// TIA Portal V20 export
// export: Created 2025-12-01T14:56:32.2454153Z, ExportSetting None, DisplayName Totally Integrated Automation Portal, DisplayVersion V20 Update 3, DisplayName TIA Portal Openness, DisplayVersion V20 Update 3, DisplayName TIA Portal Version Control Interface, DisplayVersion V20 Update 3, DisplayName STEP 7 Professional, DisplayVersion V20 Update 3, DisplayName STEP 7 Safety, DisplayVersion V20 Update 2, DisplayName WinCC Basic/Comfort/Advanced, DisplayVersion V20 Update 3, DisplayName WinCC Professional, DisplayVersion V20 Update 3, DisplayName WinCC Unified, DisplayVersion V20 Update 3
FUNCTION_BLOCK "FB450_CRTL_TR_TP_E1_S234_AusSIM+Ord"   // FB450, LAD
TITLE = Control del Ramal de Salidas
{ S7_Optimized_Access := 'FALSE' }
AUTHOR : TLigero
NAME : 20191014
VERSION : 3.3
// FECHA:    19/03/2018  AUTOR: Alonso se parte de E1_S23
//                  19/03/2018                Alonso se mete orden del JdT
// stored: AutoNumber false, SetENOAutomatically false
   VAR_INPUT
      Mesa : UInt;   // Número de mesa
      En_tension : Bool;
      pHsMx_E1 : Bool;   // pHs DE AUSENCIA de la Mesa en E1
      pHsMx_S2 : Bool;   // pHs DE AUSENCIA de la Mesa en S2
      pHsMx_S3 : Bool;   // pHs DE AUSENCIA de la Mesa en S3
      pHsMx_S4 : Bool;   // pHs DE AUSENCIA de la Mesa en S4
      PosTR_E1 : Bool;   // Posicion del TR en E1E3
      PosTR_E2 : Bool;   // Posicion del TR en E2E4
      TP1_Up : Bool;   // TP1 Arriba. E1 >> S3. si no hay tope poner ON
      TP1_Down : Bool;   // TP1 Abajo. E1 >> S3. si no hay tope poner ON
      Termico_E1S3 : Bool;   // Proteccion del Tx en E1E3
      Termico_S2S4 : Bool;   // Proteccion del Tx en E2E4
      Avance_E1S3 : Bool;   // Avance del Tx en E1E3
      Avance_S2S4 : Bool;   // Avance del Tx en E2E4
      PTF_Sal_M2 : Bool;   // S2 >> Mesa Siguiente PTF
      NXT_Avance_S2 : Bool;   // S2 >> Mesa Siguiente avanzando
      PTF_Sal_M3 : Bool;   // S3 >> Mesa Siguiente PTF
      NXT_Avance_S3 : Bool;   // S3 >> Mesa Siguiente avanzando
      PTF_Sal_M4 : Bool;   // S4 >> Mesa Siguiente PTF
      NXT_Avance_S4 : Bool;   // S4 >> Mesa Siguiente avanzando
      F_EnvMens_Mx : Bool;   // Fin de Envio de Mensaje
      Mx_BloqActivo : Bool;   // Bloqueo Activo de la Mesa
      Mx_FlujoPrin_S2 : Bool;   // El flujo principal es Saliendo por S2
      Mx_FlujoPrin_S4 : Bool;   // El flujo principal es Saliendo por S4
      AVTF_MAnt_Mx : Bool;   // E1 >> Mesa Anterior AVTF
      Habilitar_orden_JDT : Bool;   // El JDT tendrá el control del cruce con orden
      ValorOrden_S2 : Word := 16#81;   // Valor de la orden para salir por S2
      ValorOrden_S4 : Word := 16#82;   // Valor de la orden para salir por S4
      MesaS2 : UInt;   // Número de mesa por S2
      MesaS3 : UInt;   // Número de mesa por S3
      MesaS4 : UInt;   // Número de mesa por S4
      Num_Cruce : UInt;   // Número de cruce.
      DB_FIFO_Cruce : UInt := 213;   // DB de la FIFO de ordenes del cruce
      Long_FIFO_Cruce : UInt := 1;   // Longitut de la FIFO de ordenes del cruce
      V_CNT_ApHsMx_E1 : UDInt := 250;   // Valor de Ausencia por E1 en ms
      V_CNT_ApHsMx_S2 : UDInt := 250;   // Valor de Ausencia por S2 en ms
      V_CNT_ApHsMx_S3 : UDInt := 250;   // Valor de Ausencia por S3 en ms
      V_CNT_ApHsMx_S4 : UDInt := 250;   // Valor de Ausencia por S4 en ms
      V_Vaciado : UDInt := 10000;   // Valor de vaciado en ms
      V_Estabilizacion_carga : UDInt := 10;   // en ms
      V_TOut_Tx_Mx : UDInt := 5000;   // TimeOut de Atasco en ms
      V_Avance_S2 : UDInt := 5000;   // en ms
      V_TOut_TR : UDInt := 5000;   // TimeOut de Transfer en ms
      V_TOut_TP : UDInt;   // TimeOut de Tope en ms
      V_Subir_TP_Min : UDInt;   // Valor Minimo para Subir Tope. Decimas de segundo
      V_Bajar_TP_Max : UDInt;   // Valor Maximo para Bajar Tope. Decimas de segundo
      V_Paro : UDInt := 4000;   // tiempo que avanza el transportador sin aviso hasta que se para (ms)
      V_Bloqueo_largo : Time := T#20s;   // tiempo
      V_Bloqueo_corto : Time := T#4s;   // tiempo
   END_VAR
   VAR_OUTPUT
      P_EnvMens_PMx : Bool;   // Permiso de Enviar Mensaje de Presencia
      Etiqueta_Jdt : UDInt;   // Etiqueta que ha sido leida
      Orden_Ejecutada_Jdt : UInt;   // Orden que se ha ejecutado
      PTF_MAnt_Mx : Bool;   // E1 >> Mesa Anterior PTF
      AVTF_Sal_M2 : Bool;   // S2 >> Mesa Siguiente descarga activa
      AVTF_Sal_M3 : Bool;   // S3 >> Mesa Siguiente AVTF
      AVTF_Sal_M4 : Bool;   // S4 >> Mesa Siguiente descarga activa
   END_VAR
   VAR
      T1_ET00 : Bool;
      T1_ET01 : Bool;
      T1_ET02 : Bool;
      T1_ET02_JdT : Bool;
      T1_ET03 : Bool;
      T1_ET10 : Bool;
      T1_ET11 : Bool;
      T1_ET12 : Bool;
      T1_ET50 : Bool;
      T1_ET60 : Bool;
      T1_ET70 : Bool;
      T1_ET80 : Bool;
      T1_ET81 : Bool;
      T1_ET110 : Bool;
      T1_ET111 : Bool;
      T1_ET112 : Bool;
      FIFO_OK : Bool;
      TRANS_OK : Bool;
      O_Bloqueo : Bool;
      Bloqueado : Bool;
      Err_Detec_PHS : Bool;
      FN_ET02 : Bool;
      FN_ET02_JdT : Bool;
      FP_ET02_JdT : Bool;
      FP_ET80 : Bool;
      MemFN_pHsE1 : Bool;
      MemFN_pHsS3 : Bool;
      MemFN_pHsS2 : Bool;
      MemFN_pHsS4 : Bool;
      MemAuxFN_pHsE1 : Bool;
      MemAuxFN_pHsS3 : Bool;
      MemAuxFN_pHsS2 : Bool;
      MemAuxFN_pHsS4 : Bool;
      OK_TmpAusE1 : Bool;
      OK_TmpAusS3 : Bool;
      OK_TmpAusS2 : Bool;
      OK_TmpAusS4 : Bool;
      maux_fp_disparo : Bool;
      ok_vaciado : Bool;
      CNT_Mov_TP : UDInt;
      TmpAus_E1 : UDInt;
      TmpAus_S2 : UDInt;
      TmpAus_S3 : UDInt;
      TmpAus_S4 : UDInt;
      TMP_Paro : UDInt;
      TOUT_Tope : UDInt;
      TOUT_Transfer : UDInt;
      TIMVacido : UDInt;
      TOUT_Atasco : UDInt;
      TOUT_S2 : UDInt;
      TSubidaTR : UDInt;
      TMP_Bloqueo : UDInt;
      TMP_En_Tension : UDInt;
      Datos_Scanner { S7_SetPoint := 'True'} : "ROUT_Orden_Fifo_Scanner";
   END_VAR
   VAR_TEMP
      EstadoZona : "EstadoZona";   // Estado de Zona de la Mesa
      EstadoVI : "EstadosMesa";   // Estado del Vehiculo Inteliguente de la Mesa
      ConfigFB : "UDT_ConfigFB";   // Configuracion de la FB de la Mesa
      TopeUp_EnEntrada : Bool;
      producto_estable : Bool;
      tout_avance_s2 : Bool;
      O_Continuar : Bool;
      O_Entrar_S2 : Bool;
      O_Entrar_S4 : Bool;
      O_Vaciar : Bool;
      JdT_Continuar : Bool;
      JdT_Entrar_S2 : Bool;
      JdT_Entrar_S4 : Bool;
      Moti_ERRO : Bool;
      Moti_NENC : Bool;
      Moti_NORM : Bool;
      Moti_INIC : Bool;
      OK_TP_DW : Bool;
      OK_Paro : Bool;
      t_bloqueo : Bool;
      atasco : Bool;
      timeout_tr : Bool;
      timeout_tope : Bool;
      ok_tension : Bool;
      Aux_W_Moti : Word;
      INT_ORDEN : UInt;
      Aux_W_Orden : Word;
      I_Ord_Filtrada : UInt;
      I_V_Ord_Entrar_S2 : UInt;
      I_V_Ord_Entrar_S4 : UInt;
      V_TMP_BLQ : UDInt;
   END_VAR
   VAR_TEMP   // added for the SCL form of the ladder/FBD networks
      _w1 : Bool;
      _w2 : Bool;
      _w3 : Bool;
      _w4 : Bool;
      _w5 : Bool;
      _w6 : Bool;
      _w7 : Bool;
   END_VAR
BEGIN

REGION Network 1: INICIALIZAR - Recoger las Variables de Estado de la Mesa
   // Se recoge - Estado_CBx
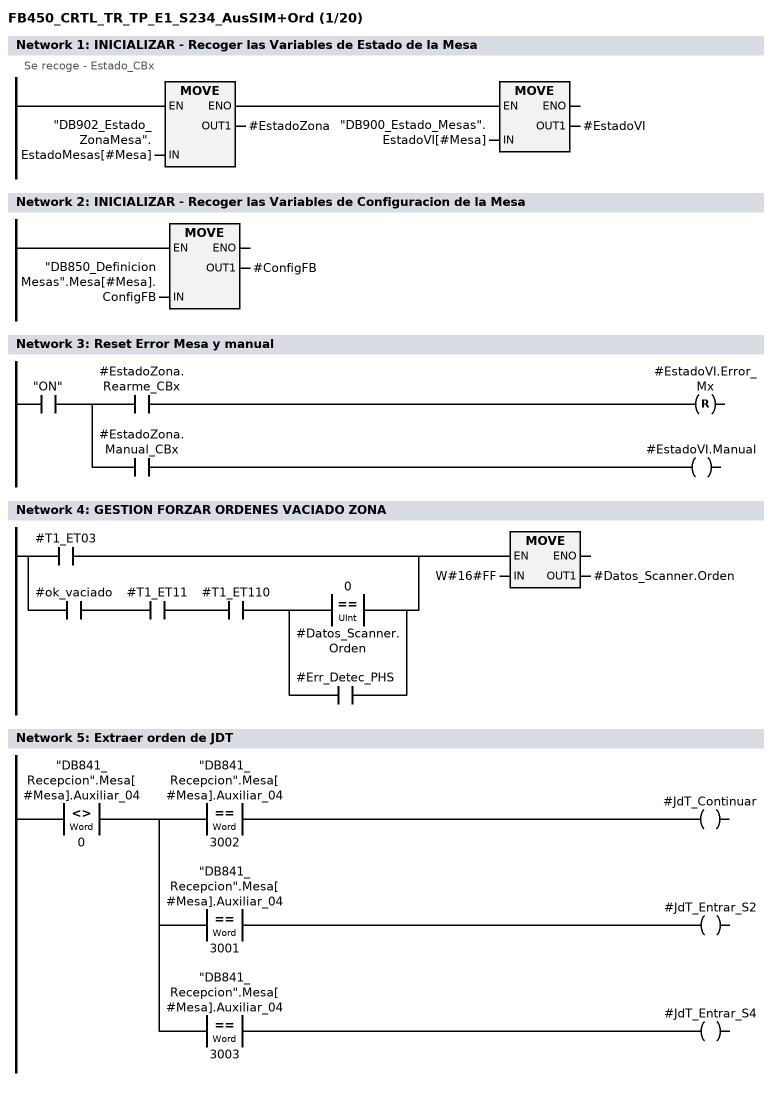
   RUNG wire#powerrail
      Move(in := "DB902_Estado_ZonaMesa".EstadoMesas[#Mesa], out1 => #EstadoZona)
      Move(in := "DB900_Estado_Mesas".EstadoVI[#Mesa], out1 => #EstadoVI)
   END_RUNG
   // the same network as SCL:
   #EstadoZona := "DB902_Estado_ZonaMesa".EstadoMesas[#Mesa];
   #EstadoVI := "DB900_Estado_Mesas".EstadoVI[#Mesa];
END_REGION

REGION Network 2: INICIALIZAR - Recoger las Variables de Configuracion de la Mesa
   RUNG wire#powerrail
      Move(in := "DB850_DefinicionMesas".Mesa[#Mesa].ConfigFB, out1 => #ConfigFB)
   END_RUNG
   // the same network as SCL:
   #ConfigFB := "DB850_DefinicionMesas".Mesa[#Mesa].ConfigFB;
END_REGION

REGION Network 3: Reset Error Mesa y manual
   RUNG wire#powerrail
      Contact( "ON" )
      wire#w1
      Contact( #EstadoZona.Rearme_CBx )
      R_Coil( #EstadoVI.Error_Mx )
   END_RUNG
   RUNG wire#w1
      Contact( #EstadoZona.Manual_CBx )
      Coil( #EstadoVI.Manual )
   END_RUNG
   // the same network as SCL:
   IF "ON" AND #EstadoZona.Rearme_CBx THEN #EstadoVI.Error_Mx := FALSE; END_IF;
   #EstadoVI.Manual := "ON" AND #EstadoZona.Manual_CBx;
END_REGION

REGION Network 4: GESTION FORZAR ORDENES VACIADO ZONA
   RUNG wire#powerrail
      Contact( #T1_ET03 )
      wire#w1
      { S7_GenerateENO := "TRUE" } Move(in := W#16#FF, out1 => #Datos_Scanner.Orden)
   END_RUNG
   RUNG wire#powerrail
      Contact( #ok_vaciado )
      Contact( #T1_ET11 )
      Contact( #T1_ET110 )
      wire#w2
      { S7_Templates := "SrcType := UInt" } EQ_Contact(in1 := 0, in2 := #Datos_Scanner.Orden)
   END_RUNG wire#w1
   RUNG wire#w2
      Contact( #Err_Detec_PHS )
   END_RUNG wire#w1
   // the same network as SCL:
   IF #T1_ET03 OR (#ok_vaciado AND #T1_ET11 AND #T1_ET110 AND ((0 = #Datos_Scanner.Orden) OR #Err_Detec_PHS)) THEN
       #Datos_Scanner.Orden := W#16#FF;
   END_IF;
END_REGION

REGION Network 5: Extraer orden de JDT
   RUNG wire#powerrail
      { S7_Templates := "SrcType := Word" } NE_Contact(in1 := "DB841_Recepcion".Mesa[#Mesa].Auxiliar_04, in2 := 0)
      wire#w1
      { S7_Templates := "SrcType := Word" } EQ_Contact(in1 := "DB841_Recepcion".Mesa[#Mesa].Auxiliar_04, in2 := 3002)
      Coil( #JdT_Continuar )
   END_RUNG
   RUNG wire#w1
      { S7_Templates := "SrcType := Word" } EQ_Contact(in1 := "DB841_Recepcion".Mesa[#Mesa].Auxiliar_04, in2 := 3001)
      Coil( #JdT_Entrar_S2 )
   END_RUNG
   RUNG wire#w1
      { S7_Templates := "SrcType := Word" } EQ_Contact(in1 := "DB841_Recepcion".Mesa[#Mesa].Auxiliar_04, in2 := 3003)
      Coil( #JdT_Entrar_S4 )
   END_RUNG
   // the same network as SCL:
   #_w1 := "DB841_Recepcion".Mesa[#Mesa].Auxiliar_04 <> 0;
   #JdT_Continuar := #_w1 AND ("DB841_Recepcion".Mesa[#Mesa].Auxiliar_04 = 3002);
   #JdT_Entrar_S2 := #_w1 AND ("DB841_Recepcion".Mesa[#Mesa].Auxiliar_04 = 3001);
   #JdT_Entrar_S4 := #_w1 AND ("DB841_Recepcion".Mesa[#Mesa].Auxiliar_04 = 3003);
END_REGION

REGION Network 6: extraer ordenes mesa
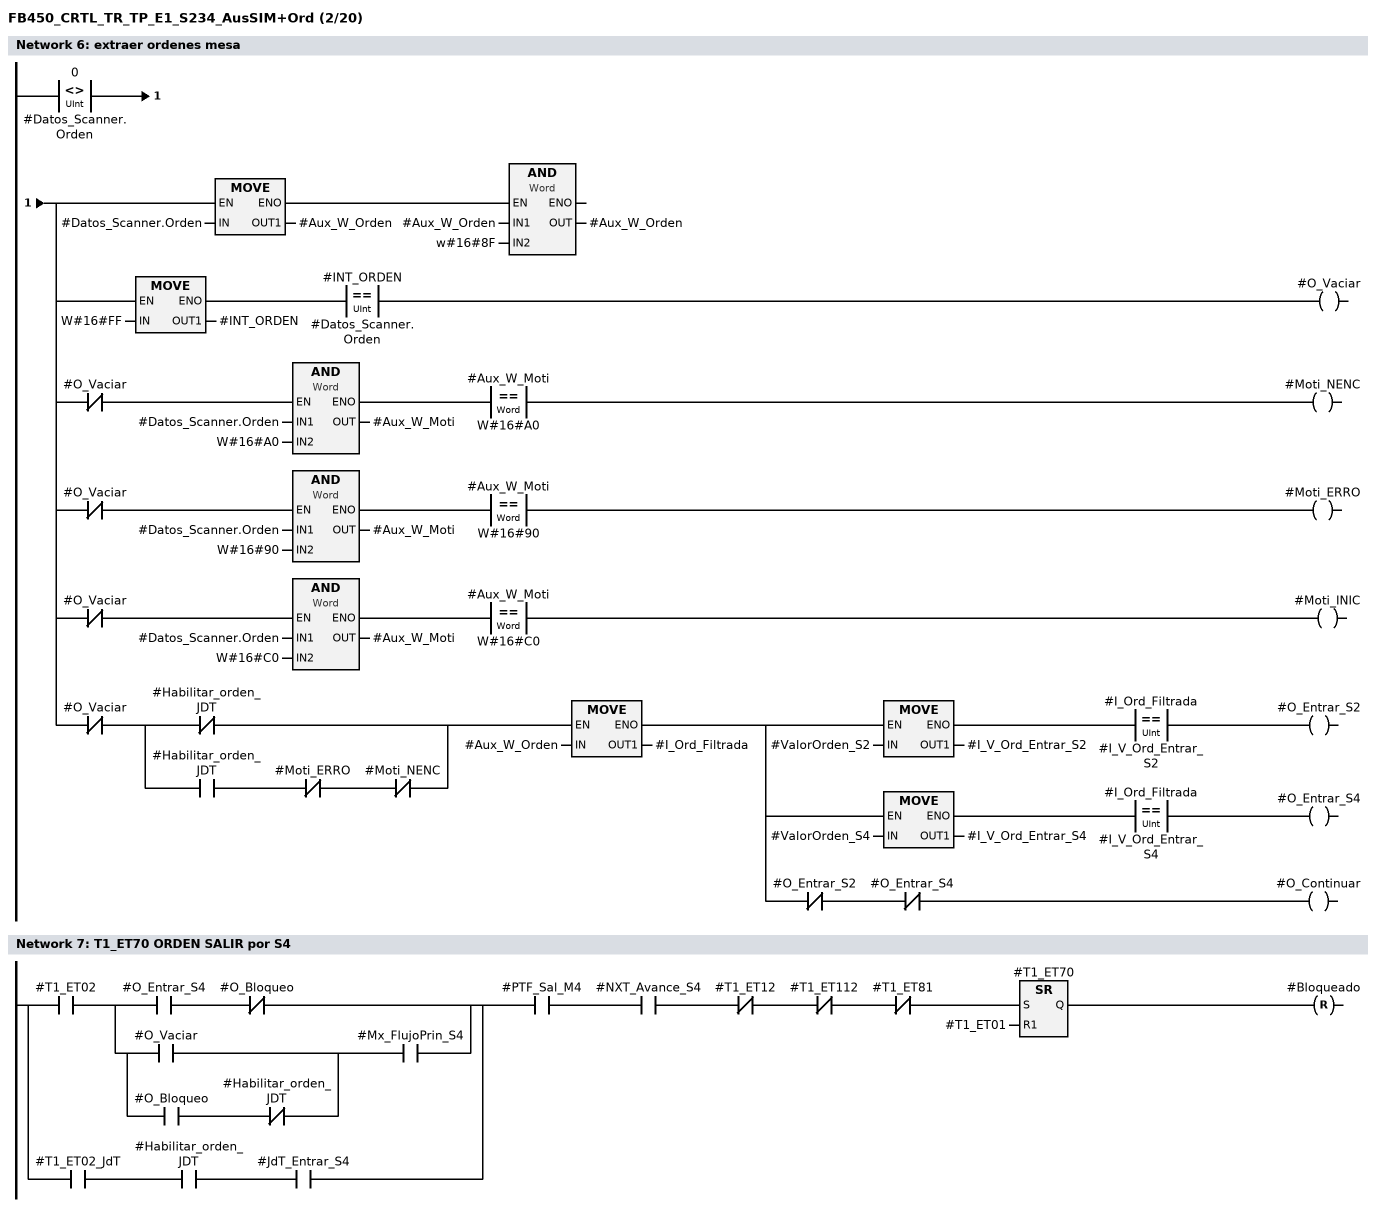
   RUNG wire#powerrail
      { S7_Templates := "SrcType := UInt" } NE_Contact(in1 := 0, in2 := #Datos_Scanner.Orden)
      wire#w1
      { S7_GenerateENO := "TRUE" } Move(in := #Datos_Scanner.Orden, out1 => #Aux_W_Orden)
      { S7_Templates := "SrcType := Word"; S7_GenerateENO := "TRUE" } And(in1 := #Aux_W_Orden, in2 := w#16#8F, out => #Aux_W_Orden)
   END_RUNG
   RUNG wire#w1
      { S7_GenerateENO := "TRUE" } Move(in := W#16#FF, out1 => #INT_ORDEN)
      { S7_Templates := "SrcType := UInt" } EQ_Contact(in1 := #INT_ORDEN, in2 := #Datos_Scanner.Orden)
      Coil( #O_Vaciar )
   END_RUNG
   RUNG wire#w1
      I_Contact( #O_Vaciar )
      { S7_Templates := "SrcType := Word"; S7_GenerateENO := "TRUE" } And(in1 := #Datos_Scanner.Orden, in2 := W#16#A0, out => #Aux_W_Moti)
      { S7_Templates := "SrcType := Word" } EQ_Contact(in1 := #Aux_W_Moti, in2 := W#16#A0)
      Coil( #Moti_NENC )
   END_RUNG
   RUNG wire#w1
      I_Contact( #O_Vaciar )
      { S7_Templates := "SrcType := Word"; S7_GenerateENO := "TRUE" } And(in1 := #Datos_Scanner.Orden, in2 := W#16#90, out => #Aux_W_Moti)
      { S7_Templates := "SrcType := Word" } EQ_Contact(in1 := #Aux_W_Moti, in2 := W#16#90)
      Coil( #Moti_ERRO )
   END_RUNG
   RUNG wire#w1
      I_Contact( #O_Vaciar )
      { S7_Templates := "SrcType := Word"; S7_GenerateENO := "TRUE" } And(in1 := #Datos_Scanner.Orden, in2 := W#16#C0, out => #Aux_W_Moti)
      { S7_Templates := "SrcType := Word" } EQ_Contact(in1 := #Aux_W_Moti, in2 := W#16#C0)
      Coil( #Moti_INIC )
   END_RUNG
   RUNG wire#w1
      I_Contact( #O_Vaciar )
      wire#w2
      I_Contact( #Habilitar_orden_JDT )
      wire#w3
      { S7_GenerateENO := "TRUE" } Move(in := #Aux_W_Orden, out1 => #I_Ord_Filtrada)
      wire#w4
      { S7_GenerateENO := "TRUE" } Move(in := #ValorOrden_S2, out1 => #I_V_Ord_Entrar_S2)
      { S7_Templates := "SrcType := UInt" } EQ_Contact(in1 := #I_Ord_Filtrada, in2 := #I_V_Ord_Entrar_S2)
      Coil( #O_Entrar_S2 )
   END_RUNG
   RUNG wire#w2
      Contact( #Habilitar_orden_JDT )
      I_Contact( #Moti_ERRO )
      I_Contact( #Moti_NENC )
   END_RUNG wire#w3
   RUNG wire#w4
      { S7_GenerateENO := "TRUE" } Move(in := #ValorOrden_S4, out1 => #I_V_Ord_Entrar_S4)
      { S7_Templates := "SrcType := UInt" } EQ_Contact(in1 := #I_Ord_Filtrada, in2 := #I_V_Ord_Entrar_S4)
      Coil( #O_Entrar_S4 )
   END_RUNG
   RUNG wire#w4
      I_Contact( #O_Entrar_S2 )
      I_Contact( #O_Entrar_S4 )
      Coil( #O_Continuar )
   END_RUNG
   // the same network as SCL:
   // ENO of a box is taken as its EN; it also drops when the box reports an error
   #_w1 := 0 <> #Datos_Scanner.Orden;
   IF #_w1 THEN
       #Aux_W_Orden := #Datos_Scanner.Orden;
       #Aux_W_Orden := #Aux_W_Orden AND w#16#8F;
       #INT_ORDEN := W#16#FF;
   END_IF;
   #O_Vaciar := #_w1 AND (#INT_ORDEN = #Datos_Scanner.Orden);
   #_w2 := #_w1 AND NOT #O_Vaciar;
   IF #_w2 THEN #Aux_W_Moti := #Datos_Scanner.Orden AND W#16#A0; END_IF;
   #Moti_NENC := #_w2 AND (#Aux_W_Moti = W#16#A0);
   #_w3 := #_w1 AND NOT #O_Vaciar;
   IF #_w3 THEN #Aux_W_Moti := #Datos_Scanner.Orden AND W#16#90; END_IF;
   #Moti_ERRO := #_w3 AND (#Aux_W_Moti = W#16#90);
   #_w4 := #_w1 AND NOT #O_Vaciar;
   IF #_w4 THEN #Aux_W_Moti := #Datos_Scanner.Orden AND W#16#C0; END_IF;
   #Moti_INIC := #_w4 AND (#Aux_W_Moti = W#16#C0);
   #_w5 := #_w1 AND NOT #O_Vaciar AND (NOT #Habilitar_orden_JDT OR (#Habilitar_orden_JDT AND NOT #Moti_ERRO AND NOT #Moti_NENC));
   IF #_w5 THEN
       #I_Ord_Filtrada := #Aux_W_Orden;
       #I_V_Ord_Entrar_S2 := #ValorOrden_S2;
   END_IF;
   #O_Entrar_S2 := #_w5 AND (#I_Ord_Filtrada = #I_V_Ord_Entrar_S2);
   IF #_w5 THEN #I_V_Ord_Entrar_S4 := #ValorOrden_S4; END_IF;
   #O_Entrar_S4 := #_w5 AND (#I_Ord_Filtrada = #I_V_Ord_Entrar_S4);
   #O_Continuar := #_w5 AND NOT #O_Entrar_S2 AND NOT #O_Entrar_S4;
END_REGION

REGION Network 7: T1_ET70 ORDEN SALIR por S4
   RUNG wire#powerrail
      Contact( #T1_ET02 )
      wire#w1
      Contact( #O_Entrar_S4 )
      I_Contact( #O_Bloqueo )
      wire#w2
      Contact( #PTF_Sal_M4 )
      Contact( #NXT_Avance_S4 )
      I_Contact( #T1_ET12 )
      I_Contact( #T1_ET112 )
      I_Contact( #T1_ET81 )
      S_SR(operand := #T1_ET70, r1 := #T1_ET01)
      R_Coil( #Bloqueado )
   END_RUNG
   RUNG wire#w1
      Contact( #O_Vaciar )
      wire#w3
      Contact( #Mx_FlujoPrin_S4 )
   END_RUNG wire#w2
   RUNG wire#w1
      Contact( #O_Bloqueo )
      I_Contact( #Habilitar_orden_JDT )
   END_RUNG wire#w3
   RUNG wire#powerrail
      Contact( #T1_ET02_JdT )
      Contact( #Habilitar_orden_JDT )
      Contact( #JdT_Entrar_S4 )
   END_RUNG wire#w2
   // the same network as SCL:
   IF ((#T1_ET02 AND ((#O_Entrar_S4 AND NOT #O_Bloqueo) OR ((#O_Vaciar OR (#O_Bloqueo AND NOT #Habilitar_orden_JDT)) AND #Mx_FlujoPrin_S4))) OR (#T1_ET02_JdT AND #Habilitar_orden_JDT AND #JdT_Entrar_S4)) AND #PTF_Sal_M4 AND #NXT_Avance_S4 AND NOT #T1_ET12 AND NOT #T1_ET112 AND NOT #T1_ET81 THEN
       #T1_ET70 := TRUE;   // SR flip-flop
   END_IF;
   IF #T1_ET01 THEN #T1_ET70 := FALSE; END_IF;
   IF #T1_ET70 THEN #Bloqueado := FALSE; END_IF;
END_REGION

REGION Network 8: T1_ET60 ORDEN SALIR por S2
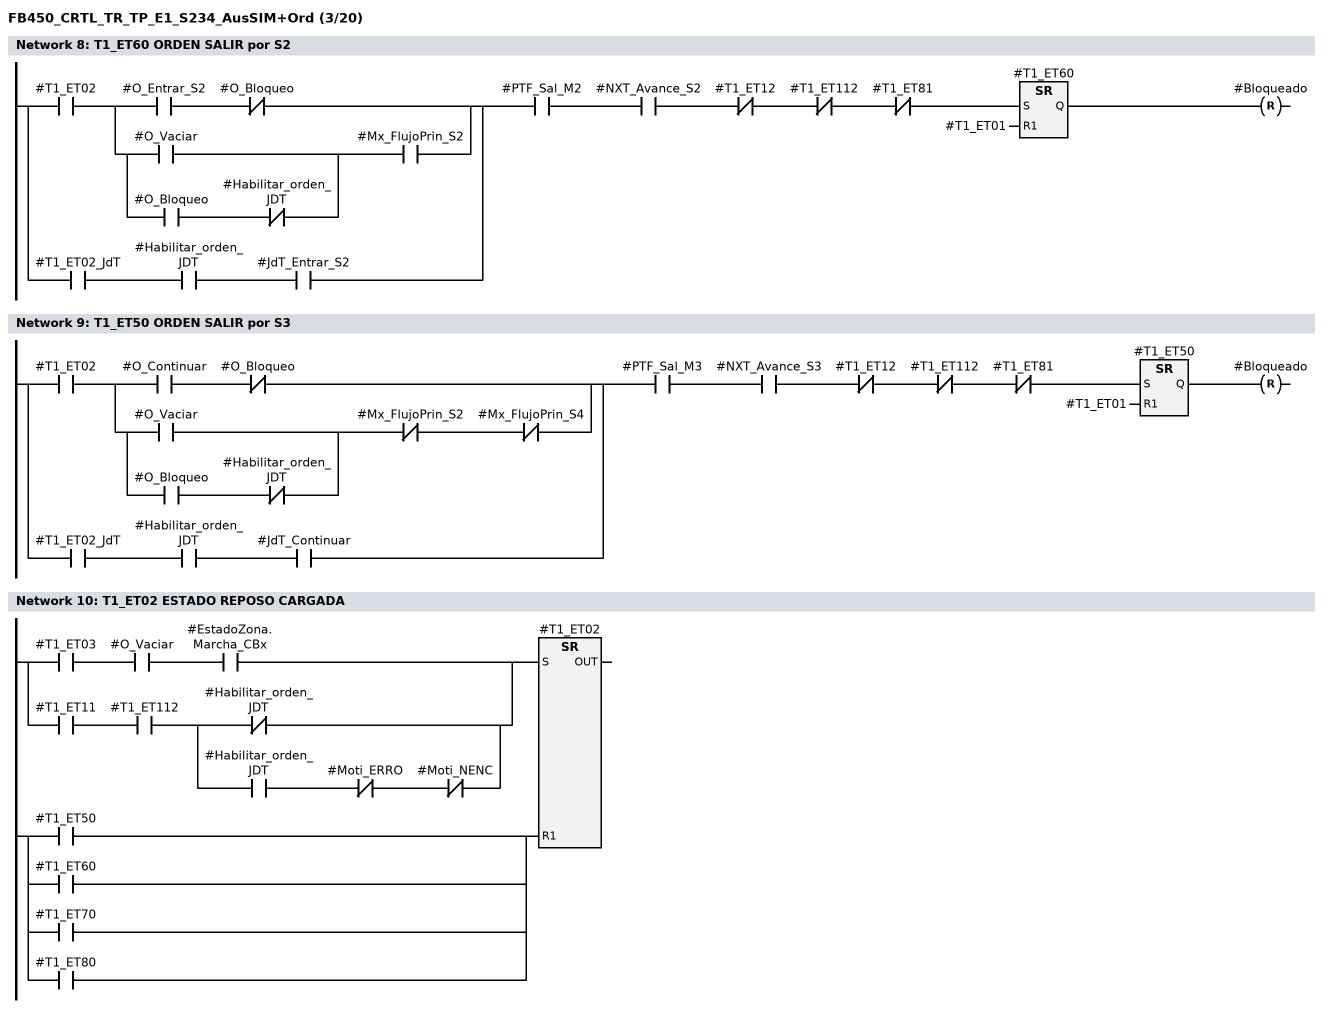
   RUNG wire#powerrail
      Contact( #T1_ET02 )
      wire#w1
      Contact( #O_Entrar_S2 )
      I_Contact( #O_Bloqueo )
      wire#w2
      Contact( #PTF_Sal_M2 )
      Contact( #NXT_Avance_S2 )
      I_Contact( #T1_ET12 )
      I_Contact( #T1_ET112 )
      I_Contact( #T1_ET81 )
      S_SR(operand := #T1_ET60, r1 := #T1_ET01)
      R_Coil( #Bloqueado )
   END_RUNG
   RUNG wire#w1
      Contact( #O_Vaciar )
      wire#w3
      Contact( #Mx_FlujoPrin_S2 )
   END_RUNG wire#w2
   RUNG wire#w1
      Contact( #O_Bloqueo )
      I_Contact( #Habilitar_orden_JDT )
   END_RUNG wire#w3
   RUNG wire#powerrail
      Contact( #T1_ET02_JdT )
      Contact( #Habilitar_orden_JDT )
      Contact( #JdT_Entrar_S2 )
   END_RUNG wire#w2
   // the same network as SCL:
   IF ((#T1_ET02 AND ((#O_Entrar_S2 AND NOT #O_Bloqueo) OR ((#O_Vaciar OR (#O_Bloqueo AND NOT #Habilitar_orden_JDT)) AND #Mx_FlujoPrin_S2))) OR (#T1_ET02_JdT AND #Habilitar_orden_JDT AND #JdT_Entrar_S2)) AND #PTF_Sal_M2 AND #NXT_Avance_S2 AND NOT #T1_ET12 AND NOT #T1_ET112 AND NOT #T1_ET81 THEN
       #T1_ET60 := TRUE;   // SR flip-flop
   END_IF;
   IF #T1_ET01 THEN #T1_ET60 := FALSE; END_IF;
   IF #T1_ET60 THEN #Bloqueado := FALSE; END_IF;
END_REGION

REGION Network 9: T1_ET50 ORDEN SALIR por S3
   RUNG wire#powerrail
      Contact( #T1_ET02 )
      wire#w1
      Contact( #O_Continuar )
      I_Contact( #O_Bloqueo )
      wire#w2
      Contact( #PTF_Sal_M3 )
      Contact( #NXT_Avance_S3 )
      I_Contact( #T1_ET12 )
      I_Contact( #T1_ET112 )
      I_Contact( #T1_ET81 )
      S_SR(operand := #T1_ET50, r1 := #T1_ET01)
      R_Coil( #Bloqueado )
   END_RUNG
   RUNG wire#w1
      Contact( #O_Vaciar )
      wire#w3
      I_Contact( #Mx_FlujoPrin_S2 )
      I_Contact( #Mx_FlujoPrin_S4 )
   END_RUNG wire#w2
   RUNG wire#w1
      Contact( #O_Bloqueo )
      I_Contact( #Habilitar_orden_JDT )
   END_RUNG wire#w3
   RUNG wire#powerrail
      Contact( #T1_ET02_JdT )
      Contact( #Habilitar_orden_JDT )
      Contact( #JdT_Continuar )
   END_RUNG wire#w2
   // the same network as SCL:
   IF ((#T1_ET02 AND ((#O_Continuar AND NOT #O_Bloqueo) OR ((#O_Vaciar OR (#O_Bloqueo AND NOT #Habilitar_orden_JDT)) AND NOT #Mx_FlujoPrin_S2 AND NOT #Mx_FlujoPrin_S4))) OR (#T1_ET02_JdT AND #Habilitar_orden_JDT AND #JdT_Continuar)) AND #PTF_Sal_M3 AND #NXT_Avance_S3 AND NOT #T1_ET12 AND NOT #T1_ET112 AND NOT #T1_ET81 THEN
       #T1_ET50 := TRUE;   // SR flip-flop
   END_IF;
   IF #T1_ET01 THEN #T1_ET50 := FALSE; END_IF;
   IF #T1_ET50 THEN #Bloqueado := FALSE; END_IF;
END_REGION

REGION Network 10: T1_ET02 ESTADO REPOSO CARGADA
   RUNG wire#powerrail
      Contact( #T1_ET03 )
      Contact( #O_Vaciar )
      Contact( #EstadoZona.Marcha_CBx )
      wire#w1
      S_SR(operand := #T1_ET02, r1 := wire#w3)
   END_RUNG
   RUNG wire#powerrail
      Contact( #T1_ET11 )
      Contact( #T1_ET112 )
      wire#w2
      I_Contact( #Habilitar_orden_JDT )
   END_RUNG wire#w1
   RUNG wire#w2
      Contact( #Habilitar_orden_JDT )
      I_Contact( #Moti_ERRO )
      I_Contact( #Moti_NENC )
   END_RUNG wire#w1
   RUNG wire#powerrail
      Contact( #T1_ET50 )
   END_RUNG wire#w3
   RUNG wire#powerrail
      Contact( #T1_ET60 )
   END_RUNG wire#w3
   RUNG wire#powerrail
      Contact( #T1_ET70 )
   END_RUNG wire#w3
   RUNG wire#powerrail
      Contact( #T1_ET80 )
   END_RUNG wire#w3
   // the same network as SCL:
   IF (#T1_ET03 AND #O_Vaciar AND #EstadoZona.Marcha_CBx) OR (#T1_ET11 AND #T1_ET112 AND (NOT #Habilitar_orden_JDT OR (#Habilitar_orden_JDT AND NOT #Moti_ERRO AND NOT #Moti_NENC))) THEN
       #T1_ET02 := TRUE;   // SR flip-flop
   END_IF;
   IF #T1_ET50 OR #T1_ET60 OR #T1_ET70 OR #T1_ET80 THEN #T1_ET02 := FALSE; END_IF;
END_REGION

REGION Network 11: T1_ET02_JDT --- REPOSO CARGADA A LA ESPERA DE ORDEN DE JDT
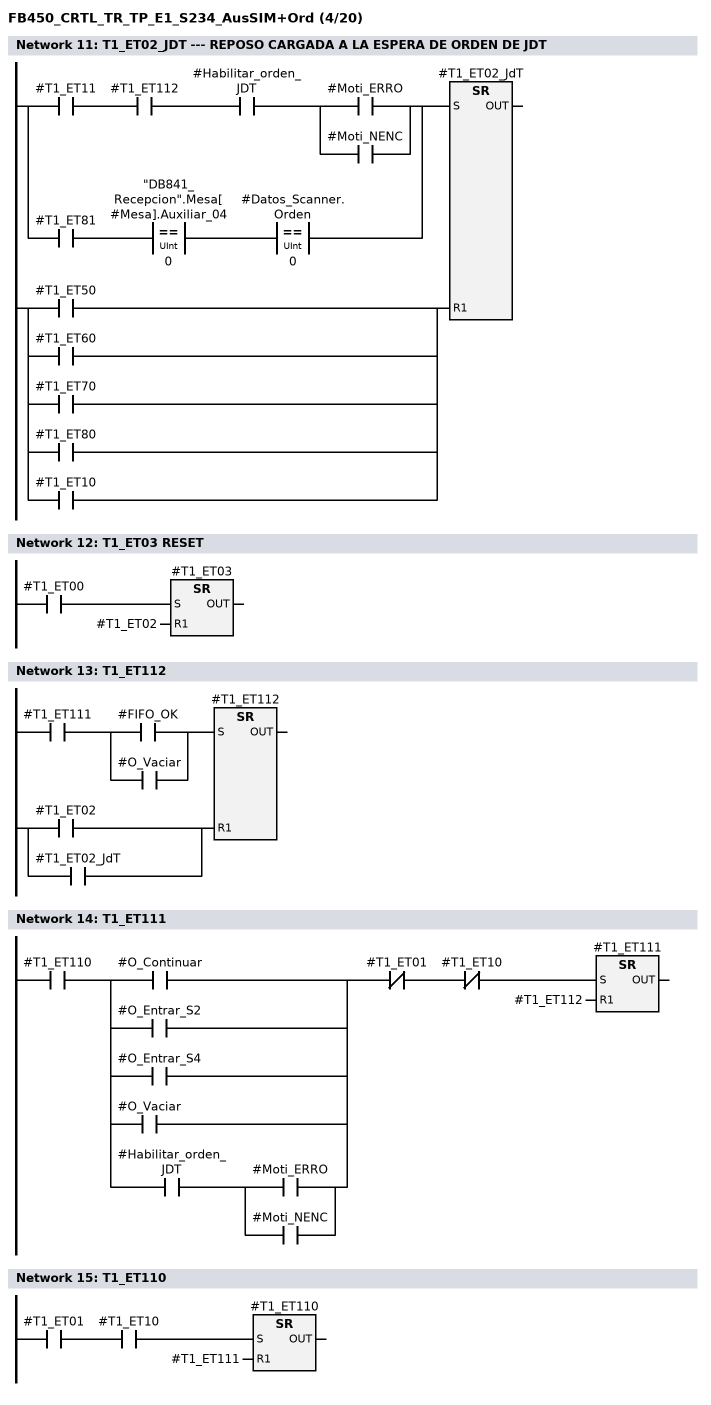
   RUNG wire#powerrail
      Contact( #T1_ET11 )
      Contact( #T1_ET112 )
      Contact( #Habilitar_orden_JDT )
      wire#w1
      Contact( #Moti_ERRO )
      wire#w2
      S_SR(operand := #T1_ET02_JdT, r1 := wire#w3)
   END_RUNG
   RUNG wire#w1
      Contact( #Moti_NENC )
   END_RUNG wire#w2
   RUNG wire#powerrail
      Contact( #T1_ET81 )
      { S7_Templates := "SrcType := UInt" } EQ_Contact(in1 := "DB841_Recepcion".Mesa[#Mesa].Auxiliar_04, in2 := 0)
      { S7_Templates := "SrcType := UInt" } EQ_Contact(in1 := #Datos_Scanner.Orden, in2 := 0)
   END_RUNG wire#w2
   RUNG wire#powerrail
      Contact( #T1_ET50 )
   END_RUNG wire#w3
   RUNG wire#powerrail
      Contact( #T1_ET60 )
   END_RUNG wire#w3
   RUNG wire#powerrail
      Contact( #T1_ET70 )
   END_RUNG wire#w3
   RUNG wire#powerrail
      Contact( #T1_ET80 )
   END_RUNG wire#w3
   RUNG wire#powerrail
      Contact( #T1_ET10 )
   END_RUNG wire#w3
   // the same network as SCL:
   IF (#T1_ET11 AND #T1_ET112 AND #Habilitar_orden_JDT AND (#Moti_ERRO OR #Moti_NENC)) OR (#T1_ET81 AND ("DB841_Recepcion".Mesa[#Mesa].Auxiliar_04 = 0) AND (#Datos_Scanner.Orden = 0)) THEN
       #T1_ET02_JdT := TRUE;   // SR flip-flop
   END_IF;
   IF #T1_ET50 OR #T1_ET60 OR #T1_ET70 OR #T1_ET80 OR #T1_ET10 THEN #T1_ET02_JdT := FALSE; END_IF;
END_REGION

REGION Network 12: T1_ET03 RESET
   RUNG wire#powerrail
      Contact( #T1_ET00 )
      S_SR(operand := #T1_ET03, r1 := #T1_ET02)
   END_RUNG
   // the same network as SCL:
   IF #T1_ET00 THEN
       #T1_ET03 := TRUE;   // SR flip-flop
   END_IF;
   IF #T1_ET02 THEN #T1_ET03 := FALSE; END_IF;
END_REGION

REGION Network 13: T1_ET112
   RUNG wire#powerrail
      Contact( #T1_ET111 )
      wire#w1
      Contact( #FIFO_OK )
      wire#w2
      S_SR(operand := #T1_ET112, r1 := wire#w3)
   END_RUNG
   RUNG wire#w1
      Contact( #O_Vaciar )
   END_RUNG wire#w2
   RUNG wire#powerrail
      Contact( #T1_ET02 )
   END_RUNG wire#w3
   RUNG wire#powerrail
      Contact( #T1_ET02_JdT )
   END_RUNG wire#w3
   // the same network as SCL:
   IF #T1_ET111 AND (#FIFO_OK OR #O_Vaciar) THEN
       #T1_ET112 := TRUE;   // SR flip-flop
   END_IF;
   IF #T1_ET02 OR #T1_ET02_JdT THEN #T1_ET112 := FALSE; END_IF;
END_REGION

REGION Network 14: T1_ET111
   RUNG wire#powerrail
      Contact( #T1_ET110 )
      wire#w1
      Contact( #O_Continuar )
      wire#w2
      I_Contact( #T1_ET01 )
      I_Contact( #T1_ET10 )
      S_SR(operand := #T1_ET111, r1 := #T1_ET112)
   END_RUNG
   RUNG wire#w1
      Contact( #O_Entrar_S2 )
   END_RUNG wire#w2
   RUNG wire#w1
      Contact( #O_Entrar_S4 )
   END_RUNG wire#w2
   RUNG wire#w1
      Contact( #O_Vaciar )
   END_RUNG wire#w2
   RUNG wire#w1
      Contact( #Habilitar_orden_JDT )
      wire#w3
      Contact( #Moti_ERRO )
   END_RUNG wire#w2
   RUNG wire#w3
      Contact( #Moti_NENC )
   END_RUNG wire#w2
   // the same network as SCL:
   IF #T1_ET110 AND (#O_Continuar OR #O_Entrar_S2 OR #O_Entrar_S4 OR #O_Vaciar OR (#Habilitar_orden_JDT AND (#Moti_ERRO OR #Moti_NENC))) AND NOT #T1_ET01 AND NOT #T1_ET10 THEN
       #T1_ET111 := TRUE;   // SR flip-flop
   END_IF;
   IF #T1_ET112 THEN #T1_ET111 := FALSE; END_IF;
END_REGION

REGION Network 15: T1_ET110
   RUNG wire#powerrail
      Contact( #T1_ET01 )
      Contact( #T1_ET10 )
      S_SR(operand := #T1_ET110, r1 := #T1_ET111)
   END_RUNG
   // the same network as SCL:
   IF #T1_ET01 AND #T1_ET10 THEN
       #T1_ET110 := TRUE;   // SR flip-flop
   END_IF;
   IF #T1_ET111 THEN #T1_ET110 := FALSE; END_IF;
END_REGION

REGION Network 16: T1_ET11
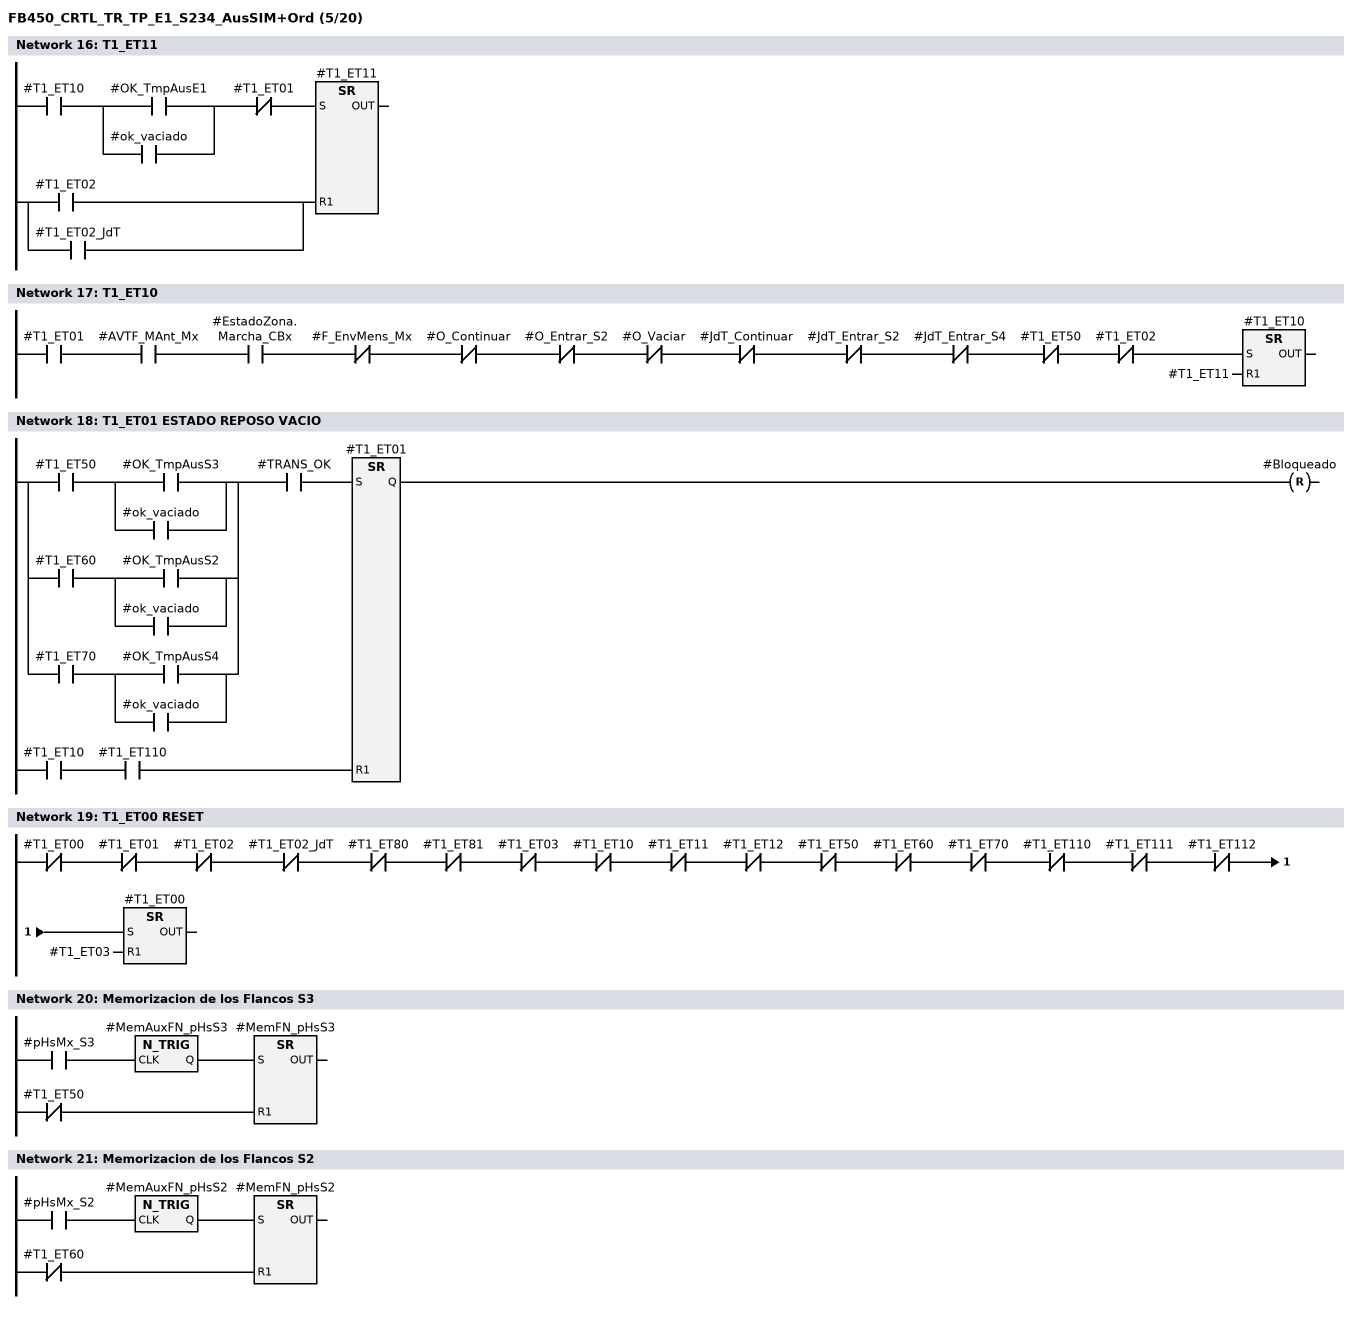
   RUNG wire#powerrail
      Contact( #T1_ET10 )
      wire#w1
      Contact( #OK_TmpAusE1 )
      wire#w2
      I_Contact( #T1_ET01 )
      S_SR(operand := #T1_ET11, r1 := wire#w3)
   END_RUNG
   RUNG wire#w1
      Contact( #ok_vaciado )
   END_RUNG wire#w2
   RUNG wire#powerrail
      Contact( #T1_ET02 )
   END_RUNG wire#w3
   RUNG wire#powerrail
      Contact( #T1_ET02_JdT )
   END_RUNG wire#w3
   // the same network as SCL:
   IF #T1_ET10 AND (#OK_TmpAusE1 OR #ok_vaciado) AND NOT #T1_ET01 THEN
       #T1_ET11 := TRUE;   // SR flip-flop
   END_IF;
   IF #T1_ET02 OR #T1_ET02_JdT THEN #T1_ET11 := FALSE; END_IF;
END_REGION

REGION Network 17: T1_ET10
   RUNG wire#powerrail
      Contact( #T1_ET01 )
      Contact( #AVTF_MAnt_Mx )
      Contact( #EstadoZona.Marcha_CBx )
      I_Contact( #F_EnvMens_Mx )
      I_Contact( #O_Continuar )
      I_Contact( #O_Entrar_S2 )
      I_Contact( #O_Vaciar )
      I_Contact( #JdT_Continuar )
      I_Contact( #JdT_Entrar_S2 )
      I_Contact( #JdT_Entrar_S4 )
      I_Contact( #T1_ET50 )
      I_Contact( #T1_ET02 )
      S_SR(operand := #T1_ET10, r1 := #T1_ET11)
   END_RUNG
   // the same network as SCL:
   IF #T1_ET01 AND #AVTF_MAnt_Mx AND #EstadoZona.Marcha_CBx AND NOT #F_EnvMens_Mx AND NOT #O_Continuar AND NOT #O_Entrar_S2 AND NOT #O_Vaciar AND NOT #JdT_Continuar AND NOT #JdT_Entrar_S2 AND NOT #JdT_Entrar_S4 AND NOT #T1_ET50 AND NOT #T1_ET02 THEN
       #T1_ET10 := TRUE;   // SR flip-flop
   END_IF;
   IF #T1_ET11 THEN #T1_ET10 := FALSE; END_IF;
END_REGION

REGION Network 18: T1_ET01 ESTADO REPOSO VACIO
   RUNG wire#powerrail
      Contact( #T1_ET50 )
      wire#w1
      Contact( #OK_TmpAusS3 )
      wire#w2
      Contact( #TRANS_OK )
      S_SR(operand := #T1_ET01, r1 := wire#w5)
      R_Coil( #Bloqueado )
   END_RUNG
   RUNG wire#w1
      Contact( #ok_vaciado )
   END_RUNG wire#w2
   RUNG wire#powerrail
      Contact( #T1_ET60 )
      wire#w3
      Contact( #OK_TmpAusS2 )
   END_RUNG wire#w2
   RUNG wire#w3
      Contact( #ok_vaciado )
   END_RUNG wire#w2
   RUNG wire#powerrail
      Contact( #T1_ET70 )
      wire#w4
      Contact( #OK_TmpAusS4 )
   END_RUNG wire#w2
   RUNG wire#w4
      Contact( #ok_vaciado )
   END_RUNG wire#w2
   RUNG wire#powerrail
      Contact( #T1_ET10 )
      Contact( #T1_ET110 )
   END_RUNG wire#w5
   // the same network as SCL:
   IF ((#T1_ET50 AND (#OK_TmpAusS3 OR #ok_vaciado)) OR (#T1_ET60 AND (#OK_TmpAusS2 OR #ok_vaciado)) OR (#T1_ET70 AND (#OK_TmpAusS4 OR #ok_vaciado))) AND #TRANS_OK THEN
       #T1_ET01 := TRUE;   // SR flip-flop
   END_IF;
   IF #T1_ET10 AND #T1_ET110 THEN #T1_ET01 := FALSE; END_IF;
   IF #T1_ET01 THEN #Bloqueado := FALSE; END_IF;
END_REGION

REGION Network 19: T1_ET00 RESET
   RUNG wire#powerrail
      I_Contact( #T1_ET00 )
      I_Contact( #T1_ET01 )
      I_Contact( #T1_ET02 )
      I_Contact( #T1_ET02_JdT )
      I_Contact( #T1_ET80 )
      I_Contact( #T1_ET81 )
      I_Contact( #T1_ET03 )
      I_Contact( #T1_ET10 )
      I_Contact( #T1_ET11 )
      I_Contact( #T1_ET12 )
      I_Contact( #T1_ET50 )
      I_Contact( #T1_ET60 )
      I_Contact( #T1_ET70 )
      I_Contact( #T1_ET110 )
      I_Contact( #T1_ET111 )
      I_Contact( #T1_ET112 )
      S_SR(operand := #T1_ET00, r1 := #T1_ET03)
   END_RUNG
   // the same network as SCL:
   IF NOT #T1_ET00 AND NOT #T1_ET01 AND NOT #T1_ET02 AND NOT #T1_ET02_JdT AND NOT #T1_ET80 AND NOT #T1_ET81 AND NOT #T1_ET03 AND NOT #T1_ET10 AND NOT #T1_ET11 AND NOT #T1_ET12 AND NOT #T1_ET50 AND NOT #T1_ET60 AND NOT #T1_ET70 AND NOT #T1_ET110 AND NOT #T1_ET111 AND NOT #T1_ET112 THEN
       #T1_ET00 := TRUE;   // SR flip-flop
   END_IF;
   IF #T1_ET03 THEN #T1_ET00 := FALSE; END_IF;
END_REGION

REGION Network 20: Memorizacion de los Flancos S3
   RUNG wire#powerrail
      Contact( #pHsMx_S3 )
      N_Trig( #MemAuxFN_pHsS3 )
      S_SR(operand := #MemFN_pHsS3, r1 := wire#w1)
   END_RUNG
   RUNG wire#powerrail
      I_Contact( #T1_ET50 )
   END_RUNG wire#w1
   // the same network as SCL:
   #_w1 := NOT #pHsMx_S3 AND #MemAuxFN_pHsS3;   // falling edge
   #MemAuxFN_pHsS3 := #pHsMx_S3;
   IF #_w1 THEN
       #MemFN_pHsS3 := TRUE;   // SR flip-flop
   END_IF;
   IF NOT #T1_ET50 THEN #MemFN_pHsS3 := FALSE; END_IF;
END_REGION

REGION Network 21: Memorizacion de los Flancos S2
   RUNG wire#powerrail
      Contact( #pHsMx_S2 )
      N_Trig( #MemAuxFN_pHsS2 )
      S_SR(operand := #MemFN_pHsS2, r1 := wire#w1)
   END_RUNG
   RUNG wire#powerrail
      I_Contact( #T1_ET60 )
   END_RUNG wire#w1
   // the same network as SCL:
   #_w1 := NOT #pHsMx_S2 AND #MemAuxFN_pHsS2;   // falling edge
   #MemAuxFN_pHsS2 := #pHsMx_S2;
   IF #_w1 THEN
       #MemFN_pHsS2 := TRUE;   // SR flip-flop
   END_IF;
   IF NOT #T1_ET60 THEN #MemFN_pHsS2 := FALSE; END_IF;
END_REGION

REGION Network 22: Memorizacion de los Flancos S4
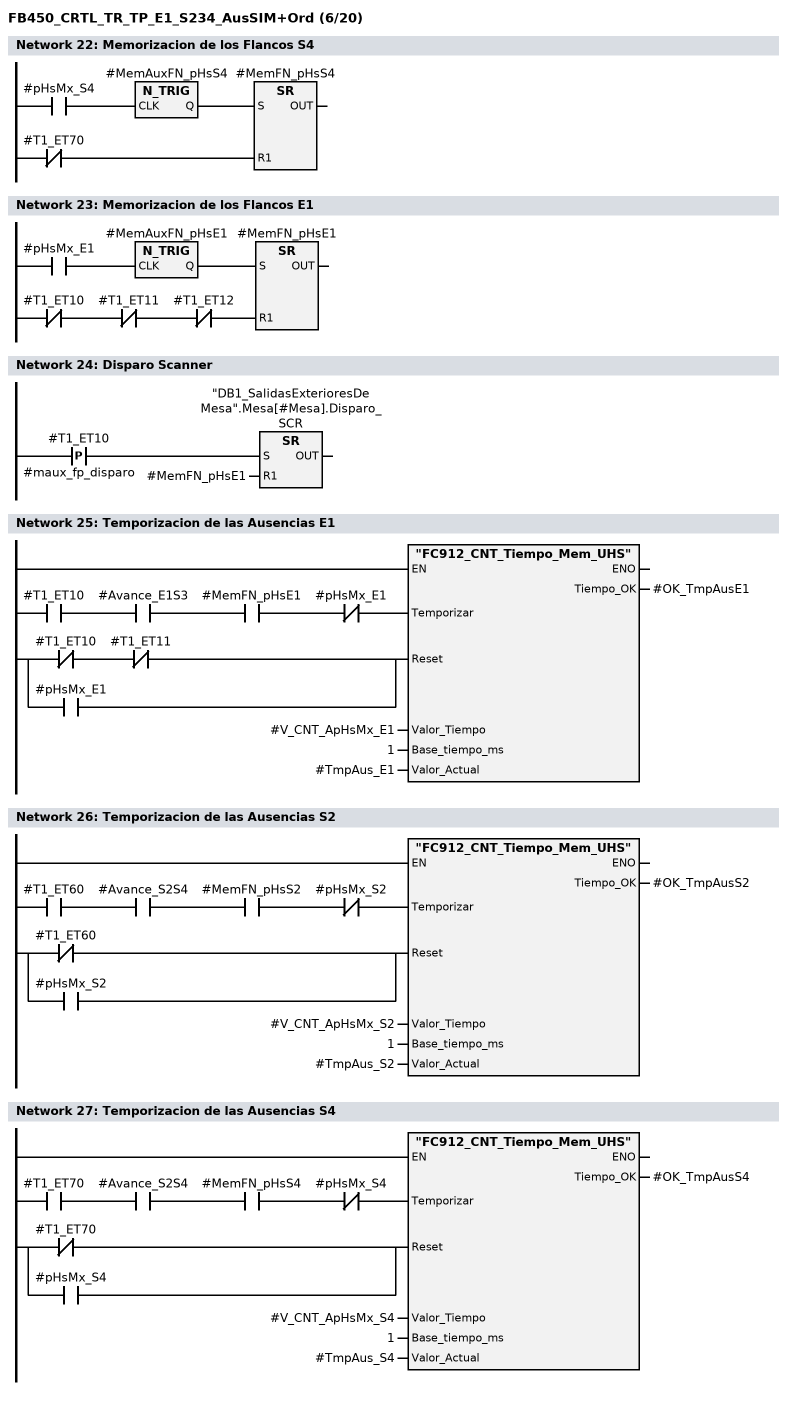
   RUNG wire#powerrail
      Contact( #pHsMx_S4 )
      N_Trig( #MemAuxFN_pHsS4 )
      S_SR(operand := #MemFN_pHsS4, r1 := wire#w1)
   END_RUNG
   RUNG wire#powerrail
      I_Contact( #T1_ET70 )
   END_RUNG wire#w1
   // the same network as SCL:
   #_w1 := NOT #pHsMx_S4 AND #MemAuxFN_pHsS4;   // falling edge
   #MemAuxFN_pHsS4 := #pHsMx_S4;
   IF #_w1 THEN
       #MemFN_pHsS4 := TRUE;   // SR flip-flop
   END_IF;
   IF NOT #T1_ET70 THEN #MemFN_pHsS4 := FALSE; END_IF;
END_REGION

REGION Network 23: Memorizacion de los Flancos E1
   RUNG wire#powerrail
      Contact( #pHsMx_E1 )
      N_Trig( #MemAuxFN_pHsE1 )
      S_SR(operand := #MemFN_pHsE1, r1 := wire#w1)
   END_RUNG
   RUNG wire#powerrail
      I_Contact( #T1_ET10 )
      I_Contact( #T1_ET11 )
      I_Contact( #T1_ET12 )
   END_RUNG wire#w1
   // the same network as SCL:
   #_w1 := NOT #pHsMx_E1 AND #MemAuxFN_pHsE1;   // falling edge
   #MemAuxFN_pHsE1 := #pHsMx_E1;
   IF #_w1 THEN
       #MemFN_pHsE1 := TRUE;   // SR flip-flop
   END_IF;
   IF NOT #T1_ET10 AND NOT #T1_ET11 AND NOT #T1_ET12 THEN #MemFN_pHsE1 := FALSE; END_IF;
END_REGION

REGION Network 24: Disparo Scanner
   RUNG wire#powerrail
      P_Contact(operand := #T1_ET10, bit := #maux_fp_disparo)
      S_SR(operand := "DB1_SalidasExterioresDeMesa".Mesa[#Mesa].Disparo_SCR, r1 := #MemFN_pHsE1)
   END_RUNG
   // the same network as SCL:
   #_w1 := #T1_ET10 AND NOT #maux_fp_disparo;   // rising edge of #T1_ET10
   #maux_fp_disparo := #T1_ET10;
   IF #_w1 THEN
       "DB1_SalidasExterioresDeMesa".Mesa[#Mesa].Disparo_SCR := TRUE;   // SR flip-flop
   END_IF;
   IF #MemFN_pHsE1 THEN "DB1_SalidasExterioresDeMesa".Mesa[#Mesa].Disparo_SCR := FALSE; END_IF;
END_REGION

REGION Network 25: Temporizacion de las Ausencias E1
   RUNG wire#powerrail
      "FC912_CNT_Tiempo_Mem_UHS"(Temporizar := wire#w1, Reset := wire#w2, Valor_Tiempo := #V_CNT_ApHsMx_E1, Base_tiempo_ms := 1, Valor_Actual := #TmpAus_E1, Tiempo_OK => #OK_TmpAusE1)
   END_RUNG
   RUNG wire#powerrail
      Contact( #T1_ET10 )
      Contact( #Avance_E1S3 )
      Contact( #MemFN_pHsE1 )
      I_Contact( #pHsMx_E1 )
   END_RUNG wire#w1
   RUNG wire#powerrail
      I_Contact( #T1_ET10 )
      I_Contact( #T1_ET11 )
   END_RUNG wire#w2
   RUNG wire#powerrail
      Contact( #pHsMx_E1 )
   END_RUNG wire#w2
   // the same network as SCL:
   "FC912_CNT_Tiempo_Mem_UHS"(Temporizar := #T1_ET10 AND #Avance_E1S3 AND #MemFN_pHsE1 AND NOT #pHsMx_E1,
                           Reset := (NOT #T1_ET10 AND NOT #T1_ET11) OR #pHsMx_E1,
                           Valor_Tiempo := #V_CNT_ApHsMx_E1,
                           Base_tiempo_ms := 1,
                           Valor_Actual := #TmpAus_E1,
                           Tiempo_OK => #OK_TmpAusE1);
END_REGION

REGION Network 26: Temporizacion de las Ausencias S2
   RUNG wire#powerrail
      "FC912_CNT_Tiempo_Mem_UHS"(Temporizar := wire#w1, Reset := wire#w2, Valor_Tiempo := #V_CNT_ApHsMx_S2, Base_tiempo_ms := 1, Valor_Actual := #TmpAus_S2, Tiempo_OK => #OK_TmpAusS2)
   END_RUNG
   RUNG wire#powerrail
      Contact( #T1_ET60 )
      Contact( #Avance_S2S4 )
      Contact( #MemFN_pHsS2 )
      I_Contact( #pHsMx_S2 )
   END_RUNG wire#w1
   RUNG wire#powerrail
      I_Contact( #T1_ET60 )
   END_RUNG wire#w2
   RUNG wire#powerrail
      Contact( #pHsMx_S2 )
   END_RUNG wire#w2
   // the same network as SCL:
   "FC912_CNT_Tiempo_Mem_UHS"(Temporizar := #T1_ET60 AND #Avance_S2S4 AND #MemFN_pHsS2 AND NOT #pHsMx_S2,
                           Reset := NOT #T1_ET60 OR #pHsMx_S2,
                           Valor_Tiempo := #V_CNT_ApHsMx_S2,
                           Base_tiempo_ms := 1,
                           Valor_Actual := #TmpAus_S2,
                           Tiempo_OK => #OK_TmpAusS2);
END_REGION

REGION Network 27: Temporizacion de las Ausencias S4
   RUNG wire#powerrail
      "FC912_CNT_Tiempo_Mem_UHS"(Temporizar := wire#w1, Reset := wire#w2, Valor_Tiempo := #V_CNT_ApHsMx_S4, Base_tiempo_ms := 1, Valor_Actual := #TmpAus_S4, Tiempo_OK => #OK_TmpAusS4)
   END_RUNG
   RUNG wire#powerrail
      Contact( #T1_ET70 )
      Contact( #Avance_S2S4 )
      Contact( #MemFN_pHsS4 )
      I_Contact( #pHsMx_S4 )
   END_RUNG wire#w1
   RUNG wire#powerrail
      I_Contact( #T1_ET70 )
   END_RUNG wire#w2
   RUNG wire#powerrail
      Contact( #pHsMx_S4 )
   END_RUNG wire#w2
   // the same network as SCL:
   "FC912_CNT_Tiempo_Mem_UHS"(Temporizar := #T1_ET70 AND #Avance_S2S4 AND #MemFN_pHsS4 AND NOT #pHsMx_S4,
                           Reset := NOT #T1_ET70 OR #pHsMx_S4,
                           Valor_Tiempo := #V_CNT_ApHsMx_S4,
                           Base_tiempo_ms := 1,
                           Valor_Actual := #TmpAus_S4,
                           Tiempo_OK => #OK_TmpAusS4);
END_REGION

REGION Network 28: Temporizacion de las Ausencias S3
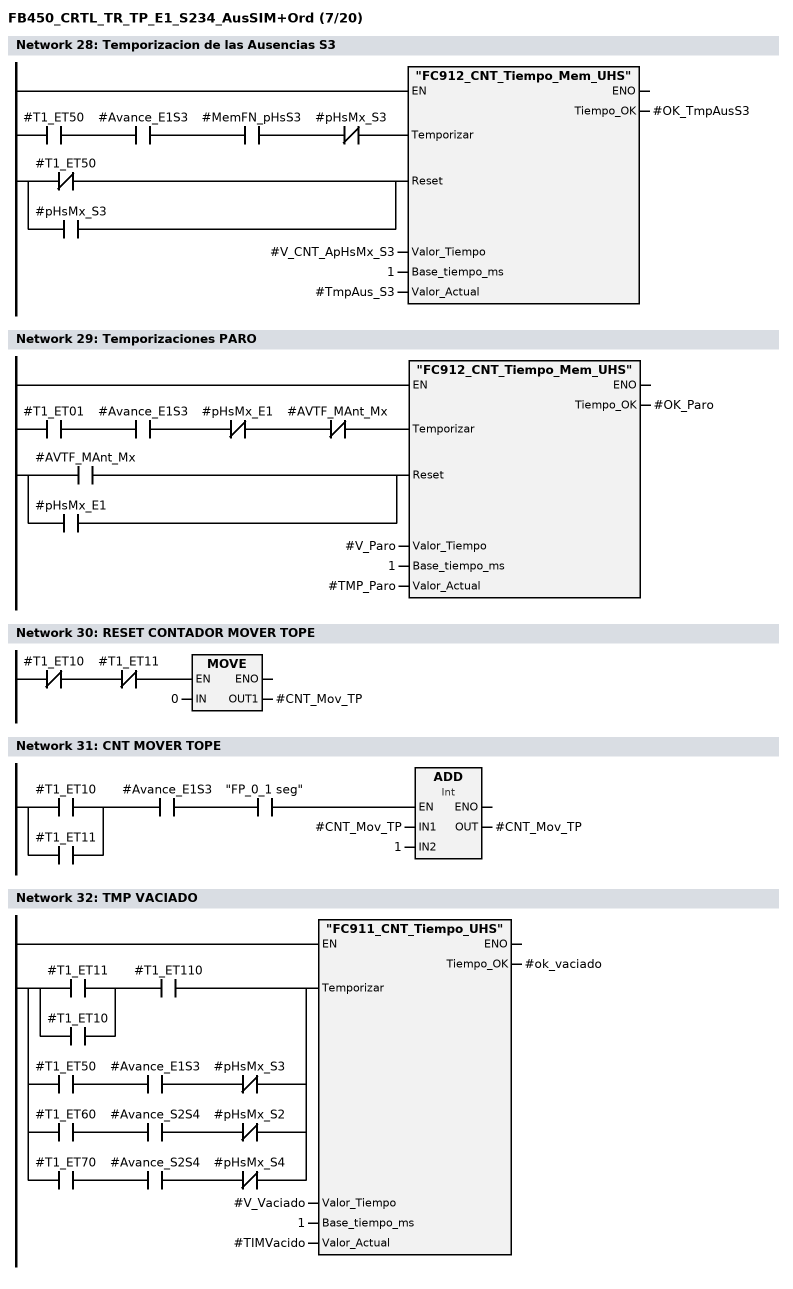
   RUNG wire#powerrail
      "FC912_CNT_Tiempo_Mem_UHS"(Temporizar := wire#w1, Reset := wire#w2, Valor_Tiempo := #V_CNT_ApHsMx_S3, Base_tiempo_ms := 1, Valor_Actual := #TmpAus_S3, Tiempo_OK => #OK_TmpAusS3)
   END_RUNG
   RUNG wire#powerrail
      Contact( #T1_ET50 )
      Contact( #Avance_E1S3 )
      Contact( #MemFN_pHsS3 )
      I_Contact( #pHsMx_S3 )
   END_RUNG wire#w1
   RUNG wire#powerrail
      I_Contact( #T1_ET50 )
   END_RUNG wire#w2
   RUNG wire#powerrail
      Contact( #pHsMx_S3 )
   END_RUNG wire#w2
   // the same network as SCL:
   "FC912_CNT_Tiempo_Mem_UHS"(Temporizar := #T1_ET50 AND #Avance_E1S3 AND #MemFN_pHsS3 AND NOT #pHsMx_S3,
                           Reset := NOT #T1_ET50 OR #pHsMx_S3,
                           Valor_Tiempo := #V_CNT_ApHsMx_S3,
                           Base_tiempo_ms := 1,
                           Valor_Actual := #TmpAus_S3,
                           Tiempo_OK => #OK_TmpAusS3);
END_REGION

REGION Network 29: Temporizaciones PARO
   RUNG wire#powerrail
      "FC912_CNT_Tiempo_Mem_UHS"(Temporizar := wire#w1, Reset := wire#w2, Valor_Tiempo := #V_Paro, Base_tiempo_ms := 1, Valor_Actual := #TMP_Paro, Tiempo_OK => #OK_Paro)
   END_RUNG
   RUNG wire#powerrail
      Contact( #T1_ET01 )
      Contact( #Avance_E1S3 )
      I_Contact( #pHsMx_E1 )
      I_Contact( #AVTF_MAnt_Mx )
   END_RUNG wire#w1
   RUNG wire#powerrail
      Contact( #AVTF_MAnt_Mx )
   END_RUNG wire#w2
   RUNG wire#powerrail
      Contact( #pHsMx_E1 )
   END_RUNG wire#w2
   // the same network as SCL:
   "FC912_CNT_Tiempo_Mem_UHS"(Temporizar := #T1_ET01 AND #Avance_E1S3 AND NOT #pHsMx_E1 AND NOT #AVTF_MAnt_Mx,
                           Reset := #AVTF_MAnt_Mx OR #pHsMx_E1,
                           Valor_Tiempo := #V_Paro,
                           Base_tiempo_ms := 1,
                           Valor_Actual := #TMP_Paro,
                           Tiempo_OK => #OK_Paro);
END_REGION

REGION Network 30: RESET CONTADOR MOVER TOPE
   RUNG wire#powerrail
      I_Contact( #T1_ET10 )
      I_Contact( #T1_ET11 )
      { S7_GenerateENO := "TRUE" } Move(in := 0, out1 => #CNT_Mov_TP)
   END_RUNG
   // the same network as SCL:
   IF NOT #T1_ET10 AND NOT #T1_ET11 THEN #CNT_Mov_TP := 0; END_IF;
END_REGION

REGION Network 31: CNT MOVER TOPE
   RUNG wire#powerrail
      Contact( #T1_ET10 )
      wire#w1
      Contact( #Avance_E1S3 )
      Contact( "FP_0_1 seg" )
      { S7_Templates := "SrcType := Int"; S7_GenerateENO := "TRUE" } Add(in1 := #CNT_Mov_TP, in2 := 1, out => #CNT_Mov_TP)
   END_RUNG
   RUNG wire#powerrail
      Contact( #T1_ET11 )
   END_RUNG wire#w1
   // the same network as SCL:
   IF (#T1_ET10 OR #T1_ET11) AND #Avance_E1S3 AND "FP_0_1 seg" THEN #CNT_Mov_TP := #CNT_Mov_TP + 1; END_IF;
END_REGION

REGION Network 32: TMP VACIADO
   RUNG wire#powerrail
      "FC911_CNT_Tiempo_UHS"(Temporizar := wire#w2, Valor_Tiempo := #V_Vaciado, Base_tiempo_ms := 1, Valor_Actual := #TIMVacido, Tiempo_OK => #ok_vaciado)
   END_RUNG
   RUNG wire#powerrail
      Contact( #T1_ET11 )
      wire#w1
      Contact( #T1_ET110 )
   END_RUNG wire#w2
   RUNG wire#powerrail
      Contact( #T1_ET10 )
   END_RUNG wire#w1
   RUNG wire#powerrail
      Contact( #T1_ET50 )
      Contact( #Avance_E1S3 )
      I_Contact( #pHsMx_S3 )
   END_RUNG wire#w2
   RUNG wire#powerrail
      Contact( #T1_ET60 )
      Contact( #Avance_S2S4 )
      I_Contact( #pHsMx_S2 )
   END_RUNG wire#w2
   RUNG wire#powerrail
      Contact( #T1_ET70 )
      Contact( #Avance_S2S4 )
      I_Contact( #pHsMx_S4 )
   END_RUNG wire#w2
   // the same network as SCL:
   "FC911_CNT_Tiempo_UHS"(Temporizar := ((#T1_ET11 OR #T1_ET10) AND #T1_ET110) OR (#T1_ET50 AND #Avance_E1S3 AND NOT #pHsMx_S3) OR (#T1_ET60 AND #Avance_S2S4 AND NOT #pHsMx_S2) OR (#T1_ET70 AND #Avance_S2S4 AND NOT #pHsMx_S4),
                          Valor_Tiempo := #V_Vaciado,
                          Base_tiempo_ms := 1,
                          Valor_Actual := #TIMVacido,
                          Tiempo_OK => #ok_vaciado);
END_REGION

REGION Network 33: Valores temporizacion para Bloqueo de la Orden
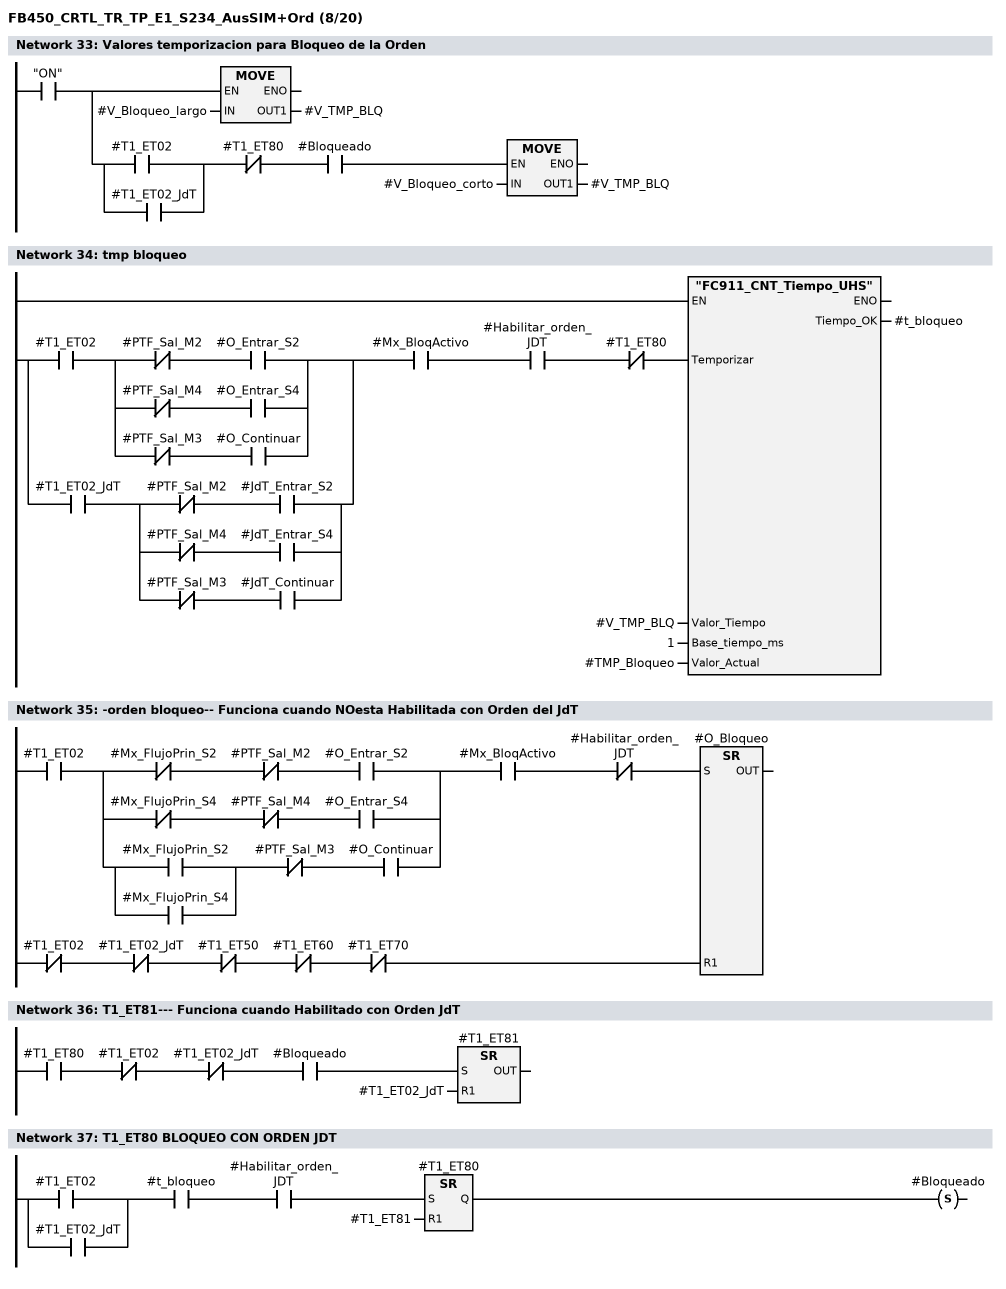
   RUNG wire#powerrail
      Contact( "ON" )
      wire#w1
      { S7_GenerateENO := "TRUE" } Move(in := #V_Bloqueo_largo, out1 => #V_TMP_BLQ)
   END_RUNG
   RUNG wire#w1
      Contact( #T1_ET02 )
      wire#w2
      I_Contact( #T1_ET80 )
      Contact( #Bloqueado )
      { S7_GenerateENO := "TRUE" } Move(in := #V_Bloqueo_corto, out1 => #V_TMP_BLQ)
   END_RUNG
   RUNG wire#w1
      Contact( #T1_ET02_JdT )
   END_RUNG wire#w2
   // the same network as SCL:
   IF "ON" THEN #V_TMP_BLQ := #V_Bloqueo_largo; END_IF;
   IF "ON" AND (#T1_ET02 OR #T1_ET02_JdT) AND NOT #T1_ET80 AND #Bloqueado THEN
       #V_TMP_BLQ := #V_Bloqueo_corto;
   END_IF;
END_REGION

REGION Network 34: tmp bloqueo
   RUNG wire#powerrail
      "FC911_CNT_Tiempo_UHS"(Temporizar := wire#w4, Valor_Tiempo := #V_TMP_BLQ, Base_tiempo_ms := 1, Valor_Actual := #TMP_Bloqueo, Tiempo_OK => #t_bloqueo)
   END_RUNG
   RUNG wire#powerrail
      Contact( #T1_ET02 )
      wire#w1
      I_Contact( #PTF_Sal_M2 )
      Contact( #O_Entrar_S2 )
      wire#w2
      Contact( #Mx_BloqActivo )
      Contact( #Habilitar_orden_JDT )
      I_Contact( #T1_ET80 )
   END_RUNG wire#w4
   RUNG wire#w1
      I_Contact( #PTF_Sal_M4 )
      Contact( #O_Entrar_S4 )
   END_RUNG wire#w2
   RUNG wire#w1
      I_Contact( #PTF_Sal_M3 )
      Contact( #O_Continuar )
   END_RUNG wire#w2
   RUNG wire#powerrail
      Contact( #T1_ET02_JdT )
      wire#w3
      I_Contact( #PTF_Sal_M2 )
      Contact( #JdT_Entrar_S2 )
   END_RUNG wire#w2
   RUNG wire#w3
      I_Contact( #PTF_Sal_M4 )
      Contact( #JdT_Entrar_S4 )
   END_RUNG wire#w2
   RUNG wire#w3
      I_Contact( #PTF_Sal_M3 )
      Contact( #JdT_Continuar )
   END_RUNG wire#w2
   // the same network as SCL:
   "FC911_CNT_Tiempo_UHS"(Temporizar := ((#T1_ET02 AND ((NOT #PTF_Sal_M2 AND #O_Entrar_S2) OR (NOT #PTF_Sal_M4 AND #O_Entrar_S4) OR (NOT #PTF_Sal_M3 AND #O_Continuar))) OR (#T1_ET02_JdT AND ((NOT #PTF_Sal_M2 AND #JdT_Entrar_S2) OR (NOT #PTF_Sal_M4 AND #JdT_Entrar_S4) OR (NOT #PTF_Sal_M3 AND #JdT_Continuar)))) AND #Mx_BloqActivo AND #Habilitar_orden_JDT AND NOT #T1_ET80,
                          Valor_Tiempo := #V_TMP_BLQ,
                          Base_tiempo_ms := 1,
                          Valor_Actual := #TMP_Bloqueo,
                          Tiempo_OK => #t_bloqueo);
END_REGION

REGION Network 35: -orden bloqueo-- Funciona cuando NOesta Habilitada con Orden del JdT
   RUNG wire#powerrail
      Contact( #T1_ET02 )
      wire#w1
      I_Contact( #Mx_FlujoPrin_S2 )
      I_Contact( #PTF_Sal_M2 )
      Contact( #O_Entrar_S2 )
      wire#w2
      Contact( #Mx_BloqActivo )
      I_Contact( #Habilitar_orden_JDT )
      S_SR(operand := #O_Bloqueo, r1 := wire#w4)
   END_RUNG
   RUNG wire#w1
      I_Contact( #Mx_FlujoPrin_S4 )
      I_Contact( #PTF_Sal_M4 )
      Contact( #O_Entrar_S4 )
   END_RUNG wire#w2
   RUNG wire#w1
      Contact( #Mx_FlujoPrin_S2 )
      wire#w3
      I_Contact( #PTF_Sal_M3 )
      Contact( #O_Continuar )
   END_RUNG wire#w2
   RUNG wire#w1
      Contact( #Mx_FlujoPrin_S4 )
   END_RUNG wire#w3
   RUNG wire#powerrail
      I_Contact( #T1_ET02 )
      I_Contact( #T1_ET02_JdT )
      I_Contact( #T1_ET50 )
      I_Contact( #T1_ET60 )
      I_Contact( #T1_ET70 )
   END_RUNG wire#w4
   // the same network as SCL:
   IF #T1_ET02 AND ((NOT #Mx_FlujoPrin_S2 AND NOT #PTF_Sal_M2 AND #O_Entrar_S2) OR (NOT #Mx_FlujoPrin_S4 AND NOT #PTF_Sal_M4 AND #O_Entrar_S4) OR ((#Mx_FlujoPrin_S2 OR #Mx_FlujoPrin_S4) AND NOT #PTF_Sal_M3 AND #O_Continuar)) AND #Mx_BloqActivo AND NOT #Habilitar_orden_JDT THEN
       #O_Bloqueo := TRUE;   // SR flip-flop
   END_IF;
   IF NOT #T1_ET02 AND NOT #T1_ET02_JdT AND NOT #T1_ET50 AND NOT #T1_ET60 AND NOT #T1_ET70 THEN
       #O_Bloqueo := FALSE;
   END_IF;
END_REGION

REGION Network 36: T1_ET81--- Funciona cuando Habilitado con Orden JdT
   RUNG wire#powerrail
      Contact( #T1_ET80 )
      I_Contact( #T1_ET02 )
      I_Contact( #T1_ET02_JdT )
      Contact( #Bloqueado )
      S_SR(operand := #T1_ET81, r1 := #T1_ET02_JdT)
   END_RUNG
   // the same network as SCL:
   IF #T1_ET80 AND NOT #T1_ET02 AND NOT #T1_ET02_JdT AND #Bloqueado THEN
       #T1_ET81 := TRUE;   // SR flip-flop
   END_IF;
   IF #T1_ET02_JdT THEN #T1_ET81 := FALSE; END_IF;
END_REGION

REGION Network 37: T1_ET80 BLOQUEO CON ORDEN JDT
   RUNG wire#powerrail
      Contact( #T1_ET02 )
      wire#w1
      Contact( #t_bloqueo )
      Contact( #Habilitar_orden_JDT )
      S_SR(operand := #T1_ET80, r1 := #T1_ET81)
      S_Coil( #Bloqueado )
   END_RUNG
   RUNG wire#powerrail
      Contact( #T1_ET02_JdT )
   END_RUNG wire#w1
   // the same network as SCL:
   IF (#T1_ET02 OR #T1_ET02_JdT) AND #t_bloqueo AND #Habilitar_orden_JDT THEN
       #T1_ET80 := TRUE;   // SR flip-flop
   END_IF;
   IF #T1_ET81 THEN #T1_ET80 := FALSE; END_IF;
   IF #T1_ET80 THEN #Bloqueado := TRUE; END_IF;
END_REGION

REGION Network 38: GESTION BORRADO ORDENES
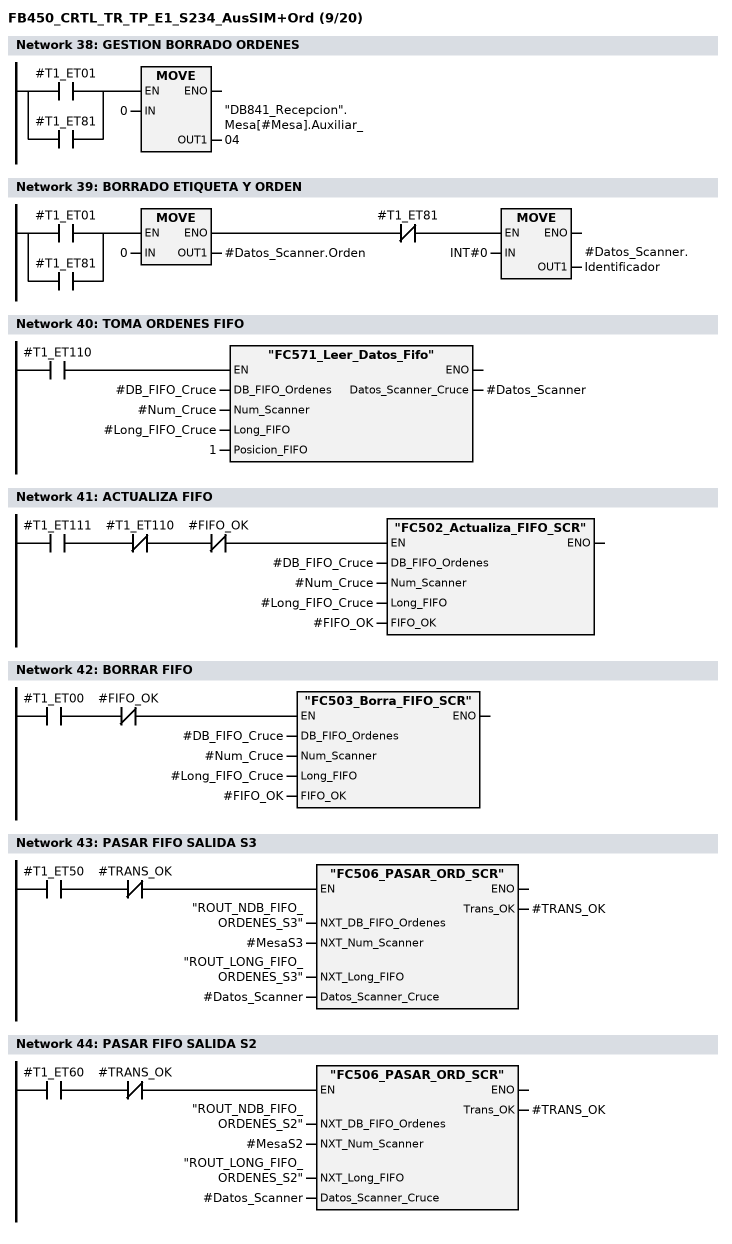
   RUNG wire#powerrail
      Contact( #T1_ET01 )
      wire#w1
      { S7_GenerateENO := "TRUE" } Move(in := 0, out1 => "DB841_Recepcion".Mesa[#Mesa].Auxiliar_04)
   END_RUNG
   RUNG wire#powerrail
      Contact( #T1_ET81 )
   END_RUNG wire#w1
   // the same network as SCL:
   IF #T1_ET01 OR #T1_ET81 THEN "DB841_Recepcion".Mesa[#Mesa].Auxiliar_04 := 0; END_IF;
END_REGION

REGION Network 39: BORRADO ETIQUETA Y ORDEN
   RUNG wire#powerrail
      Contact( #T1_ET01 )
      wire#w1
      { S7_GenerateENO := "TRUE" } Move(in := 0, out1 => #Datos_Scanner.Orden)
      I_Contact( #T1_ET81 )
      { S7_GenerateENO := "TRUE" } Move(in := INT#0, out1 => #Datos_Scanner.Identificador)
   END_RUNG
   RUNG wire#powerrail
      Contact( #T1_ET81 )
   END_RUNG wire#w1
   // the same network as SCL:
   // ENO of a box is taken as its EN; it also drops when the box reports an error
   #_w1 := #T1_ET01 OR #T1_ET81;
   IF #_w1 THEN #Datos_Scanner.Orden := 0; END_IF;
   IF #_w1 AND NOT #T1_ET81 THEN #Datos_Scanner.Identificador := INT#0; END_IF;
END_REGION

REGION Network 40: TOMA ORDENES FIFO
   RUNG wire#powerrail
      Contact( #T1_ET110 )
      "FC571_Leer_Datos_Fifo"(DB_FIFO_Ordenes := #DB_FIFO_Cruce, Num_Scanner := #Num_Cruce, Long_FIFO := #Long_FIFO_Cruce, Posicion_FIFO := 1, Datos_Scanner_Cruce => #Datos_Scanner)
   END_RUNG
   // the same network as SCL:
   IF #T1_ET110 THEN
       "FC571_Leer_Datos_Fifo"(DB_FIFO_Ordenes := #DB_FIFO_Cruce,
                               Num_Scanner := #Num_Cruce,
                               Long_FIFO := #Long_FIFO_Cruce,
                               Posicion_FIFO := 1,
                               Datos_Scanner_Cruce => #Datos_Scanner);
   END_IF;
END_REGION

REGION Network 41: ACTUALIZA FIFO
   RUNG wire#powerrail
      Contact( #T1_ET111 )
      I_Contact( #T1_ET110 )
      I_Contact( #FIFO_OK )
      "FC502_Actualiza_FIFO_SCR"(DB_FIFO_Ordenes := #DB_FIFO_Cruce, Num_Scanner := #Num_Cruce, Long_FIFO := #Long_FIFO_Cruce, FIFO_OK := #FIFO_OK)
   END_RUNG
   // the same network as SCL:
   IF #T1_ET111 AND NOT #T1_ET110 AND NOT #FIFO_OK THEN
       "FC502_Actualiza_FIFO_SCR"(DB_FIFO_Ordenes := #DB_FIFO_Cruce,
                               Num_Scanner := #Num_Cruce,
                               Long_FIFO := #Long_FIFO_Cruce,
                               FIFO_OK := #FIFO_OK);
   END_IF;
END_REGION

REGION Network 42: BORRAR FIFO
   RUNG wire#powerrail
      Contact( #T1_ET00 )
      I_Contact( #FIFO_OK )
      "FC503_Borra_FIFO_SCR"(DB_FIFO_Ordenes := #DB_FIFO_Cruce, Num_Scanner := #Num_Cruce, Long_FIFO := #Long_FIFO_Cruce, FIFO_OK := #FIFO_OK)
   END_RUNG
   // the same network as SCL:
   IF #T1_ET00 AND NOT #FIFO_OK THEN
       "FC503_Borra_FIFO_SCR"(DB_FIFO_Ordenes := #DB_FIFO_Cruce,
                              Num_Scanner := #Num_Cruce,
                              Long_FIFO := #Long_FIFO_Cruce,
                              FIFO_OK := #FIFO_OK);
   END_IF;
END_REGION

REGION Network 43: PASAR FIFO SALIDA S3
   RUNG wire#powerrail
      Contact( #T1_ET50 )
      I_Contact( #TRANS_OK )
      "FC506_PASAR_ORD_SCR"(NXT_DB_FIFO_Ordenes := "ROUT_NDB_FIFO_ORDENES_S3", NXT_Num_Scanner := #MesaS3, NXT_Long_FIFO := "ROUT_LONG_FIFO_ORDENES_S3", Datos_Scanner_Cruce := #Datos_Scanner, Trans_OK => #TRANS_OK)
   END_RUNG
   // the same network as SCL:
   IF #T1_ET50 AND NOT #TRANS_OK THEN
       "FC506_PASAR_ORD_SCR"(NXT_DB_FIFO_Ordenes := "ROUT_NDB_FIFO_ORDENES_S3",
                             NXT_Num_Scanner := #MesaS3,
                             NXT_Long_FIFO := "ROUT_LONG_FIFO_ORDENES_S3",
                             Datos_Scanner_Cruce := #Datos_Scanner,
                             Trans_OK => #TRANS_OK);
   END_IF;
END_REGION

REGION Network 44: PASAR FIFO SALIDA S2
   RUNG wire#powerrail
      Contact( #T1_ET60 )
      I_Contact( #TRANS_OK )
      "FC506_PASAR_ORD_SCR"(NXT_DB_FIFO_Ordenes := "ROUT_NDB_FIFO_ORDENES_S2", NXT_Num_Scanner := #MesaS2, NXT_Long_FIFO := "ROUT_LONG_FIFO_ORDENES_S2", Datos_Scanner_Cruce := #Datos_Scanner, Trans_OK => #TRANS_OK)
   END_RUNG
   // the same network as SCL:
   IF #T1_ET60 AND NOT #TRANS_OK THEN
       "FC506_PASAR_ORD_SCR"(NXT_DB_FIFO_Ordenes := "ROUT_NDB_FIFO_ORDENES_S2",
                             NXT_Num_Scanner := #MesaS2,
                             NXT_Long_FIFO := "ROUT_LONG_FIFO_ORDENES_S2",
                             Datos_Scanner_Cruce := #Datos_Scanner,
                             Trans_OK => #TRANS_OK);
   END_IF;
END_REGION

REGION Network 45: PASAR FIFO SALIDA S4
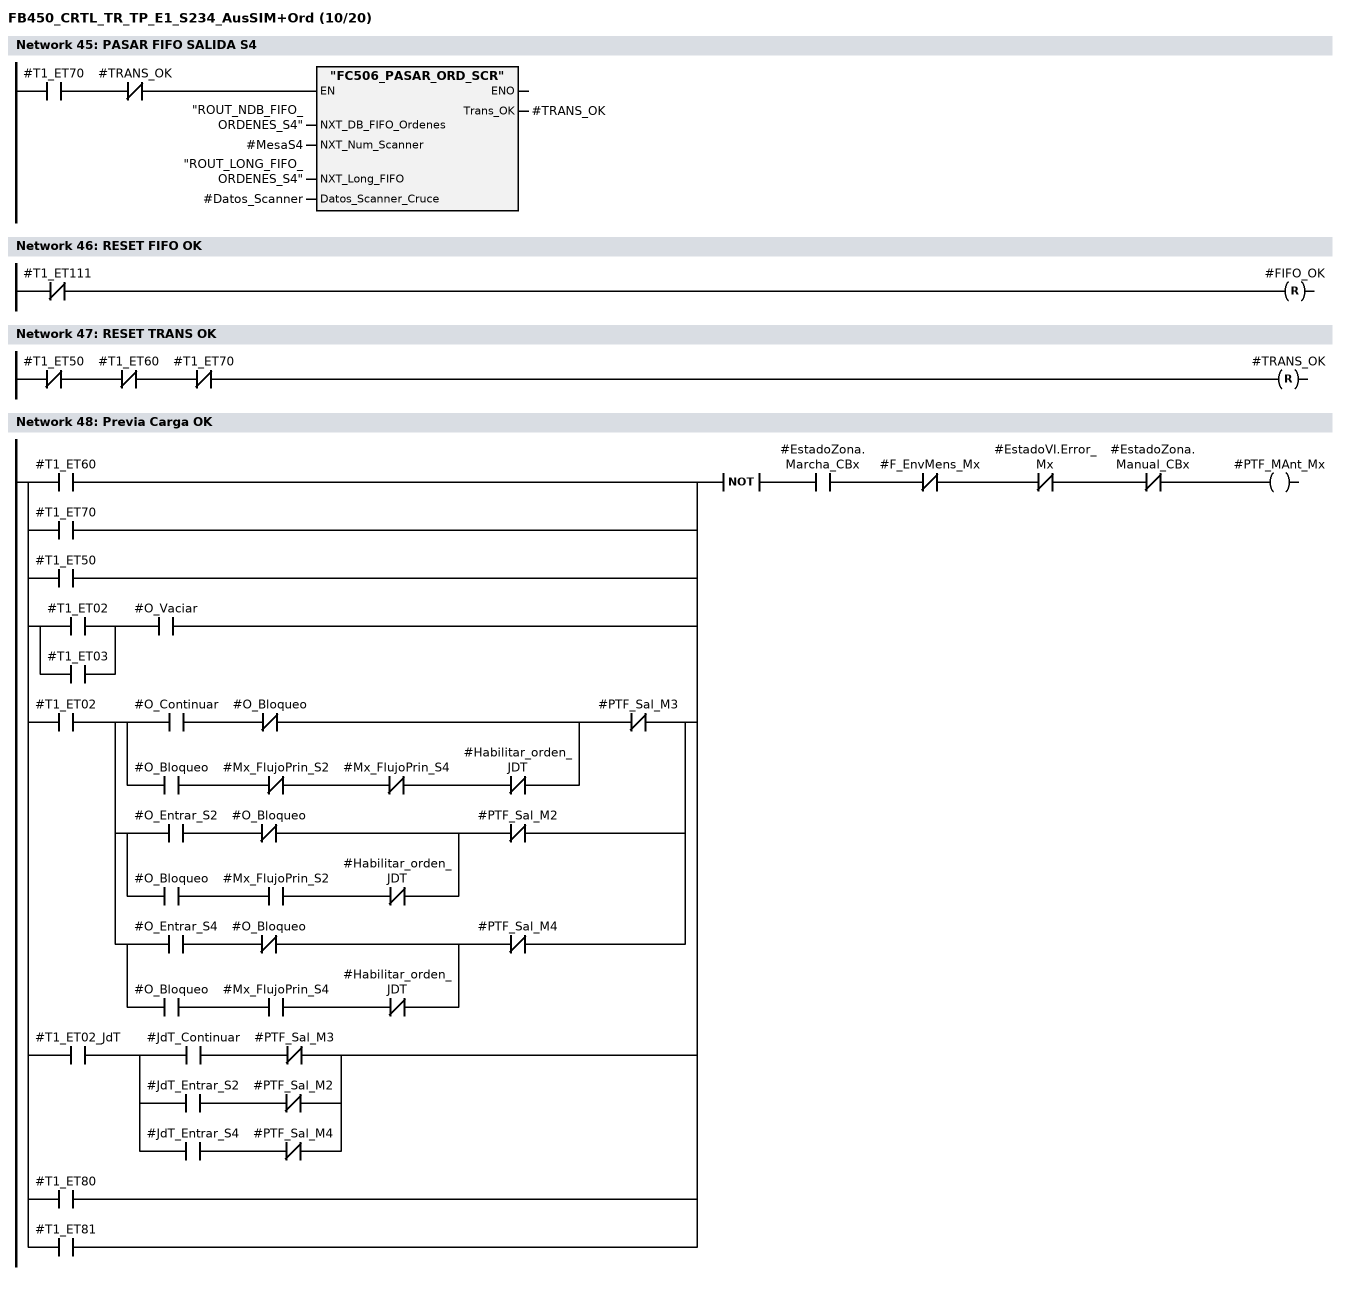
   RUNG wire#powerrail
      Contact( #T1_ET70 )
      I_Contact( #TRANS_OK )
      "FC506_PASAR_ORD_SCR"(NXT_DB_FIFO_Ordenes := "ROUT_NDB_FIFO_ORDENES_S4", NXT_Num_Scanner := #MesaS4, NXT_Long_FIFO := "ROUT_LONG_FIFO_ORDENES_S4", Datos_Scanner_Cruce := #Datos_Scanner, Trans_OK => #TRANS_OK)
   END_RUNG
   // the same network as SCL:
   IF #T1_ET70 AND NOT #TRANS_OK THEN
       "FC506_PASAR_ORD_SCR"(NXT_DB_FIFO_Ordenes := "ROUT_NDB_FIFO_ORDENES_S4",
                             NXT_Num_Scanner := #MesaS4,
                             NXT_Long_FIFO := "ROUT_LONG_FIFO_ORDENES_S4",
                             Datos_Scanner_Cruce := #Datos_Scanner,
                             Trans_OK => #TRANS_OK);
   END_IF;
END_REGION

REGION Network 46: RESET FIFO OK
   RUNG wire#powerrail
      I_Contact( #T1_ET111 )
      R_Coil( #FIFO_OK )
   END_RUNG
   // the same network as SCL:
   IF NOT #T1_ET111 THEN #FIFO_OK := FALSE; END_IF;
END_REGION

REGION Network 47: RESET TRANS OK
   RUNG wire#powerrail
      I_Contact( #T1_ET50 )
      I_Contact( #T1_ET60 )
      I_Contact( #T1_ET70 )
      R_Coil( #TRANS_OK )
   END_RUNG
   // the same network as SCL:
   IF NOT #T1_ET50 AND NOT #T1_ET60 AND NOT #T1_ET70 THEN #TRANS_OK := FALSE; END_IF;
END_REGION

REGION Network 48: Previa Carga OK
   RUNG wire#powerrail
      Contact( #T1_ET60 )
      wire#w1
      Not()
      Contact( #EstadoZona.Marcha_CBx )
      I_Contact( #F_EnvMens_Mx )
      I_Contact( #EstadoVI.Error_Mx )
      I_Contact( #EstadoZona.Manual_CBx )
      Coil( #PTF_MAnt_Mx )
   END_RUNG
   RUNG wire#powerrail
      Contact( #T1_ET70 )
   END_RUNG wire#w1
   RUNG wire#powerrail
      Contact( #T1_ET50 )
   END_RUNG wire#w1
   RUNG wire#powerrail
      Contact( #T1_ET02 )
      wire#w2
      Contact( #O_Vaciar )
   END_RUNG wire#w1
   RUNG wire#powerrail
      Contact( #T1_ET03 )
   END_RUNG wire#w2
   RUNG wire#powerrail
      Contact( #T1_ET02 )
      wire#w3
      Contact( #O_Continuar )
      I_Contact( #O_Bloqueo )
      wire#w4
      I_Contact( #PTF_Sal_M3 )
   END_RUNG wire#w1
   RUNG wire#w3
      Contact( #O_Bloqueo )
      I_Contact( #Mx_FlujoPrin_S2 )
      I_Contact( #Mx_FlujoPrin_S4 )
      I_Contact( #Habilitar_orden_JDT )
   END_RUNG wire#w4
   RUNG wire#w3
      Contact( #O_Entrar_S2 )
      I_Contact( #O_Bloqueo )
      wire#w5
      I_Contact( #PTF_Sal_M2 )
   END_RUNG wire#w1
   RUNG wire#w3
      Contact( #O_Bloqueo )
      Contact( #Mx_FlujoPrin_S2 )
      I_Contact( #Habilitar_orden_JDT )
   END_RUNG wire#w5
   RUNG wire#w3
      Contact( #O_Entrar_S4 )
      I_Contact( #O_Bloqueo )
      wire#w6
      I_Contact( #PTF_Sal_M4 )
   END_RUNG wire#w1
   RUNG wire#w3
      Contact( #O_Bloqueo )
      Contact( #Mx_FlujoPrin_S4 )
      I_Contact( #Habilitar_orden_JDT )
   END_RUNG wire#w6
   RUNG wire#powerrail
      Contact( #T1_ET02_JdT )
      wire#w7
      Contact( #JdT_Continuar )
      I_Contact( #PTF_Sal_M3 )
   END_RUNG wire#w1
   RUNG wire#w7
      Contact( #JdT_Entrar_S2 )
      I_Contact( #PTF_Sal_M2 )
   END_RUNG wire#w1
   RUNG wire#w7
      Contact( #JdT_Entrar_S4 )
      I_Contact( #PTF_Sal_M4 )
   END_RUNG wire#w1
   RUNG wire#powerrail
      Contact( #T1_ET80 )
   END_RUNG wire#w1
   RUNG wire#powerrail
      Contact( #T1_ET81 )
   END_RUNG wire#w1
   // the same network as SCL:
   #PTF_MAnt_Mx := NOT (#T1_ET60 OR #T1_ET70 OR #T1_ET50 OR ((#T1_ET02 OR #T1_ET03) AND #O_Vaciar) OR (#T1_ET02 AND ((((#O_Continuar AND NOT #O_Bloqueo) OR (#O_Bloqueo AND NOT #Mx_FlujoPrin_S2 AND NOT #Mx_FlujoPrin_S4 AND NOT #Habilitar_orden_JDT)) AND NOT #PTF_Sal_M3) OR (((#O_Entrar_S2 AND NOT #O_Bloqueo) OR (#O_Bloqueo AND #Mx_FlujoPrin_S2 AND NOT #Habilitar_orden_JDT)) AND NOT #PTF_Sal_M2) OR (((#O_Entrar_S4 AND NOT #O_Bloqueo) OR (#O_Bloqueo AND #Mx_FlujoPrin_S4 AND NOT #Habilitar_orden_JDT)) AND NOT #PTF_Sal_M4))) OR (#T1_ET02_JdT AND ((#JdT_Continuar AND NOT #PTF_Sal_M3) OR (#JdT_Entrar_S2 AND NOT #PTF_Sal_M2) OR (#JdT_Entrar_S4 AND NOT #PTF_Sal_M4))) OR #T1_ET80 OR #T1_ET81) AND #EstadoZona.Marcha_CBx AND NOT #F_EnvMens_Mx AND NOT #EstadoVI.Error_Mx AND NOT #EstadoZona.Manual_CBx;
END_REGION

REGION Network 49: NXT AVTF S3
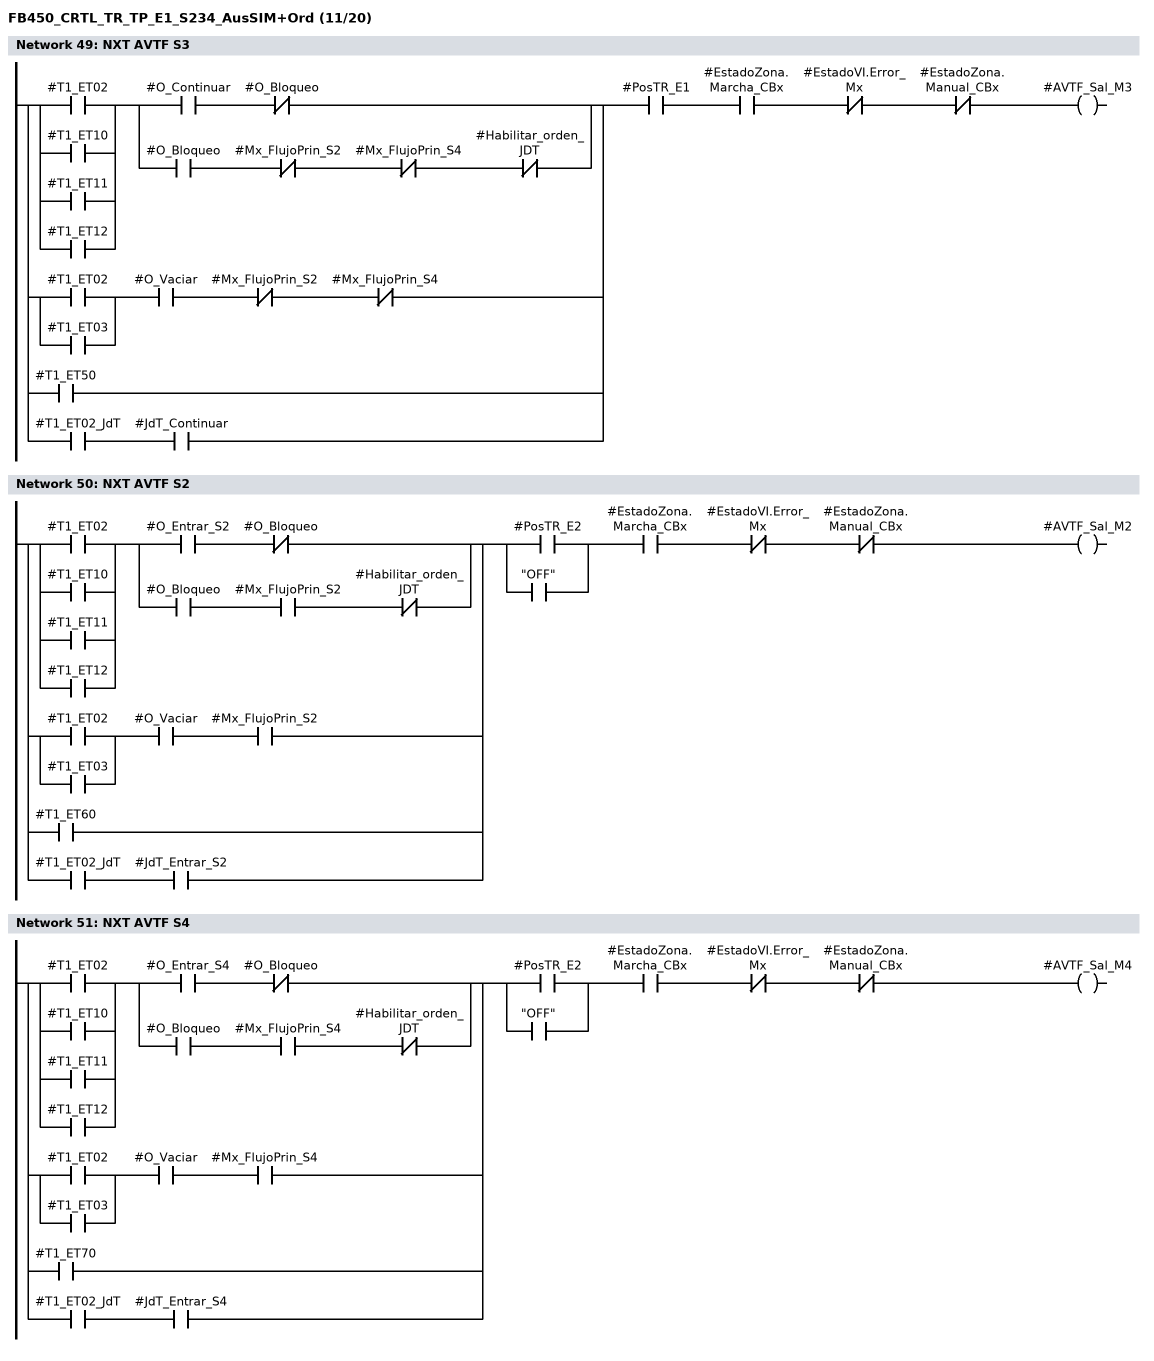
   RUNG wire#powerrail
      Contact( #T1_ET02 )
      wire#w1
      Contact( #O_Continuar )
      I_Contact( #O_Bloqueo )
      wire#w2
      Contact( #PosTR_E1 )
      Contact( #EstadoZona.Marcha_CBx )
      I_Contact( #EstadoVI.Error_Mx )
      I_Contact( #EstadoZona.Manual_CBx )
      Coil( #AVTF_Sal_M3 )
   END_RUNG
   RUNG wire#powerrail
      Contact( #T1_ET10 )
   END_RUNG wire#w1
   RUNG wire#powerrail
      Contact( #T1_ET11 )
   END_RUNG wire#w1
   RUNG wire#powerrail
      Contact( #T1_ET12 )
   END_RUNG wire#w1
   RUNG wire#w1
      Contact( #O_Bloqueo )
      I_Contact( #Mx_FlujoPrin_S2 )
      I_Contact( #Mx_FlujoPrin_S4 )
      I_Contact( #Habilitar_orden_JDT )
   END_RUNG wire#w2
   RUNG wire#powerrail
      Contact( #T1_ET02 )
      wire#w3
      Contact( #O_Vaciar )
      I_Contact( #Mx_FlujoPrin_S2 )
      I_Contact( #Mx_FlujoPrin_S4 )
   END_RUNG wire#w2
   RUNG wire#powerrail
      Contact( #T1_ET03 )
   END_RUNG wire#w3
   RUNG wire#powerrail
      Contact( #T1_ET50 )
   END_RUNG wire#w2
   RUNG wire#powerrail
      Contact( #T1_ET02_JdT )
      Contact( #JdT_Continuar )
   END_RUNG wire#w2
   // the same network as SCL:
   #AVTF_Sal_M3 := (((#T1_ET02 OR #T1_ET10 OR #T1_ET11 OR #T1_ET12) AND ((#O_Continuar AND NOT #O_Bloqueo) OR (#O_Bloqueo AND NOT #Mx_FlujoPrin_S2 AND NOT #Mx_FlujoPrin_S4 AND NOT #Habilitar_orden_JDT))) OR ((#T1_ET02 OR #T1_ET03) AND #O_Vaciar AND NOT #Mx_FlujoPrin_S2 AND NOT #Mx_FlujoPrin_S4) OR #T1_ET50 OR (#T1_ET02_JdT AND #JdT_Continuar)) AND #PosTR_E1 AND #EstadoZona.Marcha_CBx AND NOT #EstadoVI.Error_Mx AND NOT #EstadoZona.Manual_CBx;
END_REGION

REGION Network 50: NXT AVTF S2
   RUNG wire#powerrail
      Contact( #T1_ET02 )
      wire#w1
      Contact( #O_Entrar_S2 )
      I_Contact( #O_Bloqueo )
      wire#w2
      Contact( #PosTR_E2 )
      wire#w4
      Contact( #EstadoZona.Marcha_CBx )
      I_Contact( #EstadoVI.Error_Mx )
      I_Contact( #EstadoZona.Manual_CBx )
      Coil( #AVTF_Sal_M2 )
   END_RUNG
   RUNG wire#powerrail
      Contact( #T1_ET10 )
   END_RUNG wire#w1
   RUNG wire#powerrail
      Contact( #T1_ET11 )
   END_RUNG wire#w1
   RUNG wire#powerrail
      Contact( #T1_ET12 )
   END_RUNG wire#w1
   RUNG wire#w1
      Contact( #O_Bloqueo )
      Contact( #Mx_FlujoPrin_S2 )
      I_Contact( #Habilitar_orden_JDT )
   END_RUNG wire#w2
   RUNG wire#powerrail
      Contact( #T1_ET02 )
      wire#w3
      Contact( #O_Vaciar )
      Contact( #Mx_FlujoPrin_S2 )
   END_RUNG wire#w2
   RUNG wire#powerrail
      Contact( #T1_ET03 )
   END_RUNG wire#w3
   RUNG wire#powerrail
      Contact( #T1_ET60 )
   END_RUNG wire#w2
   RUNG wire#powerrail
      Contact( #T1_ET02_JdT )
      Contact( #JdT_Entrar_S2 )
   END_RUNG wire#w2
   RUNG wire#w2
      Contact( "OFF" )
   END_RUNG wire#w4
   // the same network as SCL:
   #AVTF_Sal_M2 := (((#T1_ET02 OR #T1_ET10 OR #T1_ET11 OR #T1_ET12) AND ((#O_Entrar_S2 AND NOT #O_Bloqueo) OR (#O_Bloqueo AND #Mx_FlujoPrin_S2 AND NOT #Habilitar_orden_JDT))) OR ((#T1_ET02 OR #T1_ET03) AND #O_Vaciar AND #Mx_FlujoPrin_S2) OR #T1_ET60 OR (#T1_ET02_JdT AND #JdT_Entrar_S2)) AND (#PosTR_E2 OR "OFF") AND #EstadoZona.Marcha_CBx AND NOT #EstadoVI.Error_Mx AND NOT #EstadoZona.Manual_CBx;
END_REGION

REGION Network 51: NXT AVTF S4
   RUNG wire#powerrail
      Contact( #T1_ET02 )
      wire#w1
      Contact( #O_Entrar_S4 )
      I_Contact( #O_Bloqueo )
      wire#w2
      Contact( #PosTR_E2 )
      wire#w4
      Contact( #EstadoZona.Marcha_CBx )
      I_Contact( #EstadoVI.Error_Mx )
      I_Contact( #EstadoZona.Manual_CBx )
      Coil( #AVTF_Sal_M4 )
   END_RUNG
   RUNG wire#powerrail
      Contact( #T1_ET10 )
   END_RUNG wire#w1
   RUNG wire#powerrail
      Contact( #T1_ET11 )
   END_RUNG wire#w1
   RUNG wire#powerrail
      Contact( #T1_ET12 )
   END_RUNG wire#w1
   RUNG wire#w1
      Contact( #O_Bloqueo )
      Contact( #Mx_FlujoPrin_S4 )
      I_Contact( #Habilitar_orden_JDT )
   END_RUNG wire#w2
   RUNG wire#powerrail
      Contact( #T1_ET02 )
      wire#w3
      Contact( #O_Vaciar )
      Contact( #Mx_FlujoPrin_S4 )
   END_RUNG wire#w2
   RUNG wire#powerrail
      Contact( #T1_ET03 )
   END_RUNG wire#w3
   RUNG wire#powerrail
      Contact( #T1_ET70 )
   END_RUNG wire#w2
   RUNG wire#powerrail
      Contact( #T1_ET02_JdT )
      Contact( #JdT_Entrar_S4 )
   END_RUNG wire#w2
   RUNG wire#w2
      Contact( "OFF" )
   END_RUNG wire#w4
   // the same network as SCL:
   #AVTF_Sal_M4 := (((#T1_ET02 OR #T1_ET10 OR #T1_ET11 OR #T1_ET12) AND ((#O_Entrar_S4 AND NOT #O_Bloqueo) OR (#O_Bloqueo AND #Mx_FlujoPrin_S4 AND NOT #Habilitar_orden_JDT))) OR ((#T1_ET02 OR #T1_ET03) AND #O_Vaciar AND #Mx_FlujoPrin_S4) OR #T1_ET70 OR (#T1_ET02_JdT AND #JdT_Entrar_S4)) AND (#PosTR_E2 OR "OFF") AND #EstadoZona.Marcha_CBx AND NOT #EstadoVI.Error_Mx AND NOT #EstadoZona.Manual_CBx;
END_REGION

REGION Network 52: TMP Movimientos del Transfer --> Subida y Bajada
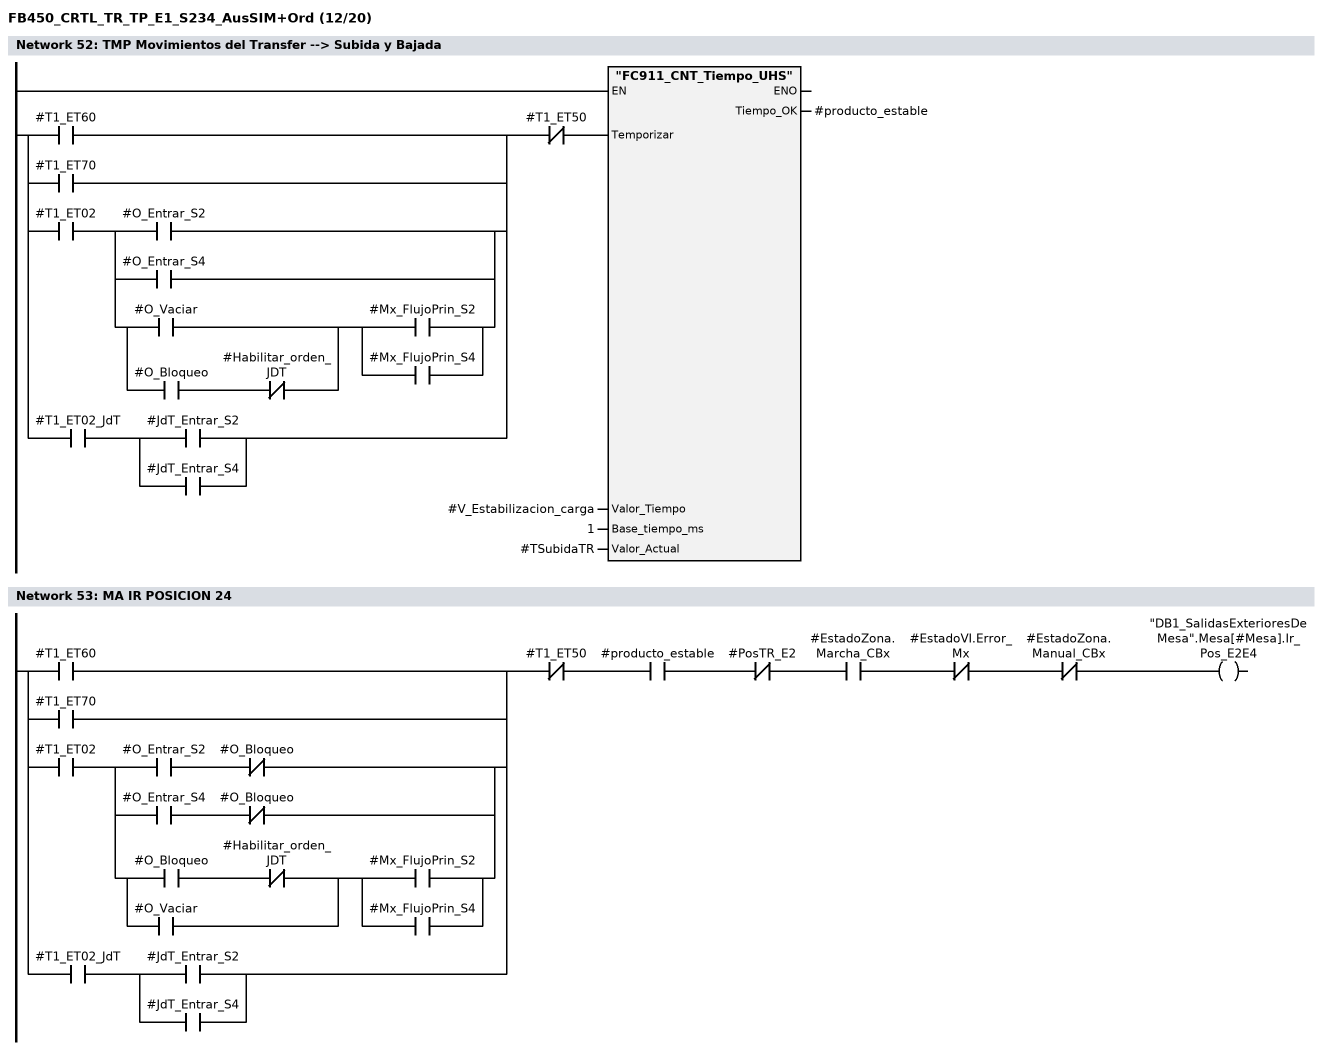
   RUNG wire#powerrail
      "FC911_CNT_Tiempo_UHS"(Temporizar := wire#w5, Valor_Tiempo := #V_Estabilizacion_carga, Base_tiempo_ms := 1, Valor_Actual := #TSubidaTR, Tiempo_OK => #producto_estable)
   END_RUNG
   RUNG wire#powerrail
      Contact( #T1_ET60 )
      wire#w1
      I_Contact( #T1_ET50 )
   END_RUNG wire#w5
   RUNG wire#powerrail
      Contact( #T1_ET70 )
   END_RUNG wire#w1
   RUNG wire#powerrail
      Contact( #T1_ET02 )
      wire#w2
      Contact( #O_Entrar_S2 )
   END_RUNG wire#w1
   RUNG wire#w2
      Contact( #O_Entrar_S4 )
   END_RUNG wire#w1
   RUNG wire#w2
      Contact( #O_Vaciar )
      wire#w3
      Contact( #Mx_FlujoPrin_S2 )
   END_RUNG wire#w1
   RUNG wire#w2
      Contact( #O_Bloqueo )
      I_Contact( #Habilitar_orden_JDT )
   END_RUNG wire#w3
   RUNG wire#w3
      Contact( #Mx_FlujoPrin_S4 )
   END_RUNG wire#w1
   RUNG wire#powerrail
      Contact( #T1_ET02_JdT )
      wire#w4
      Contact( #JdT_Entrar_S2 )
   END_RUNG wire#w1
   RUNG wire#w4
      Contact( #JdT_Entrar_S4 )
   END_RUNG wire#w1
   // the same network as SCL:
   "FC911_CNT_Tiempo_UHS"(Temporizar := (#T1_ET60 OR #T1_ET70 OR (#T1_ET02 AND (#O_Entrar_S2 OR #O_Entrar_S4 OR ((#O_Vaciar OR (#O_Bloqueo AND NOT #Habilitar_orden_JDT)) AND (#Mx_FlujoPrin_S2 OR #Mx_FlujoPrin_S4)))) OR (#T1_ET02_JdT AND (#JdT_Entrar_S2 OR #JdT_Entrar_S4))) AND NOT #T1_ET50,
                          Valor_Tiempo := #V_Estabilizacion_carga,
                          Base_tiempo_ms := 1,
                          Valor_Actual := #TSubidaTR,
                          Tiempo_OK => #producto_estable);
END_REGION

REGION Network 53: MA IR POSICION 24
   RUNG wire#powerrail
      Contact( #T1_ET60 )
      wire#w1
      I_Contact( #T1_ET50 )
      Contact( #producto_estable )
      I_Contact( #PosTR_E2 )
      Contact( #EstadoZona.Marcha_CBx )
      I_Contact( #EstadoVI.Error_Mx )
      I_Contact( #EstadoZona.Manual_CBx )
      Coil( "DB1_SalidasExterioresDeMesa".Mesa[#Mesa].Ir_Pos_E2E4 )
   END_RUNG
   RUNG wire#powerrail
      Contact( #T1_ET70 )
   END_RUNG wire#w1
   RUNG wire#powerrail
      Contact( #T1_ET02 )
      wire#w2
      Contact( #O_Entrar_S2 )
      I_Contact( #O_Bloqueo )
   END_RUNG wire#w1
   RUNG wire#w2
      Contact( #O_Entrar_S4 )
      I_Contact( #O_Bloqueo )
   END_RUNG wire#w1
   RUNG wire#w2
      Contact( #O_Bloqueo )
      I_Contact( #Habilitar_orden_JDT )
      wire#w3
      Contact( #Mx_FlujoPrin_S2 )
   END_RUNG wire#w1
   RUNG wire#w2
      Contact( #O_Vaciar )
   END_RUNG wire#w3
   RUNG wire#w3
      Contact( #Mx_FlujoPrin_S4 )
   END_RUNG wire#w1
   RUNG wire#powerrail
      Contact( #T1_ET02_JdT )
      wire#w4
      Contact( #JdT_Entrar_S2 )
   END_RUNG wire#w1
   RUNG wire#w4
      Contact( #JdT_Entrar_S4 )
   END_RUNG wire#w1
   // the same network as SCL:
   "DB1_SalidasExterioresDeMesa".Mesa[#Mesa].Ir_Pos_E2E4 := (#T1_ET60 OR #T1_ET70 OR (#T1_ET02 AND ((#O_Entrar_S2 AND NOT #O_Bloqueo) OR (#O_Entrar_S4 AND NOT #O_Bloqueo) OR (((#O_Bloqueo AND NOT #Habilitar_orden_JDT) OR #O_Vaciar) AND (#Mx_FlujoPrin_S2 OR #Mx_FlujoPrin_S4)))) OR (#T1_ET02_JdT AND (#JdT_Entrar_S2 OR #JdT_Entrar_S4))) AND NOT #T1_ET50 AND #producto_estable AND NOT #PosTR_E2 AND #EstadoZona.Marcha_CBx AND NOT #EstadoVI.Error_Mx AND NOT #EstadoZona.Manual_CBx;
END_REGION

REGION Network 54: MA IR POSICION 13
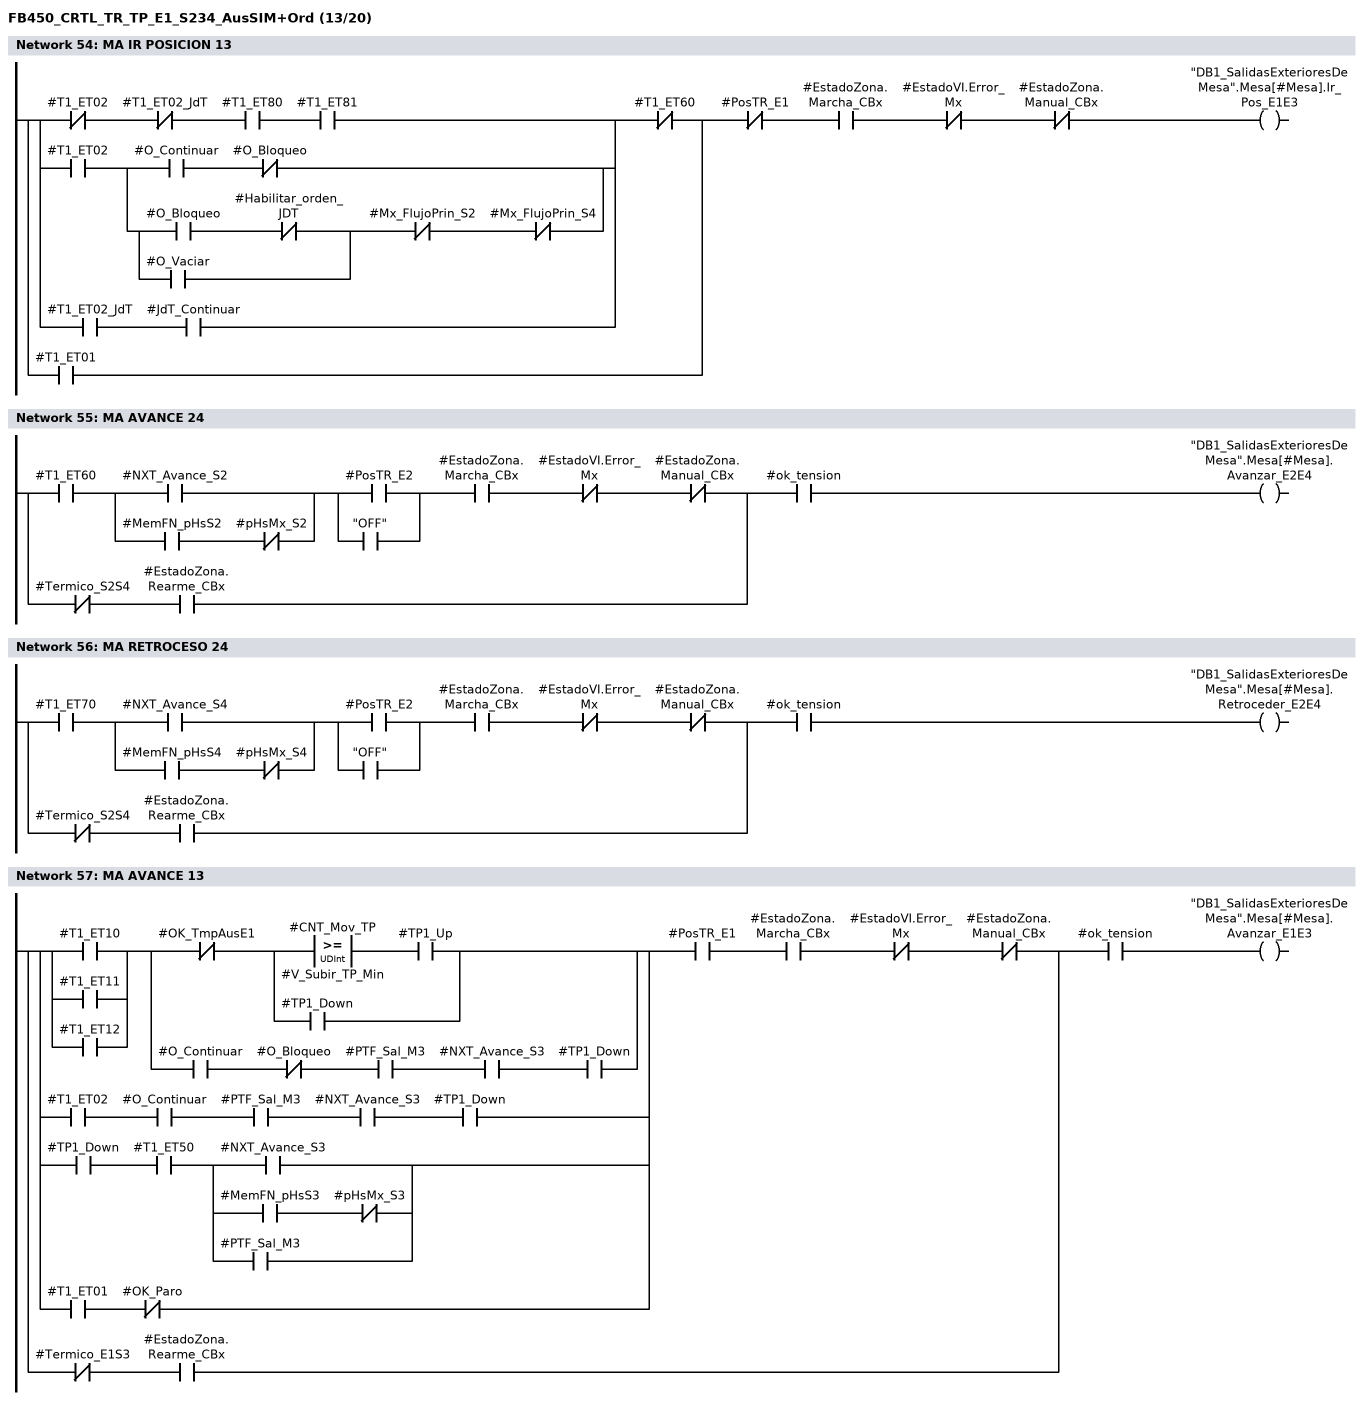
   RUNG wire#powerrail
      I_Contact( #T1_ET02 )
      I_Contact( #T1_ET02_JdT )
      Contact( #T1_ET80 )
      Contact( #T1_ET81 )
      wire#w1
      I_Contact( #T1_ET60 )
      wire#w4
      I_Contact( #PosTR_E1 )
      Contact( #EstadoZona.Marcha_CBx )
      I_Contact( #EstadoVI.Error_Mx )
      I_Contact( #EstadoZona.Manual_CBx )
      Coil( "DB1_SalidasExterioresDeMesa".Mesa[#Mesa].Ir_Pos_E1E3 )
   END_RUNG
   RUNG wire#powerrail
      Contact( #T1_ET02 )
      wire#w2
      Contact( #O_Continuar )
      I_Contact( #O_Bloqueo )
   END_RUNG wire#w1
   RUNG wire#w2
      Contact( #O_Bloqueo )
      I_Contact( #Habilitar_orden_JDT )
      wire#w3
      I_Contact( #Mx_FlujoPrin_S2 )
      I_Contact( #Mx_FlujoPrin_S4 )
   END_RUNG wire#w1
   RUNG wire#w2
      Contact( #O_Vaciar )
   END_RUNG wire#w3
   RUNG wire#powerrail
      Contact( #T1_ET02_JdT )
      Contact( #JdT_Continuar )
   END_RUNG wire#w1
   RUNG wire#powerrail
      Contact( #T1_ET01 )
   END_RUNG wire#w4
   // the same network as SCL:
   "DB1_SalidasExterioresDeMesa".Mesa[#Mesa].Ir_Pos_E1E3 := ((((NOT #T1_ET02 AND NOT #T1_ET02_JdT AND #T1_ET80 AND #T1_ET81) OR (#T1_ET02 AND ((#O_Continuar AND NOT #O_Bloqueo) OR (((#O_Bloqueo AND NOT #Habilitar_orden_JDT) OR #O_Vaciar) AND NOT #Mx_FlujoPrin_S2 AND NOT #Mx_FlujoPrin_S4))) OR (#T1_ET02_JdT AND #JdT_Continuar)) AND NOT #T1_ET60) OR #T1_ET01) AND NOT #PosTR_E1 AND #EstadoZona.Marcha_CBx AND NOT #EstadoVI.Error_Mx AND NOT #EstadoZona.Manual_CBx;
END_REGION

REGION Network 55: MA AVANCE 24
   RUNG wire#powerrail
      Contact( #T1_ET60 )
      wire#w1
      Contact( #NXT_Avance_S2 )
      wire#w2
      Contact( #PosTR_E2 )
      wire#w3
      Contact( #EstadoZona.Marcha_CBx )
      I_Contact( #EstadoVI.Error_Mx )
      I_Contact( #EstadoZona.Manual_CBx )
      wire#w4
      Contact( #ok_tension )
      Coil( "DB1_SalidasExterioresDeMesa".Mesa[#Mesa].Avanzar_E2E4 )
   END_RUNG
   RUNG wire#w1
      Contact( #MemFN_pHsS2 )
      I_Contact( #pHsMx_S2 )
   END_RUNG wire#w2
   RUNG wire#w2
      Contact( "OFF" )
   END_RUNG wire#w3
   RUNG wire#powerrail
      I_Contact( #Termico_S2S4 )
      Contact( #EstadoZona.Rearme_CBx )
   END_RUNG wire#w4
   // the same network as SCL:
   "DB1_SalidasExterioresDeMesa".Mesa[#Mesa].Avanzar_E2E4 := ((#T1_ET60 AND (#NXT_Avance_S2 OR (#MemFN_pHsS2 AND NOT #pHsMx_S2)) AND (#PosTR_E2 OR "OFF") AND #EstadoZona.Marcha_CBx AND NOT #EstadoVI.Error_Mx AND NOT #EstadoZona.Manual_CBx) OR (NOT #Termico_S2S4 AND #EstadoZona.Rearme_CBx)) AND #ok_tension;
END_REGION

REGION Network 56: MA RETROCESO 24
   RUNG wire#powerrail
      Contact( #T1_ET70 )
      wire#w1
      Contact( #NXT_Avance_S4 )
      wire#w2
      Contact( #PosTR_E2 )
      wire#w3
      Contact( #EstadoZona.Marcha_CBx )
      I_Contact( #EstadoVI.Error_Mx )
      I_Contact( #EstadoZona.Manual_CBx )
      wire#w4
      Contact( #ok_tension )
      Coil( "DB1_SalidasExterioresDeMesa".Mesa[#Mesa].Retroceder_E2E4 )
   END_RUNG
   RUNG wire#w1
      Contact( #MemFN_pHsS4 )
      I_Contact( #pHsMx_S4 )
   END_RUNG wire#w2
   RUNG wire#w2
      Contact( "OFF" )
   END_RUNG wire#w3
   RUNG wire#powerrail
      I_Contact( #Termico_S2S4 )
      Contact( #EstadoZona.Rearme_CBx )
   END_RUNG wire#w4
   // the same network as SCL:
   "DB1_SalidasExterioresDeMesa".Mesa[#Mesa].Retroceder_E2E4 := ((#T1_ET70 AND (#NXT_Avance_S4 OR (#MemFN_pHsS4 AND NOT #pHsMx_S4)) AND (#PosTR_E2 OR "OFF") AND #EstadoZona.Marcha_CBx AND NOT #EstadoVI.Error_Mx AND NOT #EstadoZona.Manual_CBx) OR (NOT #Termico_S2S4 AND #EstadoZona.Rearme_CBx)) AND #ok_tension;
END_REGION

REGION Network 57: MA AVANCE 13
   RUNG wire#powerrail
      Contact( #T1_ET10 )
      wire#w1
      I_Contact( #OK_TmpAusE1 )
      wire#w2
      { S7_Templates := "SrcType := UDInt" } GE_Contact(in1 := #CNT_Mov_TP, in2 := #V_Subir_TP_Min)
      Contact( #TP1_Up )
      wire#w3
      Contact( #PosTR_E1 )
      Contact( #EstadoZona.Marcha_CBx )
      I_Contact( #EstadoVI.Error_Mx )
      I_Contact( #EstadoZona.Manual_CBx )
      wire#w5
      Contact( #ok_tension )
      Coil( "DB1_SalidasExterioresDeMesa".Mesa[#Mesa].Avanzar_E1E3 )
   END_RUNG
   RUNG wire#powerrail
      Contact( #T1_ET11 )
   END_RUNG wire#w1
   RUNG wire#powerrail
      Contact( #T1_ET12 )
   END_RUNG wire#w1
   RUNG wire#w2
      Contact( #TP1_Down )
   END_RUNG wire#w3
   RUNG wire#w1
      Contact( #O_Continuar )
      I_Contact( #O_Bloqueo )
      Contact( #PTF_Sal_M3 )
      Contact( #NXT_Avance_S3 )
      Contact( #TP1_Down )
   END_RUNG wire#w3
   RUNG wire#powerrail
      Contact( #T1_ET02 )
      Contact( #O_Continuar )
      Contact( #PTF_Sal_M3 )
      Contact( #NXT_Avance_S3 )
      Contact( #TP1_Down )
   END_RUNG wire#w3
   RUNG wire#powerrail
      Contact( #TP1_Down )
      Contact( #T1_ET50 )
      wire#w4
      Contact( #NXT_Avance_S3 )
   END_RUNG wire#w3
   RUNG wire#w4
      Contact( #MemFN_pHsS3 )
      I_Contact( #pHsMx_S3 )
   END_RUNG wire#w3
   RUNG wire#w4
      Contact( #PTF_Sal_M3 )
   END_RUNG wire#w3
   RUNG wire#powerrail
      Contact( #T1_ET01 )
      I_Contact( #OK_Paro )
   END_RUNG wire#w3
   RUNG wire#powerrail
      I_Contact( #Termico_E1S3 )
      Contact( #EstadoZona.Rearme_CBx )
   END_RUNG wire#w5
   // the same network as SCL:
   "DB1_SalidasExterioresDeMesa".Mesa[#Mesa].Avanzar_E1E3 := (((((#T1_ET10 OR #T1_ET11 OR #T1_ET12) AND ((NOT #OK_TmpAusE1 AND (((#CNT_Mov_TP >= #V_Subir_TP_Min) AND #TP1_Up) OR #TP1_Down)) OR (#O_Continuar AND NOT #O_Bloqueo AND #PTF_Sal_M3 AND #NXT_Avance_S3 AND #TP1_Down))) OR (#T1_ET02 AND #O_Continuar AND #PTF_Sal_M3 AND #NXT_Avance_S3 AND #TP1_Down) OR (#TP1_Down AND #T1_ET50 AND (#NXT_Avance_S3 OR (#MemFN_pHsS3 AND NOT #pHsMx_S3) OR #PTF_Sal_M3)) OR (#T1_ET01 AND NOT #OK_Paro)) AND #PosTR_E1 AND #EstadoZona.Marcha_CBx AND NOT #EstadoVI.Error_Mx AND NOT #EstadoZona.Manual_CBx) OR (NOT #Termico_E1S3 AND #EstadoZona.Rearme_CBx)) AND #ok_tension;
END_REGION

REGION Network 58: OK TOPE DW
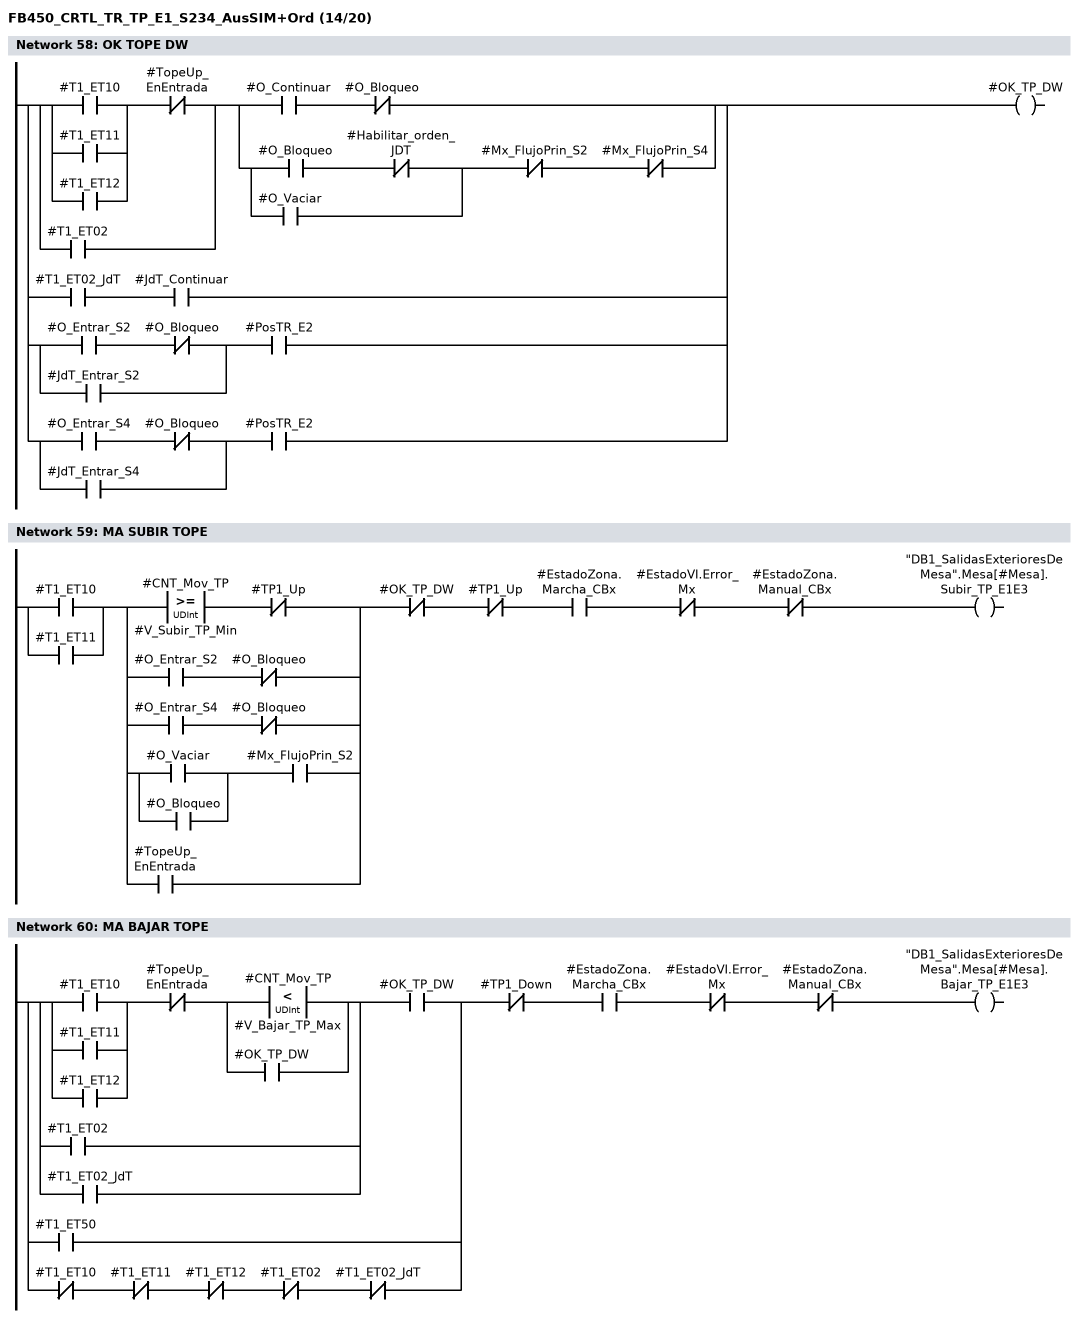
   RUNG wire#powerrail
      Contact( #T1_ET10 )
      wire#w1
      I_Contact( #TopeUp_EnEntrada )
      wire#w2
      Contact( #O_Continuar )
      I_Contact( #O_Bloqueo )
      wire#w3
      Coil( #OK_TP_DW )
   END_RUNG
   RUNG wire#powerrail
      Contact( #T1_ET11 )
   END_RUNG wire#w1
   RUNG wire#powerrail
      Contact( #T1_ET12 )
   END_RUNG wire#w1
   RUNG wire#powerrail
      Contact( #T1_ET02 )
   END_RUNG wire#w2
   RUNG wire#w2
      Contact( #O_Bloqueo )
      I_Contact( #Habilitar_orden_JDT )
      wire#w4
      I_Contact( #Mx_FlujoPrin_S2 )
      I_Contact( #Mx_FlujoPrin_S4 )
   END_RUNG wire#w3
   RUNG wire#w2
      Contact( #O_Vaciar )
   END_RUNG wire#w4
   RUNG wire#powerrail
      Contact( #T1_ET02_JdT )
      Contact( #JdT_Continuar )
   END_RUNG wire#w3
   RUNG wire#powerrail
      Contact( #O_Entrar_S2 )
      I_Contact( #O_Bloqueo )
      wire#w5
      Contact( #PosTR_E2 )
   END_RUNG wire#w3
   RUNG wire#powerrail
      Contact( #JdT_Entrar_S2 )
   END_RUNG wire#w5
   RUNG wire#powerrail
      Contact( #O_Entrar_S4 )
      I_Contact( #O_Bloqueo )
      wire#w6
      Contact( #PosTR_E2 )
   END_RUNG wire#w3
   RUNG wire#powerrail
      Contact( #JdT_Entrar_S4 )
   END_RUNG wire#w6
   // the same network as SCL:
   #OK_TP_DW := ((((#T1_ET10 OR #T1_ET11 OR #T1_ET12) AND NOT #TopeUp_EnEntrada) OR #T1_ET02) AND ((#O_Continuar AND NOT #O_Bloqueo) OR (((#O_Bloqueo AND NOT #Habilitar_orden_JDT) OR #O_Vaciar) AND NOT #Mx_FlujoPrin_S2 AND NOT #Mx_FlujoPrin_S4))) OR (#T1_ET02_JdT AND #JdT_Continuar) OR (((#O_Entrar_S2 AND NOT #O_Bloqueo) OR #JdT_Entrar_S2) AND #PosTR_E2) OR (((#O_Entrar_S4 AND NOT #O_Bloqueo) OR #JdT_Entrar_S4) AND #PosTR_E2);
END_REGION

REGION Network 59: MA SUBIR TOPE
   RUNG wire#powerrail
      Contact( #T1_ET10 )
      wire#w1
      { S7_Templates := "SrcType := UDInt" } GE_Contact(in1 := #CNT_Mov_TP, in2 := #V_Subir_TP_Min)
      I_Contact( #TP1_Up )
      wire#w2
      I_Contact( #OK_TP_DW )
      I_Contact( #TP1_Up )
      Contact( #EstadoZona.Marcha_CBx )
      I_Contact( #EstadoVI.Error_Mx )
      I_Contact( #EstadoZona.Manual_CBx )
      Coil( "DB1_SalidasExterioresDeMesa".Mesa[#Mesa].Subir_TP_E1E3 )
   END_RUNG
   RUNG wire#powerrail
      Contact( #T1_ET11 )
   END_RUNG wire#w1
   RUNG wire#w1
      Contact( #O_Entrar_S2 )
      I_Contact( #O_Bloqueo )
   END_RUNG wire#w2
   RUNG wire#w1
      Contact( #O_Entrar_S4 )
      I_Contact( #O_Bloqueo )
   END_RUNG wire#w2
   RUNG wire#w1
      Contact( #O_Vaciar )
      wire#w3
      Contact( #Mx_FlujoPrin_S2 )
   END_RUNG wire#w2
   RUNG wire#w1
      Contact( #O_Bloqueo )
   END_RUNG wire#w3
   RUNG wire#w1
      Contact( #TopeUp_EnEntrada )
   END_RUNG wire#w2
   // the same network as SCL:
   "DB1_SalidasExterioresDeMesa".Mesa[#Mesa].Subir_TP_E1E3 := (#T1_ET10 OR #T1_ET11) AND (((#CNT_Mov_TP >= #V_Subir_TP_Min) AND NOT #TP1_Up) OR (#O_Entrar_S2 AND NOT #O_Bloqueo) OR (#O_Entrar_S4 AND NOT #O_Bloqueo) OR ((#O_Vaciar OR #O_Bloqueo) AND #Mx_FlujoPrin_S2) OR #TopeUp_EnEntrada) AND NOT #OK_TP_DW AND NOT #TP1_Up AND #EstadoZona.Marcha_CBx AND NOT #EstadoVI.Error_Mx AND NOT #EstadoZona.Manual_CBx;
END_REGION

REGION Network 60: MA BAJAR TOPE
   RUNG wire#powerrail
      Contact( #T1_ET10 )
      wire#w1
      I_Contact( #TopeUp_EnEntrada )
      wire#w2
      { S7_Templates := "SrcType := UDInt" } LT_Contact(in1 := #CNT_Mov_TP, in2 := #V_Bajar_TP_Max)
      wire#w3
      Contact( #OK_TP_DW )
      wire#w4
      I_Contact( #TP1_Down )
      Contact( #EstadoZona.Marcha_CBx )
      I_Contact( #EstadoVI.Error_Mx )
      I_Contact( #EstadoZona.Manual_CBx )
      Coil( "DB1_SalidasExterioresDeMesa".Mesa[#Mesa].Bajar_TP_E1E3 )
   END_RUNG
   RUNG wire#powerrail
      Contact( #T1_ET11 )
   END_RUNG wire#w1
   RUNG wire#powerrail
      Contact( #T1_ET12 )
   END_RUNG wire#w1
   RUNG wire#w2
      Contact( #OK_TP_DW )
   END_RUNG wire#w3
   RUNG wire#powerrail
      Contact( #T1_ET02 )
   END_RUNG wire#w3
   RUNG wire#powerrail
      Contact( #T1_ET02_JdT )
   END_RUNG wire#w3
   RUNG wire#powerrail
      Contact( #T1_ET50 )
   END_RUNG wire#w4
   RUNG wire#powerrail
      I_Contact( #T1_ET10 )
      I_Contact( #T1_ET11 )
      I_Contact( #T1_ET12 )
      I_Contact( #T1_ET02 )
      I_Contact( #T1_ET02_JdT )
   END_RUNG wire#w4
   // the same network as SCL:
   "DB1_SalidasExterioresDeMesa".Mesa[#Mesa].Bajar_TP_E1E3 := (((((#T1_ET10 OR #T1_ET11 OR #T1_ET12) AND NOT #TopeUp_EnEntrada AND ((#CNT_Mov_TP < #V_Bajar_TP_Max) OR #OK_TP_DW)) OR #T1_ET02 OR #T1_ET02_JdT) AND #OK_TP_DW) OR #T1_ET50 OR (NOT #T1_ET10 AND NOT #T1_ET11 AND NOT #T1_ET12 AND NOT #T1_ET02 AND NOT #T1_ET02_JdT)) AND NOT #TP1_Down AND #EstadoZona.Marcha_CBx AND NOT #EstadoVI.Error_Mx AND NOT #EstadoZona.Manual_CBx;
END_REGION

REGION Network 61: Envio de Mensajeria
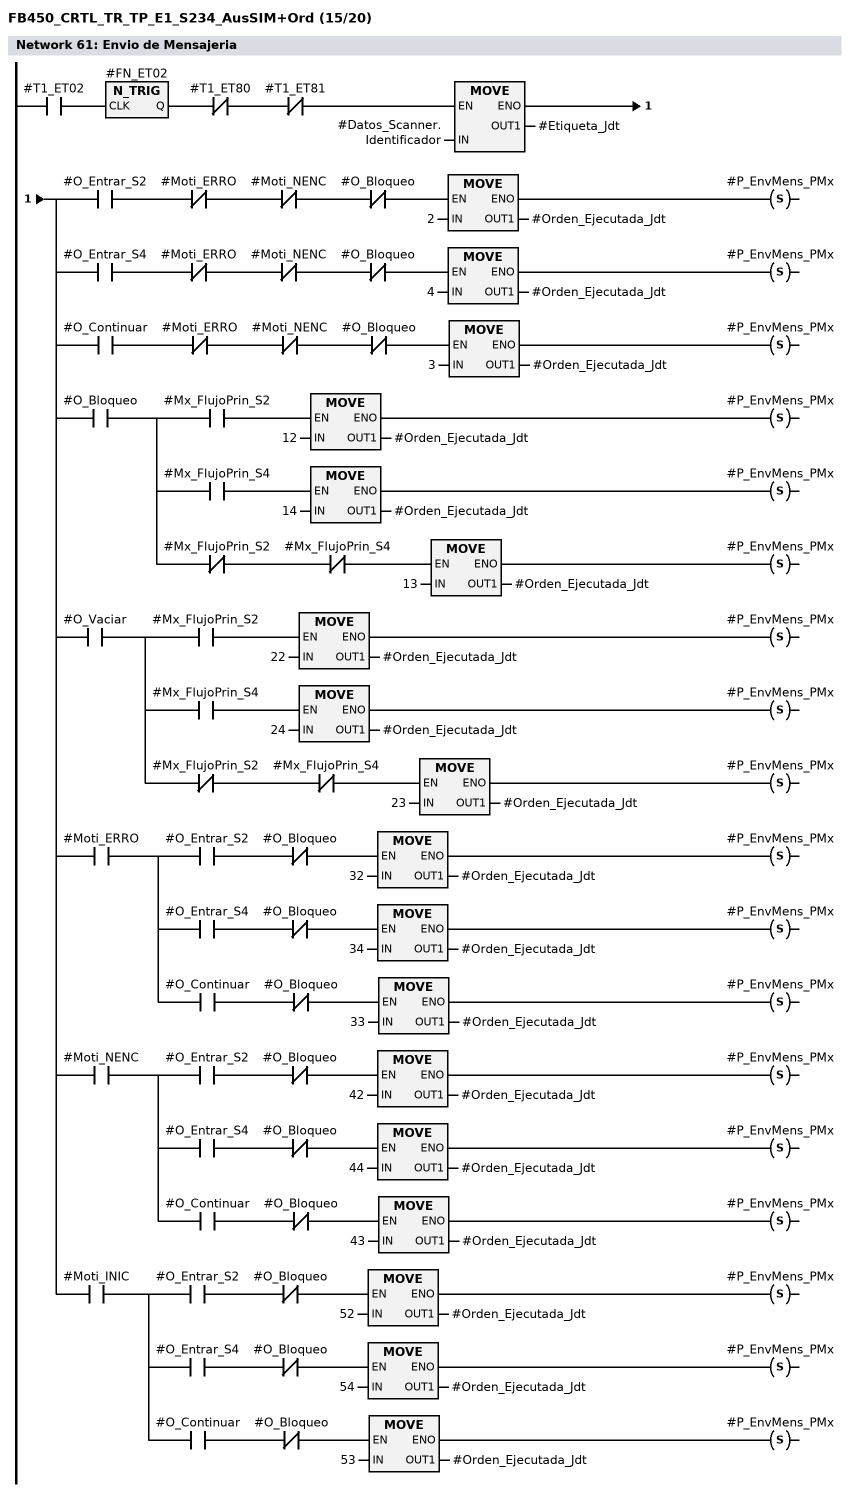
   RUNG wire#powerrail
      Contact( #T1_ET02 )
      N_Trig( #FN_ET02 )
      I_Contact( #T1_ET80 )
      I_Contact( #T1_ET81 )
      { S7_GenerateENO := "TRUE" } Move(in := #Datos_Scanner.Identificador, out1 => #Etiqueta_Jdt)
      wire#w1
      Contact( #O_Entrar_S2 )
      I_Contact( #Moti_ERRO )
      I_Contact( #Moti_NENC )
      I_Contact( #O_Bloqueo )
      { S7_GenerateENO := "TRUE" } Move(in := 2, out1 => #Orden_Ejecutada_Jdt)
      S_Coil( #P_EnvMens_PMx )
   END_RUNG
   RUNG wire#w1
      Contact( #O_Entrar_S4 )
      I_Contact( #Moti_ERRO )
      I_Contact( #Moti_NENC )
      I_Contact( #O_Bloqueo )
      { S7_GenerateENO := "TRUE" } Move(in := 4, out1 => #Orden_Ejecutada_Jdt)
      S_Coil( #P_EnvMens_PMx )
   END_RUNG
   RUNG wire#w1
      Contact( #O_Continuar )
      I_Contact( #Moti_ERRO )
      I_Contact( #Moti_NENC )
      I_Contact( #O_Bloqueo )
      { S7_GenerateENO := "TRUE" } Move(in := 3, out1 => #Orden_Ejecutada_Jdt)
      S_Coil( #P_EnvMens_PMx )
   END_RUNG
   RUNG wire#w1
      Contact( #O_Bloqueo )
      wire#w2
      Contact( #Mx_FlujoPrin_S2 )
      { S7_GenerateENO := "TRUE" } Move(in := 12, out1 => #Orden_Ejecutada_Jdt)
      S_Coil( #P_EnvMens_PMx )
   END_RUNG
   RUNG wire#w2
      Contact( #Mx_FlujoPrin_S4 )
      { S7_GenerateENO := "TRUE" } Move(in := 14, out1 => #Orden_Ejecutada_Jdt)
      S_Coil( #P_EnvMens_PMx )
   END_RUNG
   RUNG wire#w2
      I_Contact( #Mx_FlujoPrin_S2 )
      I_Contact( #Mx_FlujoPrin_S4 )
      { S7_GenerateENO := "TRUE" } Move(in := 13, out1 => #Orden_Ejecutada_Jdt)
      S_Coil( #P_EnvMens_PMx )
   END_RUNG
   RUNG wire#w1
      Contact( #O_Vaciar )
      wire#w3
      Contact( #Mx_FlujoPrin_S2 )
      { S7_GenerateENO := "TRUE" } Move(in := 22, out1 => #Orden_Ejecutada_Jdt)
      S_Coil( #P_EnvMens_PMx )
   END_RUNG
   RUNG wire#w3
      Contact( #Mx_FlujoPrin_S4 )
      { S7_GenerateENO := "TRUE" } Move(in := 24, out1 => #Orden_Ejecutada_Jdt)
      S_Coil( #P_EnvMens_PMx )
   END_RUNG
   RUNG wire#w3
      I_Contact( #Mx_FlujoPrin_S2 )
      I_Contact( #Mx_FlujoPrin_S4 )
      { S7_GenerateENO := "TRUE" } Move(in := 23, out1 => #Orden_Ejecutada_Jdt)
      S_Coil( #P_EnvMens_PMx )
   END_RUNG
   RUNG wire#w1
      Contact( #Moti_ERRO )
      wire#w4
      Contact( #O_Entrar_S2 )
      I_Contact( #O_Bloqueo )
      { S7_GenerateENO := "TRUE" } Move(in := 32, out1 => #Orden_Ejecutada_Jdt)
      S_Coil( #P_EnvMens_PMx )
   END_RUNG
   RUNG wire#w4
      Contact( #O_Entrar_S4 )
      I_Contact( #O_Bloqueo )
      { S7_GenerateENO := "TRUE" } Move(in := 34, out1 => #Orden_Ejecutada_Jdt)
      S_Coil( #P_EnvMens_PMx )
   END_RUNG
   RUNG wire#w4
      Contact( #O_Continuar )
      I_Contact( #O_Bloqueo )
      { S7_GenerateENO := "TRUE" } Move(in := 33, out1 => #Orden_Ejecutada_Jdt)
      S_Coil( #P_EnvMens_PMx )
   END_RUNG
   RUNG wire#w1
      Contact( #Moti_NENC )
      wire#w5
      Contact( #O_Entrar_S2 )
      I_Contact( #O_Bloqueo )
      { S7_GenerateENO := "TRUE" } Move(in := 42, out1 => #Orden_Ejecutada_Jdt)
      S_Coil( #P_EnvMens_PMx )
   END_RUNG
   RUNG wire#w5
      Contact( #O_Entrar_S4 )
      I_Contact( #O_Bloqueo )
      { S7_GenerateENO := "TRUE" } Move(in := 44, out1 => #Orden_Ejecutada_Jdt)
      S_Coil( #P_EnvMens_PMx )
   END_RUNG
   RUNG wire#w5
      Contact( #O_Continuar )
      I_Contact( #O_Bloqueo )
      { S7_GenerateENO := "TRUE" } Move(in := 43, out1 => #Orden_Ejecutada_Jdt)
      S_Coil( #P_EnvMens_PMx )
   END_RUNG
   RUNG wire#w1
      Contact( #Moti_INIC )
      wire#w6
      Contact( #O_Entrar_S2 )
      I_Contact( #O_Bloqueo )
      { S7_GenerateENO := "TRUE" } Move(in := 52, out1 => #Orden_Ejecutada_Jdt)
      S_Coil( #P_EnvMens_PMx )
   END_RUNG
   RUNG wire#w6
      Contact( #O_Entrar_S4 )
      I_Contact( #O_Bloqueo )
      { S7_GenerateENO := "TRUE" } Move(in := 54, out1 => #Orden_Ejecutada_Jdt)
      S_Coil( #P_EnvMens_PMx )
   END_RUNG
   RUNG wire#w6
      Contact( #O_Continuar )
      I_Contact( #O_Bloqueo )
      { S7_GenerateENO := "TRUE" } Move(in := 53, out1 => #Orden_Ejecutada_Jdt)
      S_Coil( #P_EnvMens_PMx )
   END_RUNG
   // the same network as SCL:
   // ENO of a box is taken as its EN; it also drops when the box reports an error
   #_w1 := NOT #T1_ET02 AND #FN_ET02;   // falling edge
   #FN_ET02 := #T1_ET02;
   #_w2 := #_w1 AND NOT #T1_ET80 AND NOT #T1_ET81;
   IF #_w2 THEN #Etiqueta_Jdt := #Datos_Scanner.Identificador; END_IF;
   IF #_w2 AND #O_Entrar_S2 AND NOT #Moti_ERRO AND NOT #Moti_NENC AND NOT #O_Bloqueo THEN
       #Orden_Ejecutada_Jdt := 2;
       #P_EnvMens_PMx := TRUE;
   END_IF;
   IF #_w2 AND #O_Entrar_S4 AND NOT #Moti_ERRO AND NOT #Moti_NENC AND NOT #O_Bloqueo THEN
       #Orden_Ejecutada_Jdt := 4;
       #P_EnvMens_PMx := TRUE;
   END_IF;
   IF #_w2 AND #O_Continuar AND NOT #Moti_ERRO AND NOT #Moti_NENC AND NOT #O_Bloqueo THEN
       #Orden_Ejecutada_Jdt := 3;
       #P_EnvMens_PMx := TRUE;
   END_IF;
   #_w3 := #_w2 AND #O_Bloqueo;
   IF #_w3 AND #Mx_FlujoPrin_S2 THEN
       #Orden_Ejecutada_Jdt := 12;
       #P_EnvMens_PMx := TRUE;
   END_IF;
   IF #_w3 AND #Mx_FlujoPrin_S4 THEN
       #Orden_Ejecutada_Jdt := 14;
       #P_EnvMens_PMx := TRUE;
   END_IF;
   IF #_w3 AND NOT #Mx_FlujoPrin_S2 AND NOT #Mx_FlujoPrin_S4 THEN
       #Orden_Ejecutada_Jdt := 13;
       #P_EnvMens_PMx := TRUE;
   END_IF;
   #_w4 := #_w2 AND #O_Vaciar;
   IF #_w4 AND #Mx_FlujoPrin_S2 THEN
       #Orden_Ejecutada_Jdt := 22;
       #P_EnvMens_PMx := TRUE;
   END_IF;
   IF #_w4 AND #Mx_FlujoPrin_S4 THEN
       #Orden_Ejecutada_Jdt := 24;
       #P_EnvMens_PMx := TRUE;
   END_IF;
   IF #_w4 AND NOT #Mx_FlujoPrin_S2 AND NOT #Mx_FlujoPrin_S4 THEN
       #Orden_Ejecutada_Jdt := 23;
       #P_EnvMens_PMx := TRUE;
   END_IF;
   #_w5 := #_w2 AND #Moti_ERRO;
   IF #_w5 AND #O_Entrar_S2 AND NOT #O_Bloqueo THEN
       #Orden_Ejecutada_Jdt := 32;
       #P_EnvMens_PMx := TRUE;
   END_IF;
   IF #_w5 AND #O_Entrar_S4 AND NOT #O_Bloqueo THEN
       #Orden_Ejecutada_Jdt := 34;
       #P_EnvMens_PMx := TRUE;
   END_IF;
   IF #_w5 AND #O_Continuar AND NOT #O_Bloqueo THEN
       #Orden_Ejecutada_Jdt := 33;
       #P_EnvMens_PMx := TRUE;
   END_IF;
   #_w6 := #_w2 AND #Moti_NENC;
   IF #_w6 AND #O_Entrar_S2 AND NOT #O_Bloqueo THEN
       #Orden_Ejecutada_Jdt := 42;
       #P_EnvMens_PMx := TRUE;
   END_IF;
   IF #_w6 AND #O_Entrar_S4 AND NOT #O_Bloqueo THEN
       #Orden_Ejecutada_Jdt := 44;
       #P_EnvMens_PMx := TRUE;
   END_IF;
   IF #_w6 AND #O_Continuar AND NOT #O_Bloqueo THEN
       #Orden_Ejecutada_Jdt := 43;
       #P_EnvMens_PMx := TRUE;
   END_IF;
   #_w7 := #_w2 AND #Moti_INIC;
   IF #_w7 AND #O_Entrar_S2 AND NOT #O_Bloqueo THEN
       #Orden_Ejecutada_Jdt := 52;
       #P_EnvMens_PMx := TRUE;
   END_IF;
   IF #_w7 AND #O_Entrar_S4 AND NOT #O_Bloqueo THEN
       #Orden_Ejecutada_Jdt := 54;
       #P_EnvMens_PMx := TRUE;
   END_IF;
   IF #_w7 AND #O_Continuar AND NOT #O_Bloqueo THEN
       #Orden_Ejecutada_Jdt := 53;
       #P_EnvMens_PMx := TRUE;
   END_IF;
END_REGION

REGION Network 62: ENVIO MENSAJE CON ORDEN DE JDT
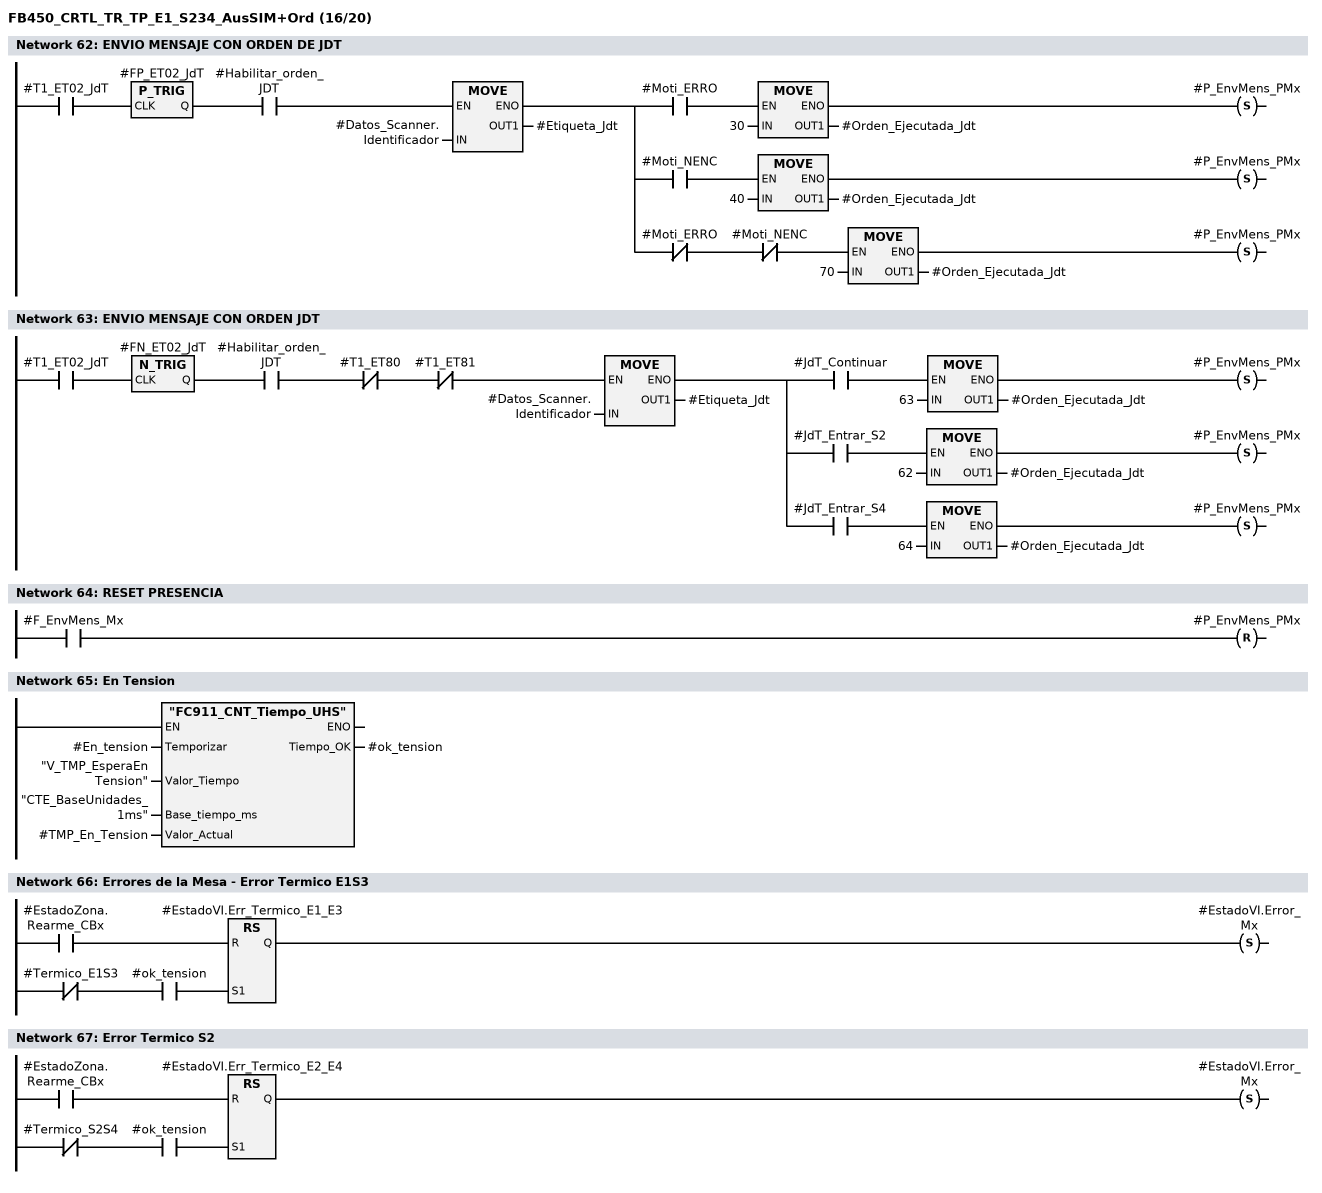
   RUNG wire#powerrail
      Contact( #T1_ET02_JdT )
      P_Trig( #FP_ET02_JdT )
      Contact( #Habilitar_orden_JDT )
      { S7_GenerateENO := "TRUE" } Move(in := #Datos_Scanner.Identificador, out1 => #Etiqueta_Jdt)
      wire#w1
      Contact( #Moti_ERRO )
      { S7_GenerateENO := "TRUE" } Move(in := 30, out1 => #Orden_Ejecutada_Jdt)
      S_Coil( #P_EnvMens_PMx )
   END_RUNG
   RUNG wire#w1
      Contact( #Moti_NENC )
      { S7_GenerateENO := "TRUE" } Move(in := 40, out1 => #Orden_Ejecutada_Jdt)
      S_Coil( #P_EnvMens_PMx )
   END_RUNG
   RUNG wire#w1
      I_Contact( #Moti_ERRO )
      I_Contact( #Moti_NENC )
      { S7_GenerateENO := "TRUE" } Move(in := 70, out1 => #Orden_Ejecutada_Jdt)
      S_Coil( #P_EnvMens_PMx )
   END_RUNG
   // the same network as SCL:
   // ENO of a box is taken as its EN; it also drops when the box reports an error
   #_w1 := #T1_ET02_JdT AND NOT #FP_ET02_JdT;   // rising edge
   #FP_ET02_JdT := #T1_ET02_JdT;
   #_w2 := #_w1 AND #Habilitar_orden_JDT;
   IF #_w2 THEN #Etiqueta_Jdt := #Datos_Scanner.Identificador; END_IF;
   IF #_w2 AND #Moti_ERRO THEN
       #Orden_Ejecutada_Jdt := 30;
       #P_EnvMens_PMx := TRUE;
   END_IF;
   IF #_w2 AND #Moti_NENC THEN
       #Orden_Ejecutada_Jdt := 40;
       #P_EnvMens_PMx := TRUE;
   END_IF;
   IF #_w2 AND NOT #Moti_ERRO AND NOT #Moti_NENC THEN
       #Orden_Ejecutada_Jdt := 70;
       #P_EnvMens_PMx := TRUE;
   END_IF;
END_REGION

REGION Network 63: ENVIO MENSAJE CON ORDEN JDT
   RUNG wire#powerrail
      Contact( #T1_ET02_JdT )
      N_Trig( #FN_ET02_JdT )
      Contact( #Habilitar_orden_JDT )
      I_Contact( #T1_ET80 )
      I_Contact( #T1_ET81 )
      { S7_GenerateENO := "TRUE" } Move(in := #Datos_Scanner.Identificador, out1 => #Etiqueta_Jdt)
      wire#w1
      Contact( #JdT_Continuar )
      { S7_GenerateENO := "TRUE" } Move(in := 63, out1 => #Orden_Ejecutada_Jdt)
      S_Coil( #P_EnvMens_PMx )
   END_RUNG
   RUNG wire#w1
      Contact( #JdT_Entrar_S2 )
      { S7_GenerateENO := "TRUE" } Move(in := 62, out1 => #Orden_Ejecutada_Jdt)
      S_Coil( #P_EnvMens_PMx )
   END_RUNG
   RUNG wire#w1
      Contact( #JdT_Entrar_S4 )
      { S7_GenerateENO := "TRUE" } Move(in := 64, out1 => #Orden_Ejecutada_Jdt)
      S_Coil( #P_EnvMens_PMx )
   END_RUNG
   // the same network as SCL:
   // ENO of a box is taken as its EN; it also drops when the box reports an error
   #_w1 := NOT #T1_ET02_JdT AND #FN_ET02_JdT;   // falling edge
   #FN_ET02_JdT := #T1_ET02_JdT;
   #_w2 := #_w1 AND #Habilitar_orden_JDT AND NOT #T1_ET80 AND NOT #T1_ET81;
   IF #_w2 THEN #Etiqueta_Jdt := #Datos_Scanner.Identificador; END_IF;
   IF #_w2 AND #JdT_Continuar THEN
       #Orden_Ejecutada_Jdt := 63;
       #P_EnvMens_PMx := TRUE;
   END_IF;
   IF #_w2 AND #JdT_Entrar_S2 THEN
       #Orden_Ejecutada_Jdt := 62;
       #P_EnvMens_PMx := TRUE;
   END_IF;
   IF #_w2 AND #JdT_Entrar_S4 THEN
       #Orden_Ejecutada_Jdt := 64;
       #P_EnvMens_PMx := TRUE;
   END_IF;
END_REGION

REGION Network 64: RESET PRESENCIA
   RUNG wire#powerrail
      Contact( #F_EnvMens_Mx )
      R_Coil( #P_EnvMens_PMx )
   END_RUNG
   // the same network as SCL:
   IF #F_EnvMens_Mx THEN #P_EnvMens_PMx := FALSE; END_IF;
END_REGION

REGION Network 65: En Tension
   RUNG wire#powerrail
      "FC911_CNT_Tiempo_UHS"(Temporizar := #En_tension, Valor_Tiempo := "V_TMP_EsperaEnTension", Base_tiempo_ms := "CTE_BaseUnidades_1ms", Valor_Actual := #TMP_En_Tension, Tiempo_OK => #ok_tension)
   END_RUNG
   // the same network as SCL:
   "FC911_CNT_Tiempo_UHS"(Temporizar := #En_tension,
                          Valor_Tiempo := "V_TMP_EsperaEnTension",
                          Base_tiempo_ms := "CTE_BaseUnidades_1ms",
                          Valor_Actual := #TMP_En_Tension,
                          Tiempo_OK => #ok_tension);
END_REGION

REGION Network 66: Errores de la Mesa - Error Termico E1S3
   RUNG wire#powerrail
      Contact( #EstadoZona.Rearme_CBx )
      S_RS(operand := #EstadoVI.Err_Termico_E1_E3, s1 := wire#w1)
      S_Coil( #EstadoVI.Error_Mx )
   END_RUNG
   RUNG wire#powerrail
      I_Contact( #Termico_E1S3 )
      Contact( #ok_tension )
   END_RUNG wire#w1
   // the same network as SCL:
   IF #EstadoZona.Rearme_CBx THEN
       #EstadoVI.Err_Termico_E1_E3 := FALSE;   // RS flip-flop
   END_IF;
   IF NOT #Termico_E1S3 AND #ok_tension THEN #EstadoVI.Err_Termico_E1_E3 := TRUE; END_IF;
   IF #EstadoVI.Err_Termico_E1_E3 THEN #EstadoVI.Error_Mx := TRUE; END_IF;
END_REGION

REGION Network 67: Error Termico S2
   RUNG wire#powerrail
      Contact( #EstadoZona.Rearme_CBx )
      S_RS(operand := #EstadoVI.Err_Termico_E2_E4, s1 := wire#w1)
      S_Coil( #EstadoVI.Error_Mx )
   END_RUNG
   RUNG wire#powerrail
      I_Contact( #Termico_S2S4 )
      Contact( #ok_tension )
   END_RUNG wire#w1
   // the same network as SCL:
   IF #EstadoZona.Rearme_CBx THEN
       #EstadoVI.Err_Termico_E2_E4 := FALSE;   // RS flip-flop
   END_IF;
   IF NOT #Termico_S2S4 AND #ok_tension THEN #EstadoVI.Err_Termico_E2_E4 := TRUE; END_IF;
   IF #EstadoVI.Err_Termico_E2_E4 THEN #EstadoVI.Error_Mx := TRUE; END_IF;
END_REGION

REGION Network 68: timeout transfer
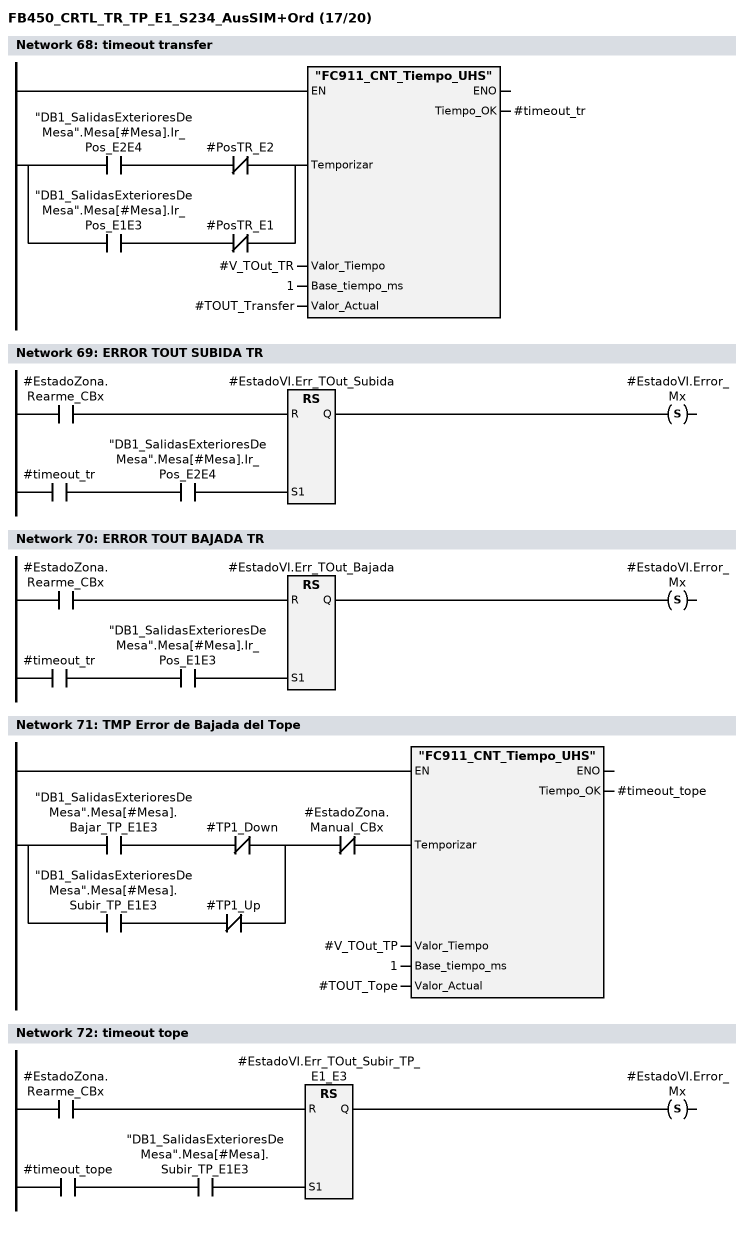
   RUNG wire#powerrail
      "FC911_CNT_Tiempo_UHS"(Temporizar := wire#w1, Valor_Tiempo := #V_TOut_TR, Base_tiempo_ms := 1, Valor_Actual := #TOUT_Transfer, Tiempo_OK => #timeout_tr)
   END_RUNG
   RUNG wire#powerrail
      Contact( "DB1_SalidasExterioresDeMesa".Mesa[#Mesa].Ir_Pos_E2E4 )
      I_Contact( #PosTR_E2 )
   END_RUNG wire#w1
   RUNG wire#powerrail
      Contact( "DB1_SalidasExterioresDeMesa".Mesa[#Mesa].Ir_Pos_E1E3 )
      I_Contact( #PosTR_E1 )
   END_RUNG wire#w1
   // the same network as SCL:
   "FC911_CNT_Tiempo_UHS"(Temporizar := ("DB1_SalidasExterioresDeMesa".Mesa[#Mesa].Ir_Pos_E2E4 AND NOT #PosTR_E2) OR ("DB1_SalidasExterioresDeMesa".Mesa[#Mesa].Ir_Pos_E1E3 AND NOT #PosTR_E1),
                          Valor_Tiempo := #V_TOut_TR,
                          Base_tiempo_ms := 1,
                          Valor_Actual := #TOUT_Transfer,
                          Tiempo_OK => #timeout_tr);
END_REGION

REGION Network 69: ERROR TOUT SUBIDA TR
   RUNG wire#powerrail
      Contact( #EstadoZona.Rearme_CBx )
      S_RS(operand := #EstadoVI.Err_TOut_Subida, s1 := wire#w1)
      S_Coil( #EstadoVI.Error_Mx )
   END_RUNG
   RUNG wire#powerrail
      Contact( #timeout_tr )
      Contact( "DB1_SalidasExterioresDeMesa".Mesa[#Mesa].Ir_Pos_E2E4 )
   END_RUNG wire#w1
   // the same network as SCL:
   IF #EstadoZona.Rearme_CBx THEN
       #EstadoVI.Err_TOut_Subida := FALSE;   // RS flip-flop
   END_IF;
   IF #timeout_tr AND "DB1_SalidasExterioresDeMesa".Mesa[#Mesa].Ir_Pos_E2E4 THEN
       #EstadoVI.Err_TOut_Subida := TRUE;
   END_IF;
   IF #EstadoVI.Err_TOut_Subida THEN #EstadoVI.Error_Mx := TRUE; END_IF;
END_REGION

REGION Network 70: ERROR TOUT BAJADA TR
   RUNG wire#powerrail
      Contact( #EstadoZona.Rearme_CBx )
      S_RS(operand := #EstadoVI.Err_TOut_Bajada, s1 := wire#w1)
      S_Coil( #EstadoVI.Error_Mx )
   END_RUNG
   RUNG wire#powerrail
      Contact( #timeout_tr )
      Contact( "DB1_SalidasExterioresDeMesa".Mesa[#Mesa].Ir_Pos_E1E3 )
   END_RUNG wire#w1
   // the same network as SCL:
   IF #EstadoZona.Rearme_CBx THEN
       #EstadoVI.Err_TOut_Bajada := FALSE;   // RS flip-flop
   END_IF;
   IF #timeout_tr AND "DB1_SalidasExterioresDeMesa".Mesa[#Mesa].Ir_Pos_E1E3 THEN
       #EstadoVI.Err_TOut_Bajada := TRUE;
   END_IF;
   IF #EstadoVI.Err_TOut_Bajada THEN #EstadoVI.Error_Mx := TRUE; END_IF;
END_REGION

REGION Network 71: TMP Error de Bajada del Tope
   RUNG wire#powerrail
      "FC911_CNT_Tiempo_UHS"(Temporizar := wire#w2, Valor_Tiempo := #V_TOut_TP, Base_tiempo_ms := 1, Valor_Actual := #TOUT_Tope, Tiempo_OK => #timeout_tope)
   END_RUNG
   RUNG wire#powerrail
      Contact( "DB1_SalidasExterioresDeMesa".Mesa[#Mesa].Bajar_TP_E1E3 )
      I_Contact( #TP1_Down )
      wire#w1
      I_Contact( #EstadoZona.Manual_CBx )
   END_RUNG wire#w2
   RUNG wire#powerrail
      Contact( "DB1_SalidasExterioresDeMesa".Mesa[#Mesa].Subir_TP_E1E3 )
      I_Contact( #TP1_Up )
   END_RUNG wire#w1
   // the same network as SCL:
   "FC911_CNT_Tiempo_UHS"(Temporizar := (("DB1_SalidasExterioresDeMesa".Mesa[#Mesa].Bajar_TP_E1E3 AND NOT #TP1_Down) OR ("DB1_SalidasExterioresDeMesa".Mesa[#Mesa].Subir_TP_E1E3 AND NOT #TP1_Up)) AND NOT #EstadoZona.Manual_CBx,
                          Valor_Tiempo := #V_TOut_TP,
                          Base_tiempo_ms := 1,
                          Valor_Actual := #TOUT_Tope,
                          Tiempo_OK => #timeout_tope);
END_REGION

REGION Network 72: timeout tope
   RUNG wire#powerrail
      Contact( #EstadoZona.Rearme_CBx )
      S_RS(operand := #EstadoVI.Err_TOut_Subir_TP_E1_E3, s1 := wire#w1)
      S_Coil( #EstadoVI.Error_Mx )
   END_RUNG
   RUNG wire#powerrail
      Contact( #timeout_tope )
      Contact( "DB1_SalidasExterioresDeMesa".Mesa[#Mesa].Subir_TP_E1E3 )
   END_RUNG wire#w1
   // the same network as SCL:
   IF #EstadoZona.Rearme_CBx THEN
       #EstadoVI.Err_TOut_Subir_TP_E1_E3 := FALSE;   // RS flip-flop
   END_IF;
   IF #timeout_tope AND "DB1_SalidasExterioresDeMesa".Mesa[#Mesa].Subir_TP_E1E3 THEN
       #EstadoVI.Err_TOut_Subir_TP_E1_E3 := TRUE;
   END_IF;
   IF #EstadoVI.Err_TOut_Subir_TP_E1_E3 THEN #EstadoVI.Error_Mx := TRUE; END_IF;
END_REGION

REGION Network 73: ERROR BAJAR TOPE
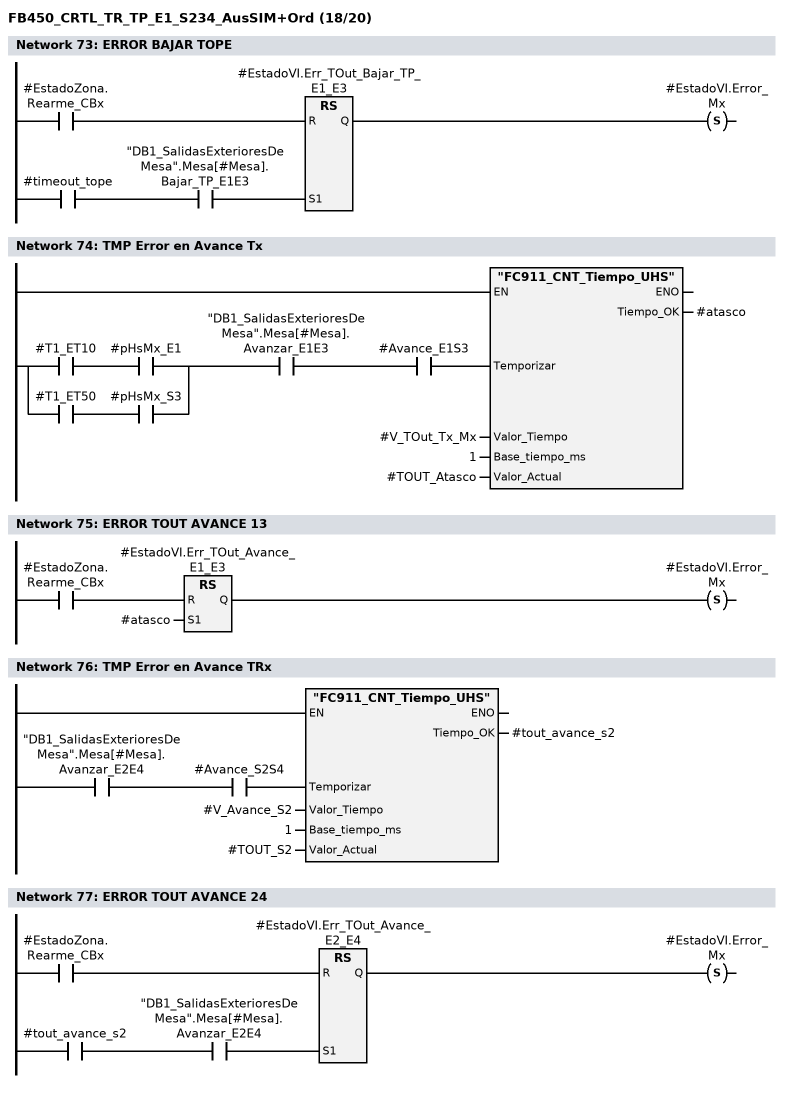
   RUNG wire#powerrail
      Contact( #EstadoZona.Rearme_CBx )
      S_RS(operand := #EstadoVI.Err_TOut_Bajar_TP_E1_E3, s1 := wire#w1)
      S_Coil( #EstadoVI.Error_Mx )
   END_RUNG
   RUNG wire#powerrail
      Contact( #timeout_tope )
      Contact( "DB1_SalidasExterioresDeMesa".Mesa[#Mesa].Bajar_TP_E1E3 )
   END_RUNG wire#w1
   // the same network as SCL:
   IF #EstadoZona.Rearme_CBx THEN
       #EstadoVI.Err_TOut_Bajar_TP_E1_E3 := FALSE;   // RS flip-flop
   END_IF;
   IF #timeout_tope AND "DB1_SalidasExterioresDeMesa".Mesa[#Mesa].Bajar_TP_E1E3 THEN
       #EstadoVI.Err_TOut_Bajar_TP_E1_E3 := TRUE;
   END_IF;
   IF #EstadoVI.Err_TOut_Bajar_TP_E1_E3 THEN #EstadoVI.Error_Mx := TRUE; END_IF;
END_REGION

REGION Network 74: TMP Error en Avance Tx
   RUNG wire#powerrail
      "FC911_CNT_Tiempo_UHS"(Temporizar := wire#w2, Valor_Tiempo := #V_TOut_Tx_Mx, Base_tiempo_ms := 1, Valor_Actual := #TOUT_Atasco, Tiempo_OK => #atasco)
   END_RUNG
   RUNG wire#powerrail
      Contact( #T1_ET10 )
      Contact( #pHsMx_E1 )
      wire#w1
      Contact( "DB1_SalidasExterioresDeMesa".Mesa[#Mesa].Avanzar_E1E3 )
      Contact( #Avance_E1S3 )
   END_RUNG wire#w2
   RUNG wire#powerrail
      Contact( #T1_ET50 )
      Contact( #pHsMx_S3 )
   END_RUNG wire#w1
   // the same network as SCL:
   "FC911_CNT_Tiempo_UHS"(Temporizar := ((#T1_ET10 AND #pHsMx_E1) OR (#T1_ET50 AND #pHsMx_S3)) AND "DB1_SalidasExterioresDeMesa".Mesa[#Mesa].Avanzar_E1E3 AND #Avance_E1S3,
                          Valor_Tiempo := #V_TOut_Tx_Mx,
                          Base_tiempo_ms := 1,
                          Valor_Actual := #TOUT_Atasco,
                          Tiempo_OK => #atasco);
END_REGION

REGION Network 75: ERROR TOUT AVANCE 13
   RUNG wire#powerrail
      Contact( #EstadoZona.Rearme_CBx )
      S_RS(operand := #EstadoVI.Err_TOut_Avance_E1_E3, s1 := #atasco)
      S_Coil( #EstadoVI.Error_Mx )
   END_RUNG
   // the same network as SCL:
   IF #EstadoZona.Rearme_CBx THEN
       #EstadoVI.Err_TOut_Avance_E1_E3 := FALSE;   // RS flip-flop
   END_IF;
   IF #atasco THEN #EstadoVI.Err_TOut_Avance_E1_E3 := TRUE; END_IF;
   IF #EstadoVI.Err_TOut_Avance_E1_E3 THEN #EstadoVI.Error_Mx := TRUE; END_IF;
END_REGION

REGION Network 76: TMP Error en Avance TRx
   RUNG wire#powerrail
      "FC911_CNT_Tiempo_UHS"(Temporizar := wire#w1, Valor_Tiempo := #V_Avance_S2, Base_tiempo_ms := 1, Valor_Actual := #TOUT_S2, Tiempo_OK => #tout_avance_s2)
   END_RUNG
   RUNG wire#powerrail
      Contact( "DB1_SalidasExterioresDeMesa".Mesa[#Mesa].Avanzar_E2E4 )
      Contact( #Avance_S2S4 )
   END_RUNG wire#w1
   // the same network as SCL:
   "FC911_CNT_Tiempo_UHS"(Temporizar := "DB1_SalidasExterioresDeMesa".Mesa[#Mesa].Avanzar_E2E4 AND #Avance_S2S4,
                          Valor_Tiempo := #V_Avance_S2,
                          Base_tiempo_ms := 1,
                          Valor_Actual := #TOUT_S2,
                          Tiempo_OK => #tout_avance_s2);
END_REGION

REGION Network 77: ERROR TOUT AVANCE 24
   RUNG wire#powerrail
      Contact( #EstadoZona.Rearme_CBx )
      S_RS(operand := #EstadoVI.Err_TOut_Avance_E2_E4, s1 := wire#w1)
      S_Coil( #EstadoVI.Error_Mx )
   END_RUNG
   RUNG wire#powerrail
      Contact( #tout_avance_s2 )
      Contact( "DB1_SalidasExterioresDeMesa".Mesa[#Mesa].Avanzar_E2E4 )
   END_RUNG wire#w1
   // the same network as SCL:
   IF #EstadoZona.Rearme_CBx THEN
       #EstadoVI.Err_TOut_Avance_E2_E4 := FALSE;   // RS flip-flop
   END_IF;
   IF #tout_avance_s2 AND "DB1_SalidasExterioresDeMesa".Mesa[#Mesa].Avanzar_E2E4 THEN
       #EstadoVI.Err_TOut_Avance_E2_E4 := TRUE;
   END_IF;
   IF #EstadoVI.Err_TOut_Avance_E2_E4 THEN #EstadoVI.Error_Mx := TRUE; END_IF;
END_REGION

REGION Network 78: Reset y Paro Blando
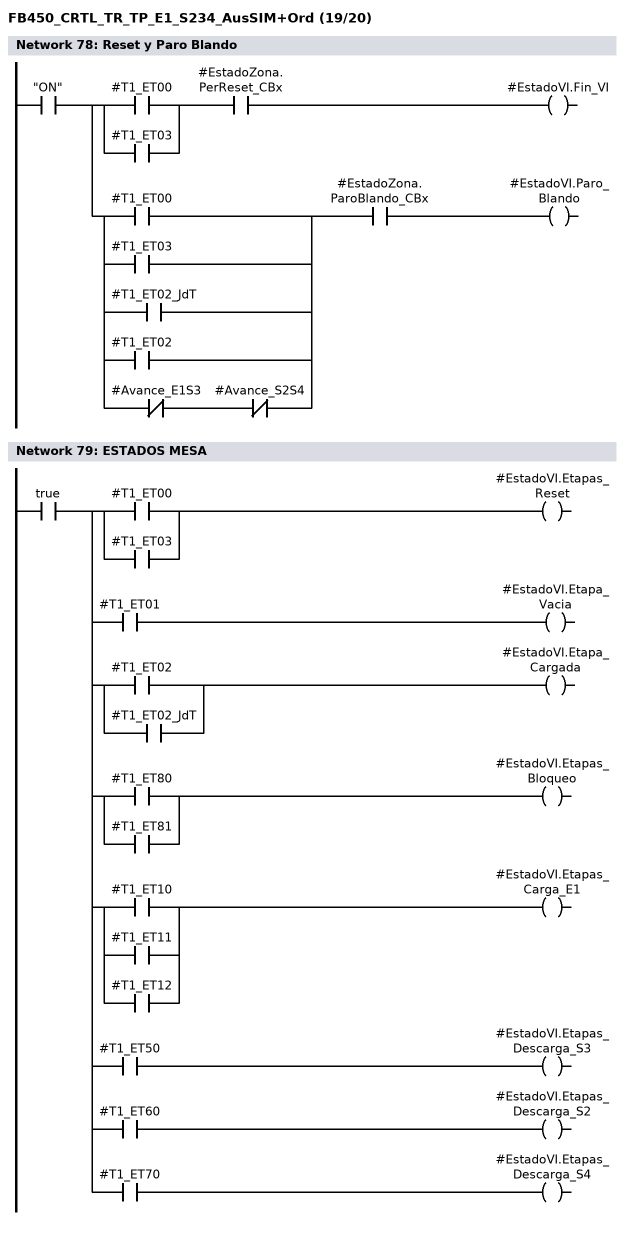
   RUNG wire#powerrail
      Contact( "ON" )
      wire#w1
      Contact( #T1_ET00 )
      wire#w2
      Contact( #EstadoZona.PerReset_CBx )
      Coil( #EstadoVI.Fin_VI )
   END_RUNG
   RUNG wire#w1
      Contact( #T1_ET03 )
   END_RUNG wire#w2
   RUNG wire#w1
      Contact( #T1_ET00 )
      wire#w3
      Contact( #EstadoZona.ParoBlando_CBx )
      Coil( #EstadoVI.Paro_Blando )
   END_RUNG
   RUNG wire#w1
      Contact( #T1_ET03 )
   END_RUNG wire#w3
   RUNG wire#w1
      Contact( #T1_ET02_JdT )
   END_RUNG wire#w3
   RUNG wire#w1
      Contact( #T1_ET02 )
   END_RUNG wire#w3
   RUNG wire#w1
      I_Contact( #Avance_E1S3 )
      I_Contact( #Avance_S2S4 )
   END_RUNG wire#w3
   // the same network as SCL:
   #EstadoVI.Fin_VI := "ON" AND (#T1_ET00 OR #T1_ET03) AND #EstadoZona.PerReset_CBx;
   #EstadoVI.Paro_Blando := "ON" AND (#T1_ET00 OR #T1_ET03 OR #T1_ET02_JdT OR #T1_ET02 OR (NOT #Avance_E1S3 AND NOT #Avance_S2S4)) AND #EstadoZona.ParoBlando_CBx;
END_REGION

REGION Network 79: ESTADOS MESA
   RUNG wire#powerrail
      Contact( true )
      wire#w1
      Contact( #T1_ET00 )
      wire#w2
      Coil( #EstadoVI.Etapas_Reset )
   END_RUNG
   RUNG wire#w1
      Contact( #T1_ET03 )
   END_RUNG wire#w2
   RUNG wire#w1
      Contact( #T1_ET01 )
      Coil( #EstadoVI.Etapa_Vacia )
   END_RUNG
   RUNG wire#w1
      Contact( #T1_ET02 )
      wire#w3
      Coil( #EstadoVI.Etapa_Cargada )
   END_RUNG
   RUNG wire#w1
      Contact( #T1_ET02_JdT )
   END_RUNG wire#w3
   RUNG wire#w1
      Contact( #T1_ET80 )
      wire#w4
      Coil( #EstadoVI.Etapas_Bloqueo )
   END_RUNG
   RUNG wire#w1
      Contact( #T1_ET81 )
   END_RUNG wire#w4
   RUNG wire#w1
      Contact( #T1_ET10 )
      wire#w5
      Coil( #EstadoVI.Etapas_Carga_E1 )
   END_RUNG
   RUNG wire#w1
      Contact( #T1_ET11 )
   END_RUNG wire#w5
   RUNG wire#w1
      Contact( #T1_ET12 )
   END_RUNG wire#w5
   RUNG wire#w1
      Contact( #T1_ET50 )
      Coil( #EstadoVI.Etapas_Descarga_S3 )
   END_RUNG
   RUNG wire#w1
      Contact( #T1_ET60 )
      Coil( #EstadoVI.Etapas_Descarga_S2 )
   END_RUNG
   RUNG wire#w1
      Contact( #T1_ET70 )
      Coil( #EstadoVI.Etapas_Descarga_S4 )
   END_RUNG
   // the same network as SCL:
   #EstadoVI.Etapas_Reset := true AND (#T1_ET00 OR #T1_ET03);
   #EstadoVI.Etapa_Vacia := true AND #T1_ET01;
   #EstadoVI.Etapa_Cargada := true AND (#T1_ET02 OR #T1_ET02_JdT);
   #EstadoVI.Etapas_Bloqueo := true AND (#T1_ET80 OR #T1_ET81);
   #EstadoVI.Etapas_Carga_E1 := true AND (#T1_ET10 OR #T1_ET11 OR #T1_ET12);
   #EstadoVI.Etapas_Descarga_S3 := true AND #T1_ET50;
   #EstadoVI.Etapas_Descarga_S2 := true AND #T1_ET60;
   #EstadoVI.Etapas_Descarga_S4 := true AND #T1_ET70;
END_REGION

REGION Network 80: Entradas Mesas
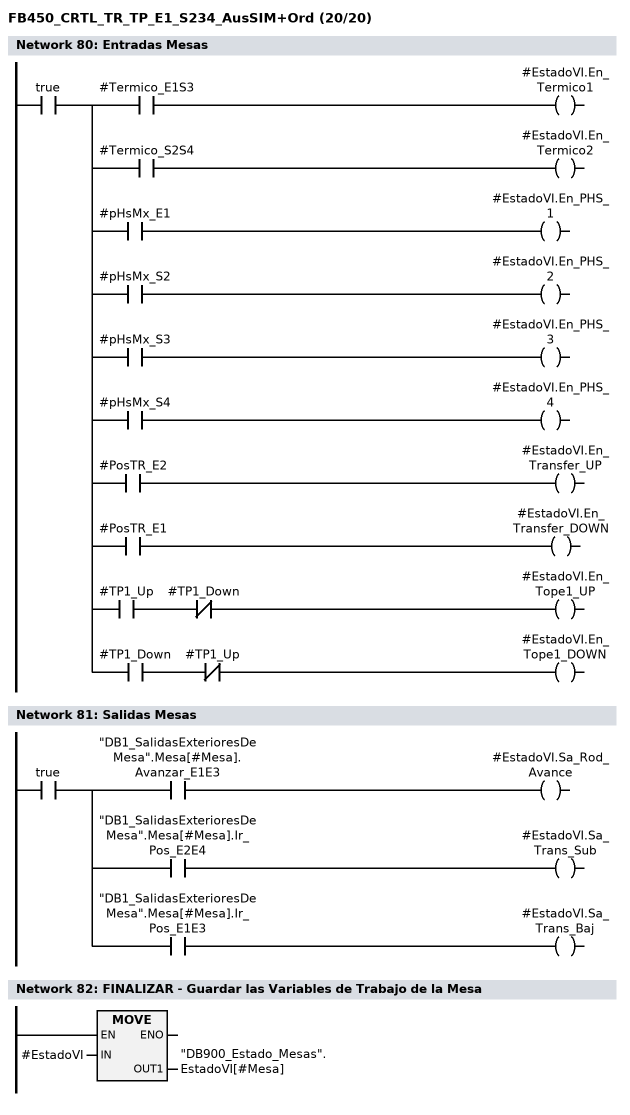
   RUNG wire#powerrail
      Contact( true )
      wire#w1
      Contact( #Termico_E1S3 )
      Coil( #EstadoVI.En_Termico1 )
   END_RUNG
   RUNG wire#w1
      Contact( #Termico_S2S4 )
      Coil( #EstadoVI.En_Termico2 )
   END_RUNG
   RUNG wire#w1
      Contact( #pHsMx_E1 )
      Coil( #EstadoVI.En_PHS_1 )
   END_RUNG
   RUNG wire#w1
      Contact( #pHsMx_S2 )
      Coil( #EstadoVI.En_PHS_2 )
   END_RUNG
   RUNG wire#w1
      Contact( #pHsMx_S3 )
      Coil( #EstadoVI.En_PHS_3 )
   END_RUNG
   RUNG wire#w1
      Contact( #pHsMx_S4 )
      Coil( #EstadoVI.En_PHS_4 )
   END_RUNG
   RUNG wire#w1
      Contact( #PosTR_E2 )
      Coil( #EstadoVI.En_Transfer_UP )
   END_RUNG
   RUNG wire#w1
      Contact( #PosTR_E1 )
      Coil( #EstadoVI.En_Transfer_DOWN )
   END_RUNG
   RUNG wire#w1
      Contact( #TP1_Up )
      I_Contact( #TP1_Down )
      Coil( #EstadoVI.En_Tope1_UP )
   END_RUNG
   RUNG wire#w1
      Contact( #TP1_Down )
      I_Contact( #TP1_Up )
      Coil( #EstadoVI.En_Tope1_DOWN )
   END_RUNG
   // the same network as SCL:
   #EstadoVI.En_Termico1 := true AND #Termico_E1S3;
   #EstadoVI.En_Termico2 := true AND #Termico_S2S4;
   #EstadoVI.En_PHS_1 := true AND #pHsMx_E1;
   #EstadoVI.En_PHS_2 := true AND #pHsMx_S2;
   #EstadoVI.En_PHS_3 := true AND #pHsMx_S3;
   #EstadoVI.En_PHS_4 := true AND #pHsMx_S4;
   #EstadoVI.En_Transfer_UP := true AND #PosTR_E2;
   #EstadoVI.En_Transfer_DOWN := true AND #PosTR_E1;
   #EstadoVI.En_Tope1_UP := true AND #TP1_Up AND NOT #TP1_Down;
   #EstadoVI.En_Tope1_DOWN := true AND #TP1_Down AND NOT #TP1_Up;
END_REGION

REGION Network 81: Salidas Mesas
   RUNG wire#powerrail
      Contact( true )
      wire#w1
      Contact( "DB1_SalidasExterioresDeMesa".Mesa[#Mesa].Avanzar_E1E3 )
      Coil( #EstadoVI.Sa_Rod_Avance )
   END_RUNG
   RUNG wire#w1
      Contact( "DB1_SalidasExterioresDeMesa".Mesa[#Mesa].Ir_Pos_E2E4 )
      Coil( #EstadoVI.Sa_Trans_Sub )
   END_RUNG
   RUNG wire#w1
      Contact( "DB1_SalidasExterioresDeMesa".Mesa[#Mesa].Ir_Pos_E1E3 )
      Coil( #EstadoVI.Sa_Trans_Baj )
   END_RUNG
   // the same network as SCL:
   #EstadoVI.Sa_Rod_Avance := true AND "DB1_SalidasExterioresDeMesa".Mesa[#Mesa].Avanzar_E1E3;
   #EstadoVI.Sa_Trans_Sub := true AND "DB1_SalidasExterioresDeMesa".Mesa[#Mesa].Ir_Pos_E2E4;
   #EstadoVI.Sa_Trans_Baj := true AND "DB1_SalidasExterioresDeMesa".Mesa[#Mesa].Ir_Pos_E1E3;
END_REGION

REGION Network 82: FINALIZAR - Guardar las Variables de Trabajo de la Mesa
   RUNG wire#powerrail
      Move(in := #EstadoVI, out1 => "DB900_Estado_Mesas".EstadoVI[#Mesa])
   END_RUNG
   // the same network as SCL:
   "DB900_Estado_Mesas".EstadoVI[#Mesa] := #EstadoVI;
END_REGION
END_FUNCTION_BLOCK
